// TIA Portal V17 export
// export: Created 2025-07-01T09:59:01.6776162Z, ExportSetting WithDefaults, DisplayName Totally Integrated Automation Portal, DisplayVersion V17 Update 8, DisplayName TIA Portal Openness, DisplayVersion V17 Update 8, DisplayName TIA Portal Version Control Interface, DisplayVersion V17, DisplayName SINAMICS Startdrive Advanced, DisplayVersion V17 SP2, DisplayName SINAMICS Startdrive G110M, G120, G120C, G120D, G120P, G115D, DisplayVersion V17 SP2, DisplayName SINAMICS Startdrive G130, G150, S120, S150, SINAMICS MV, S210, DisplayVersion V17 SP2, DisplayName STEP 7 Professional, DisplayVersion V17 Update 8, DisplayName SINUMERIK ONE STEP 7 Toolbox, DisplayVersion V17 Update 12, DisplayName SINUMERIK ONE PLC Basic Program Plus, DisplayVersion V17 Update 12, DisplayName SINUMERIK 840D sl STEP 7 Toolbox, DisplayVersion V17 Update 12, DisplayName STEP 7 Safety, DisplayVersion V17 Update 6, DisplayName WinCC Advanced, DisplayVersion V17 Update 8
FUNCTION "FC16015_METHOD_CALLS_U2_STA3_COAXIAL" : Void   // FC16015, LAD
{ S7_Optimized_Access := 'FALSE' }
VERSION : 0.1
// PC status values:
// 0-> Idle
// 1-> LaserCalibrating
// 2-> NozzleCalibrating
// 3-> JetCalibrating
// 4-> CladdingCalibrating
// 5-> NozzleAnalysis
// 6-> JetAnalysis
// 7-> CladdingAnalysis
// -1-> Error
// stored: AutoNumber false, IsIECCheckEnabled false, SetENOAutomatically false, UDAEnableTagReadback false
   VAR_TEMP
      AUX_WSTRING_PART_ID_STA3 : WString;
      AUX_WCHARS : Array[0..63] of WChar;
      index : Int;
      ALARM_AUX : Bool;
      TEMP_PULSE : Bool;
      STATUS_BLKMOV : Int;   // STATUS BLKMOV
      ZERO : Int;
   END_VAR
   VAR CONSTANT
      VERSIONS_MAJOR : UInt := 2;
      VERSIONS_MINOR : UInt := 0;
      FC_NUMBER : DInt := 16015;
   END_VAR
   VAR_TEMP   // added for the SCL form of the ladder/FBD networks
      _w1 : Bool;
      _w2 : Bool;
   END_VAR
BEGIN

REGION Network 1: ZERO
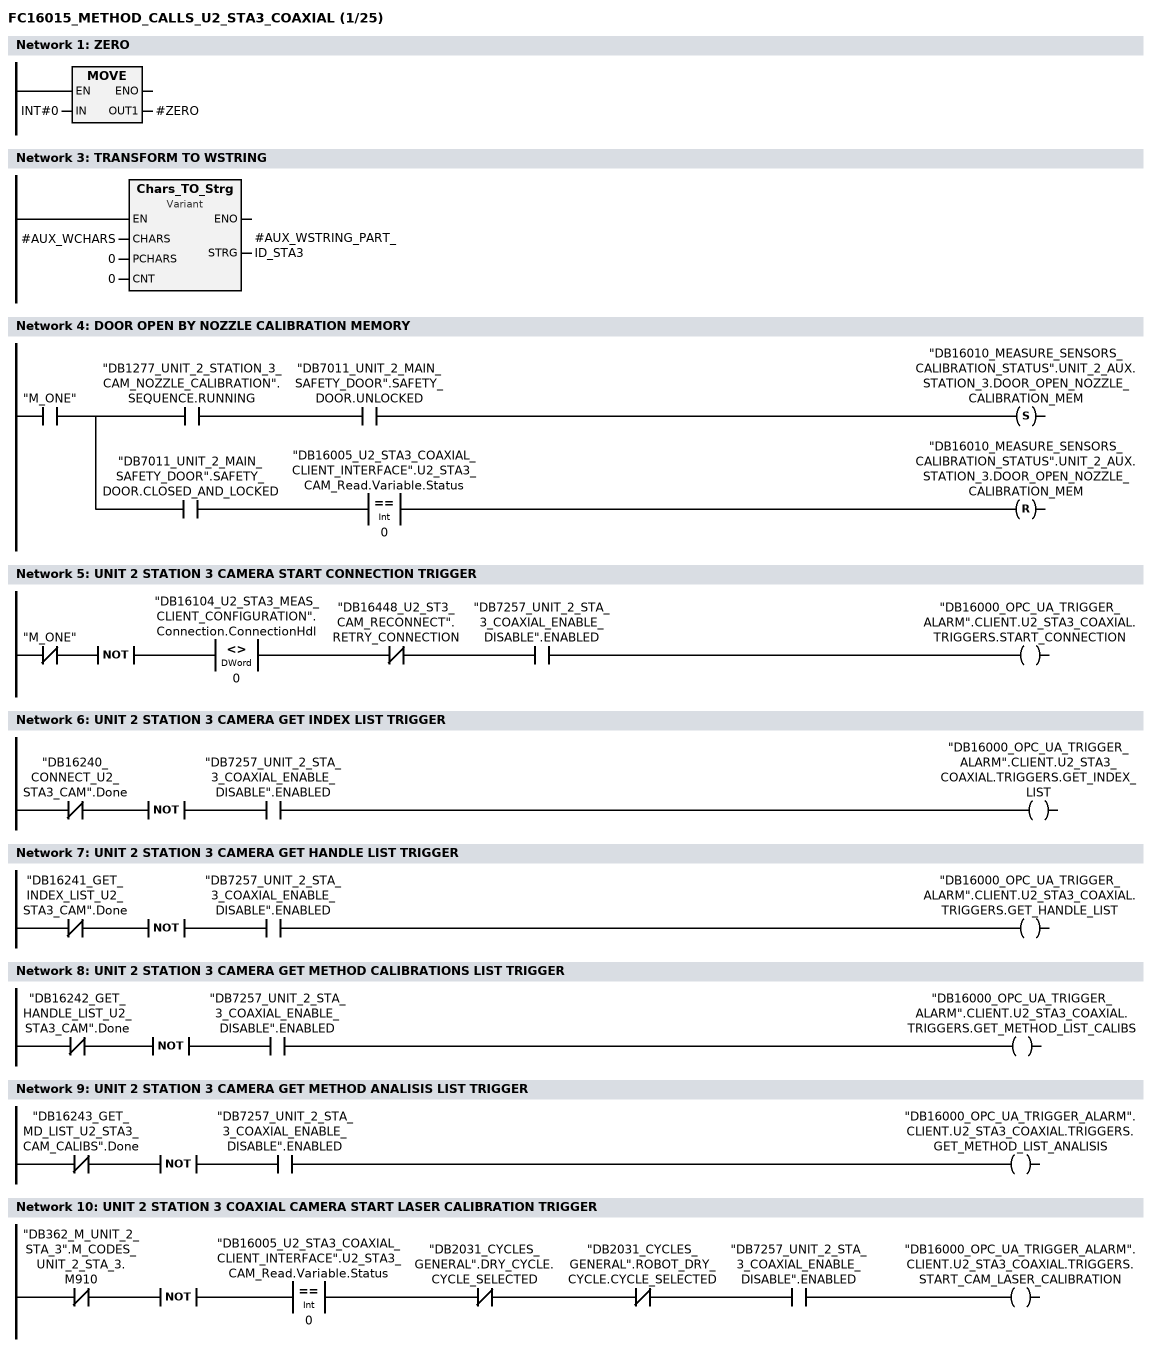
   RUNG wire#powerrail
      { S7_GenerateENO := "TRUE" } Move(in := INT#0, out1 => #ZERO)
   END_RUNG
   // the same network as SCL:
   #ZERO := INT#0;
END_REGION

REGION Network 2 (SCL): TRANSFORM TO WCHARS
   FOR #index := 0 TO 63 DO
       #AUX_WCHARS[#index] := CHAR_TO_WCHAR("DB8000_PART_STATUS".UNIT_2.STATION_3.PART_A.PART_ID[#index]);
   END_FOR;
END_REGION

REGION Network 3: TRANSFORM TO WSTRING
   RUNG wire#powerrail
      { S7_Templates := "[ptr_type := Variant, str_type := WString]" } Chars_TO_Strg(Chars := #AUX_WCHARS, pChars := 0, Cnt := 0, Strg => #AUX_WSTRING_PART_ID_STA3)
   END_RUNG
   // the same network as SCL:
   Chars_TO_Strg(Chars := #AUX_WCHARS, pChars := 0, Cnt := 0, Strg => #AUX_WSTRING_PART_ID_STA3);
END_REGION

REGION Network 4: DOOR OPEN BY NOZZLE CALIBRATION MEMORY
   RUNG wire#powerrail
      Contact( "M_ONE" )
      wire#w1
      Contact( "DB1277_UNIT_2_STATION_3_CAM_NOZZLE_CALIBRATION".SEQUENCE.RUNNING )
      Contact( "DB7011_UNIT_2_MAIN_SAFETY_DOOR".SAFETY_DOOR.UNLOCKED )
      S_Coil( "DB16010_MEASURE_SENSORS_CALIBRATION_STATUS".UNIT_2_AUX.STATION_3.DOOR_OPEN_NOZZLE_CALIBRATION_MEM )
   END_RUNG
   RUNG wire#w1
      Contact( "DB7011_UNIT_2_MAIN_SAFETY_DOOR".SAFETY_DOOR.CLOSED_AND_LOCKED )
      { S7_Templates := "SrcType := Int" } EQ_Contact(in1 := "DB16005_U2_STA3_COAXIAL_CLIENT_INTERFACE".U2_STA3_CAM_Read.Variable.Status, in2 := 0)
      R_Coil( "DB16010_MEASURE_SENSORS_CALIBRATION_STATUS".UNIT_2_AUX.STATION_3.DOOR_OPEN_NOZZLE_CALIBRATION_MEM )
   END_RUNG
   // the same network as SCL:
   IF "M_ONE" AND "DB1277_UNIT_2_STATION_3_CAM_NOZZLE_CALIBRATION".SEQUENCE.RUNNING AND "DB7011_UNIT_2_MAIN_SAFETY_DOOR".SAFETY_DOOR.UNLOCKED THEN
       "DB16010_MEASURE_SENSORS_CALIBRATION_STATUS".UNIT_2_AUX.STATION_3.DOOR_OPEN_NOZZLE_CALIBRATION_MEM := TRUE;
   END_IF;
   IF "M_ONE" AND "DB7011_UNIT_2_MAIN_SAFETY_DOOR".SAFETY_DOOR.CLOSED_AND_LOCKED AND ("DB16005_U2_STA3_COAXIAL_CLIENT_INTERFACE".U2_STA3_CAM_Read.Variable.Status = 0) THEN
       "DB16010_MEASURE_SENSORS_CALIBRATION_STATUS".UNIT_2_AUX.STATION_3.DOOR_OPEN_NOZZLE_CALIBRATION_MEM := FALSE;
   END_IF;
END_REGION

REGION Network 5: UNIT 2 STATION 3 CAMERA START CONNECTION TRIGGER
   RUNG wire#powerrail
      I_Contact( "M_ONE" )
      Not()
      { S7_Templates := "SrcType := DWord" } NE_Contact(in1 := "DB16104_U2_STA3_MEAS_CLIENT_CONFIGURATION".Connection.ConnectionHdl, in2 := 0)
      I_Contact( "DB16448_U2_ST3_CAM_RECONNECT".RETRY_CONNECTION )
      Contact( "DB7257_UNIT_2_STA_3_COAXIAL_ENABLE_DISABLE".ENABLED )
      Coil( "DB16000_OPC_UA_TRIGGER_ALARM".CLIENT.U2_STA3_COAXIAL.TRIGGERS.START_CONNECTION )
   END_RUNG
   // the same network as SCL:
   "DB16000_OPC_UA_TRIGGER_ALARM".CLIENT.U2_STA3_COAXIAL.TRIGGERS.START_CONNECTION := NOT (NOT "M_ONE") AND ("DB16104_U2_STA3_MEAS_CLIENT_CONFIGURATION".Connection.ConnectionHdl <> 0) AND NOT "DB16448_U2_ST3_CAM_RECONNECT".RETRY_CONNECTION AND "DB7257_UNIT_2_STA_3_COAXIAL_ENABLE_DISABLE".ENABLED;
END_REGION

REGION Network 6: UNIT 2 STATION 3 CAMERA GET INDEX LIST TRIGGER
   RUNG wire#powerrail
      I_Contact( "DB16240_CONNECT_U2_STA3_CAM".Done )
      Not()
      Contact( "DB7257_UNIT_2_STA_3_COAXIAL_ENABLE_DISABLE".ENABLED )
      Coil( "DB16000_OPC_UA_TRIGGER_ALARM".CLIENT.U2_STA3_COAXIAL.TRIGGERS.GET_INDEX_LIST )
   END_RUNG
   // the same network as SCL:
   "DB16000_OPC_UA_TRIGGER_ALARM".CLIENT.U2_STA3_COAXIAL.TRIGGERS.GET_INDEX_LIST := NOT (NOT "DB16240_CONNECT_U2_STA3_CAM".Done) AND "DB7257_UNIT_2_STA_3_COAXIAL_ENABLE_DISABLE".ENABLED;
END_REGION

REGION Network 7: UNIT 2 STATION 3 CAMERA GET HANDLE LIST TRIGGER
   RUNG wire#powerrail
      I_Contact( "DB16241_GET_INDEX_LIST_U2_STA3_CAM".Done )
      Not()
      Contact( "DB7257_UNIT_2_STA_3_COAXIAL_ENABLE_DISABLE".ENABLED )
      Coil( "DB16000_OPC_UA_TRIGGER_ALARM".CLIENT.U2_STA3_COAXIAL.TRIGGERS.GET_HANDLE_LIST )
   END_RUNG
   // the same network as SCL:
   "DB16000_OPC_UA_TRIGGER_ALARM".CLIENT.U2_STA3_COAXIAL.TRIGGERS.GET_HANDLE_LIST := NOT (NOT "DB16241_GET_INDEX_LIST_U2_STA3_CAM".Done) AND "DB7257_UNIT_2_STA_3_COAXIAL_ENABLE_DISABLE".ENABLED;
END_REGION

REGION Network 8: UNIT 2 STATION 3 CAMERA GET METHOD CALIBRATIONS LIST TRIGGER
   RUNG wire#powerrail
      I_Contact( "DB16242_GET_HANDLE_LIST_U2_STA3_CAM".Done )
      Not()
      Contact( "DB7257_UNIT_2_STA_3_COAXIAL_ENABLE_DISABLE".ENABLED )
      Coil( "DB16000_OPC_UA_TRIGGER_ALARM".CLIENT.U2_STA3_COAXIAL.TRIGGERS.GET_METHOD_LIST_CALIBS )
   END_RUNG
   // the same network as SCL:
   "DB16000_OPC_UA_TRIGGER_ALARM".CLIENT.U2_STA3_COAXIAL.TRIGGERS.GET_METHOD_LIST_CALIBS := NOT (NOT "DB16242_GET_HANDLE_LIST_U2_STA3_CAM".Done) AND "DB7257_UNIT_2_STA_3_COAXIAL_ENABLE_DISABLE".ENABLED;
END_REGION

REGION Network 9: UNIT 2 STATION 3 CAMERA GET METHOD ANALISIS LIST TRIGGER
   RUNG wire#powerrail
      I_Contact( "DB16243_GET_MD_LIST_U2_STA3_CAM_CALIBS".Done )
      Not()
      Contact( "DB7257_UNIT_2_STA_3_COAXIAL_ENABLE_DISABLE".ENABLED )
      Coil( "DB16000_OPC_UA_TRIGGER_ALARM".CLIENT.U2_STA3_COAXIAL.TRIGGERS.GET_METHOD_LIST_ANALISIS )
   END_RUNG
   // the same network as SCL:
   "DB16000_OPC_UA_TRIGGER_ALARM".CLIENT.U2_STA3_COAXIAL.TRIGGERS.GET_METHOD_LIST_ANALISIS := NOT (NOT "DB16243_GET_MD_LIST_U2_STA3_CAM_CALIBS".Done) AND "DB7257_UNIT_2_STA_3_COAXIAL_ENABLE_DISABLE".ENABLED;
END_REGION

REGION Network 10: UNIT 2 STATION 3 COAXIAL CAMERA START LASER CALIBRATION TRIGGER
   RUNG wire#powerrail
      I_Contact( "DB362_M_UNIT_2_STA_3".M_CODES_UNIT_2_STA_3.M910 )
      Not()
      { S7_Templates := "SrcType := Int" } EQ_Contact(in1 := "DB16005_U2_STA3_COAXIAL_CLIENT_INTERFACE".U2_STA3_CAM_Read.Variable.Status, in2 := 0)
      I_Contact( "DB2031_CYCLES_GENERAL".DRY_CYCLE.CYCLE_SELECTED )
      I_Contact( "DB2031_CYCLES_GENERAL".ROBOT_DRY_CYCLE.CYCLE_SELECTED )
      Contact( "DB7257_UNIT_2_STA_3_COAXIAL_ENABLE_DISABLE".ENABLED )
      Coil( "DB16000_OPC_UA_TRIGGER_ALARM".CLIENT.U2_STA3_COAXIAL.TRIGGERS.START_CAM_LASER_CALIBRATION )
   END_RUNG
   // the same network as SCL:
   "DB16000_OPC_UA_TRIGGER_ALARM".CLIENT.U2_STA3_COAXIAL.TRIGGERS.START_CAM_LASER_CALIBRATION := NOT (NOT "DB362_M_UNIT_2_STA_3".M_CODES_UNIT_2_STA_3.M910) AND ("DB16005_U2_STA3_COAXIAL_CLIENT_INTERFACE".U2_STA3_CAM_Read.Variable.Status = 0) AND NOT "DB2031_CYCLES_GENERAL".DRY_CYCLE.CYCLE_SELECTED AND NOT "DB2031_CYCLES_GENERAL".ROBOT_DRY_CYCLE.CYCLE_SELECTED AND "DB7257_UNIT_2_STA_3_COAXIAL_ENABLE_DISABLE".ENABLED;
END_REGION

REGION Network 11: UNIT 2 STATION 3 COAXIAL CAMERA START NOZZLE CALIBRATION TRIGGER
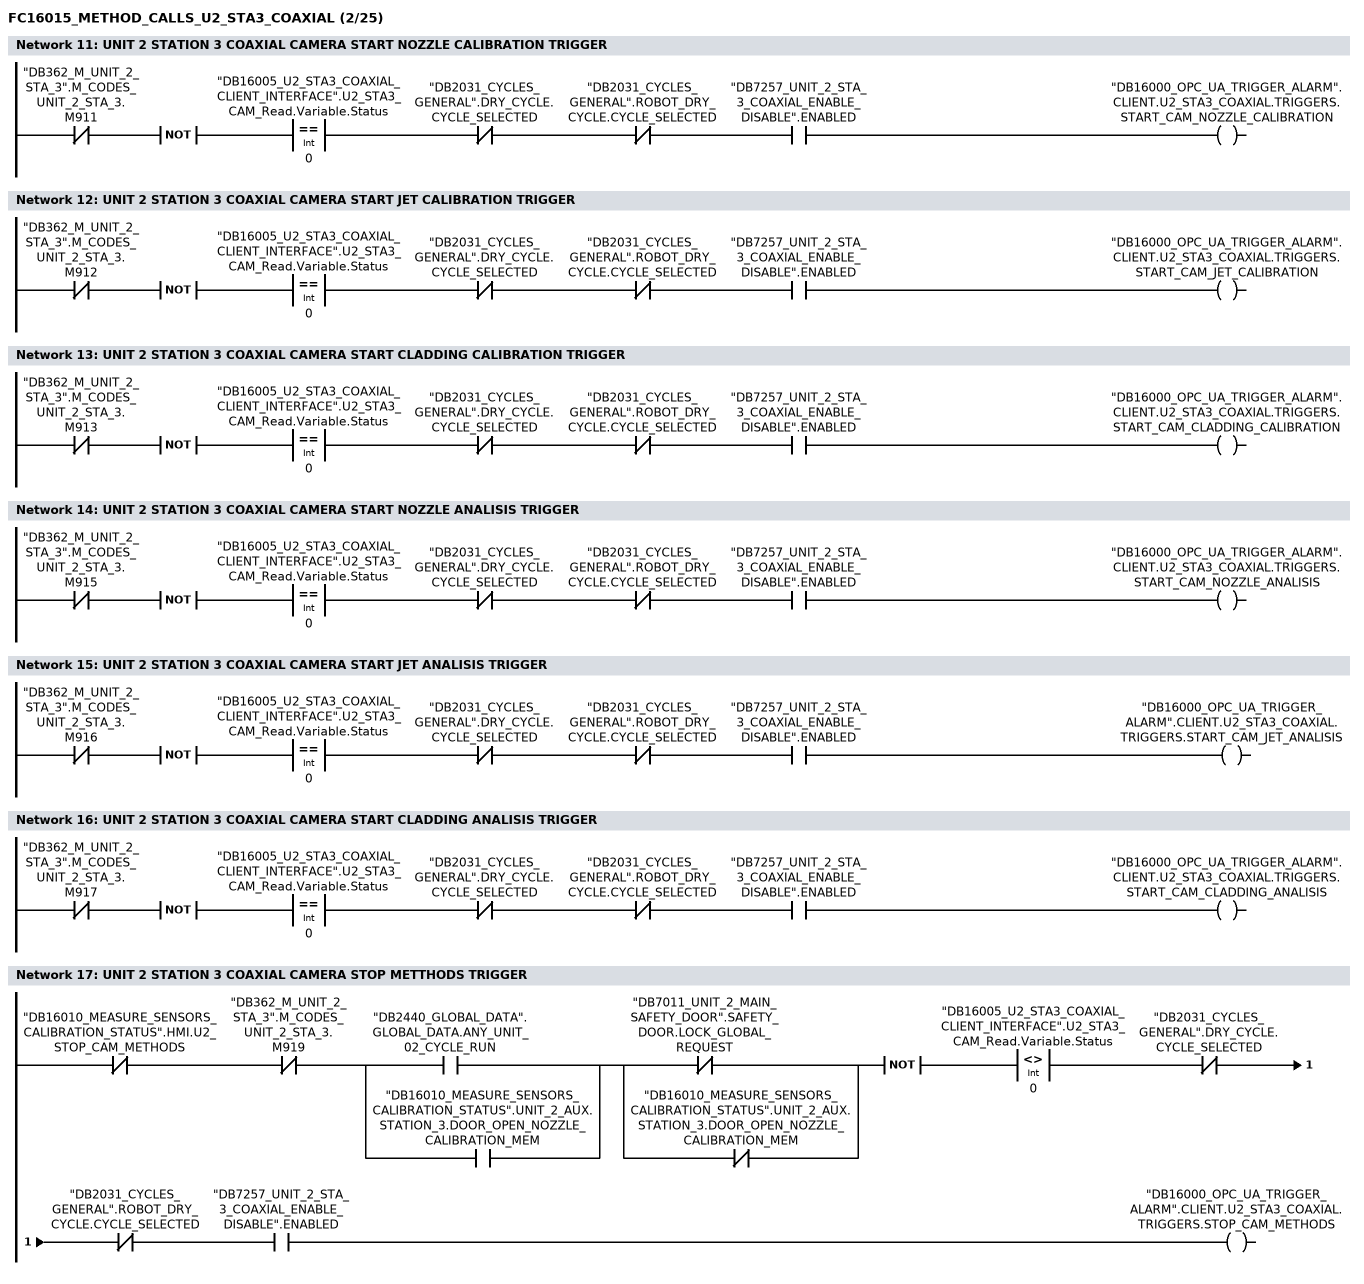
   RUNG wire#powerrail
      I_Contact( "DB362_M_UNIT_2_STA_3".M_CODES_UNIT_2_STA_3.M911 )
      Not()
      { S7_Templates := "SrcType := Int" } EQ_Contact(in1 := "DB16005_U2_STA3_COAXIAL_CLIENT_INTERFACE".U2_STA3_CAM_Read.Variable.Status, in2 := 0)
      I_Contact( "DB2031_CYCLES_GENERAL".DRY_CYCLE.CYCLE_SELECTED )
      I_Contact( "DB2031_CYCLES_GENERAL".ROBOT_DRY_CYCLE.CYCLE_SELECTED )
      Contact( "DB7257_UNIT_2_STA_3_COAXIAL_ENABLE_DISABLE".ENABLED )
      Coil( "DB16000_OPC_UA_TRIGGER_ALARM".CLIENT.U2_STA3_COAXIAL.TRIGGERS.START_CAM_NOZZLE_CALIBRATION )
   END_RUNG
   // the same network as SCL:
   "DB16000_OPC_UA_TRIGGER_ALARM".CLIENT.U2_STA3_COAXIAL.TRIGGERS.START_CAM_NOZZLE_CALIBRATION := NOT (NOT "DB362_M_UNIT_2_STA_3".M_CODES_UNIT_2_STA_3.M911) AND ("DB16005_U2_STA3_COAXIAL_CLIENT_INTERFACE".U2_STA3_CAM_Read.Variable.Status = 0) AND NOT "DB2031_CYCLES_GENERAL".DRY_CYCLE.CYCLE_SELECTED AND NOT "DB2031_CYCLES_GENERAL".ROBOT_DRY_CYCLE.CYCLE_SELECTED AND "DB7257_UNIT_2_STA_3_COAXIAL_ENABLE_DISABLE".ENABLED;
END_REGION

REGION Network 12: UNIT 2 STATION 3 COAXIAL CAMERA START JET CALIBRATION TRIGGER
   RUNG wire#powerrail
      I_Contact( "DB362_M_UNIT_2_STA_3".M_CODES_UNIT_2_STA_3.M912 )
      Not()
      { S7_Templates := "SrcType := Int" } EQ_Contact(in1 := "DB16005_U2_STA3_COAXIAL_CLIENT_INTERFACE".U2_STA3_CAM_Read.Variable.Status, in2 := 0)
      I_Contact( "DB2031_CYCLES_GENERAL".DRY_CYCLE.CYCLE_SELECTED )
      I_Contact( "DB2031_CYCLES_GENERAL".ROBOT_DRY_CYCLE.CYCLE_SELECTED )
      Contact( "DB7257_UNIT_2_STA_3_COAXIAL_ENABLE_DISABLE".ENABLED )
      Coil( "DB16000_OPC_UA_TRIGGER_ALARM".CLIENT.U2_STA3_COAXIAL.TRIGGERS.START_CAM_JET_CALIBRATION )
   END_RUNG
   // the same network as SCL:
   "DB16000_OPC_UA_TRIGGER_ALARM".CLIENT.U2_STA3_COAXIAL.TRIGGERS.START_CAM_JET_CALIBRATION := NOT (NOT "DB362_M_UNIT_2_STA_3".M_CODES_UNIT_2_STA_3.M912) AND ("DB16005_U2_STA3_COAXIAL_CLIENT_INTERFACE".U2_STA3_CAM_Read.Variable.Status = 0) AND NOT "DB2031_CYCLES_GENERAL".DRY_CYCLE.CYCLE_SELECTED AND NOT "DB2031_CYCLES_GENERAL".ROBOT_DRY_CYCLE.CYCLE_SELECTED AND "DB7257_UNIT_2_STA_3_COAXIAL_ENABLE_DISABLE".ENABLED;
END_REGION

REGION Network 13: UNIT 2 STATION 3 COAXIAL CAMERA START CLADDING CALIBRATION TRIGGER
   RUNG wire#powerrail
      I_Contact( "DB362_M_UNIT_2_STA_3".M_CODES_UNIT_2_STA_3.M913 )
      Not()
      { S7_Templates := "SrcType := Int" } EQ_Contact(in1 := "DB16005_U2_STA3_COAXIAL_CLIENT_INTERFACE".U2_STA3_CAM_Read.Variable.Status, in2 := 0)
      I_Contact( "DB2031_CYCLES_GENERAL".DRY_CYCLE.CYCLE_SELECTED )
      I_Contact( "DB2031_CYCLES_GENERAL".ROBOT_DRY_CYCLE.CYCLE_SELECTED )
      Contact( "DB7257_UNIT_2_STA_3_COAXIAL_ENABLE_DISABLE".ENABLED )
      Coil( "DB16000_OPC_UA_TRIGGER_ALARM".CLIENT.U2_STA3_COAXIAL.TRIGGERS.START_CAM_CLADDING_CALIBRATION )
   END_RUNG
   // the same network as SCL:
   "DB16000_OPC_UA_TRIGGER_ALARM".CLIENT.U2_STA3_COAXIAL.TRIGGERS.START_CAM_CLADDING_CALIBRATION := NOT (NOT "DB362_M_UNIT_2_STA_3".M_CODES_UNIT_2_STA_3.M913) AND ("DB16005_U2_STA3_COAXIAL_CLIENT_INTERFACE".U2_STA3_CAM_Read.Variable.Status = 0) AND NOT "DB2031_CYCLES_GENERAL".DRY_CYCLE.CYCLE_SELECTED AND NOT "DB2031_CYCLES_GENERAL".ROBOT_DRY_CYCLE.CYCLE_SELECTED AND "DB7257_UNIT_2_STA_3_COAXIAL_ENABLE_DISABLE".ENABLED;
END_REGION

REGION Network 14: UNIT 2 STATION 3 COAXIAL CAMERA START NOZZLE ANALISIS TRIGGER
   RUNG wire#powerrail
      I_Contact( "DB362_M_UNIT_2_STA_3".M_CODES_UNIT_2_STA_3.M915 )
      Not()
      { S7_Templates := "SrcType := Int" } EQ_Contact(in1 := "DB16005_U2_STA3_COAXIAL_CLIENT_INTERFACE".U2_STA3_CAM_Read.Variable.Status, in2 := 0)
      I_Contact( "DB2031_CYCLES_GENERAL".DRY_CYCLE.CYCLE_SELECTED )
      I_Contact( "DB2031_CYCLES_GENERAL".ROBOT_DRY_CYCLE.CYCLE_SELECTED )
      Contact( "DB7257_UNIT_2_STA_3_COAXIAL_ENABLE_DISABLE".ENABLED )
      Coil( "DB16000_OPC_UA_TRIGGER_ALARM".CLIENT.U2_STA3_COAXIAL.TRIGGERS.START_CAM_NOZZLE_ANALISIS )
   END_RUNG
   // the same network as SCL:
   "DB16000_OPC_UA_TRIGGER_ALARM".CLIENT.U2_STA3_COAXIAL.TRIGGERS.START_CAM_NOZZLE_ANALISIS := NOT (NOT "DB362_M_UNIT_2_STA_3".M_CODES_UNIT_2_STA_3.M915) AND ("DB16005_U2_STA3_COAXIAL_CLIENT_INTERFACE".U2_STA3_CAM_Read.Variable.Status = 0) AND NOT "DB2031_CYCLES_GENERAL".DRY_CYCLE.CYCLE_SELECTED AND NOT "DB2031_CYCLES_GENERAL".ROBOT_DRY_CYCLE.CYCLE_SELECTED AND "DB7257_UNIT_2_STA_3_COAXIAL_ENABLE_DISABLE".ENABLED;
END_REGION

REGION Network 15: UNIT 2 STATION 3 COAXIAL CAMERA START JET ANALISIS TRIGGER
   RUNG wire#powerrail
      I_Contact( "DB362_M_UNIT_2_STA_3".M_CODES_UNIT_2_STA_3.M916 )
      Not()
      { S7_Templates := "SrcType := Int" } EQ_Contact(in1 := "DB16005_U2_STA3_COAXIAL_CLIENT_INTERFACE".U2_STA3_CAM_Read.Variable.Status, in2 := 0)
      I_Contact( "DB2031_CYCLES_GENERAL".DRY_CYCLE.CYCLE_SELECTED )
      I_Contact( "DB2031_CYCLES_GENERAL".ROBOT_DRY_CYCLE.CYCLE_SELECTED )
      Contact( "DB7257_UNIT_2_STA_3_COAXIAL_ENABLE_DISABLE".ENABLED )
      Coil( "DB16000_OPC_UA_TRIGGER_ALARM".CLIENT.U2_STA3_COAXIAL.TRIGGERS.START_CAM_JET_ANALISIS )
   END_RUNG
   // the same network as SCL:
   "DB16000_OPC_UA_TRIGGER_ALARM".CLIENT.U2_STA3_COAXIAL.TRIGGERS.START_CAM_JET_ANALISIS := NOT (NOT "DB362_M_UNIT_2_STA_3".M_CODES_UNIT_2_STA_3.M916) AND ("DB16005_U2_STA3_COAXIAL_CLIENT_INTERFACE".U2_STA3_CAM_Read.Variable.Status = 0) AND NOT "DB2031_CYCLES_GENERAL".DRY_CYCLE.CYCLE_SELECTED AND NOT "DB2031_CYCLES_GENERAL".ROBOT_DRY_CYCLE.CYCLE_SELECTED AND "DB7257_UNIT_2_STA_3_COAXIAL_ENABLE_DISABLE".ENABLED;
END_REGION

REGION Network 16: UNIT 2 STATION 3 COAXIAL CAMERA START CLADDING ANALISIS TRIGGER
   RUNG wire#powerrail
      I_Contact( "DB362_M_UNIT_2_STA_3".M_CODES_UNIT_2_STA_3.M917 )
      Not()
      { S7_Templates := "SrcType := Int" } EQ_Contact(in1 := "DB16005_U2_STA3_COAXIAL_CLIENT_INTERFACE".U2_STA3_CAM_Read.Variable.Status, in2 := 0)
      I_Contact( "DB2031_CYCLES_GENERAL".DRY_CYCLE.CYCLE_SELECTED )
      I_Contact( "DB2031_CYCLES_GENERAL".ROBOT_DRY_CYCLE.CYCLE_SELECTED )
      Contact( "DB7257_UNIT_2_STA_3_COAXIAL_ENABLE_DISABLE".ENABLED )
      Coil( "DB16000_OPC_UA_TRIGGER_ALARM".CLIENT.U2_STA3_COAXIAL.TRIGGERS.START_CAM_CLADDING_ANALISIS )
   END_RUNG
   // the same network as SCL:
   "DB16000_OPC_UA_TRIGGER_ALARM".CLIENT.U2_STA3_COAXIAL.TRIGGERS.START_CAM_CLADDING_ANALISIS := NOT (NOT "DB362_M_UNIT_2_STA_3".M_CODES_UNIT_2_STA_3.M917) AND ("DB16005_U2_STA3_COAXIAL_CLIENT_INTERFACE".U2_STA3_CAM_Read.Variable.Status = 0) AND NOT "DB2031_CYCLES_GENERAL".DRY_CYCLE.CYCLE_SELECTED AND NOT "DB2031_CYCLES_GENERAL".ROBOT_DRY_CYCLE.CYCLE_SELECTED AND "DB7257_UNIT_2_STA_3_COAXIAL_ENABLE_DISABLE".ENABLED;
END_REGION

REGION Network 17: UNIT 2 STATION 3 COAXIAL CAMERA STOP METTHODS TRIGGER
   RUNG wire#powerrail
      I_Contact( "DB16010_MEASURE_SENSORS_CALIBRATION_STATUS".HMI.U2_STOP_CAM_METHODS )
      I_Contact( "DB362_M_UNIT_2_STA_3".M_CODES_UNIT_2_STA_3.M919 )
      wire#w1
      Contact( "DB2440_GLOBAL_DATA".GLOBAL_DATA.ANY_UNIT_02_CYCLE_RUN )
      wire#w2
      I_Contact( "DB7011_UNIT_2_MAIN_SAFETY_DOOR".SAFETY_DOOR.LOCK_GLOBAL_REQUEST )
      wire#w3
      Not()
      { S7_Templates := "SrcType := Int" } NE_Contact(in1 := "DB16005_U2_STA3_COAXIAL_CLIENT_INTERFACE".U2_STA3_CAM_Read.Variable.Status, in2 := 0)
      I_Contact( "DB2031_CYCLES_GENERAL".DRY_CYCLE.CYCLE_SELECTED )
      I_Contact( "DB2031_CYCLES_GENERAL".ROBOT_DRY_CYCLE.CYCLE_SELECTED )
      Contact( "DB7257_UNIT_2_STA_3_COAXIAL_ENABLE_DISABLE".ENABLED )
      Coil( "DB16000_OPC_UA_TRIGGER_ALARM".CLIENT.U2_STA3_COAXIAL.TRIGGERS.STOP_CAM_METHODS )
   END_RUNG
   RUNG wire#w1
      Contact( "DB16010_MEASURE_SENSORS_CALIBRATION_STATUS".UNIT_2_AUX.STATION_3.DOOR_OPEN_NOZZLE_CALIBRATION_MEM )
   END_RUNG wire#w2
   RUNG wire#w2
      I_Contact( "DB16010_MEASURE_SENSORS_CALIBRATION_STATUS".UNIT_2_AUX.STATION_3.DOOR_OPEN_NOZZLE_CALIBRATION_MEM )
   END_RUNG wire#w3
   // the same network as SCL:
   "DB16000_OPC_UA_TRIGGER_ALARM".CLIENT.U2_STA3_COAXIAL.TRIGGERS.STOP_CAM_METHODS := NOT (NOT "DB16010_MEASURE_SENSORS_CALIBRATION_STATUS".HMI.U2_STOP_CAM_METHODS AND NOT "DB362_M_UNIT_2_STA_3".M_CODES_UNIT_2_STA_3.M919 AND ("DB2440_GLOBAL_DATA".GLOBAL_DATA.ANY_UNIT_02_CYCLE_RUN OR "DB16010_MEASURE_SENSORS_CALIBRATION_STATUS".UNIT_2_AUX.STATION_3.DOOR_OPEN_NOZZLE_CALIBRATION_MEM) AND (NOT "DB7011_UNIT_2_MAIN_SAFETY_DOOR".SAFETY_DOOR.LOCK_GLOBAL_REQUEST OR NOT "DB16010_MEASURE_SENSORS_CALIBRATION_STATUS".UNIT_2_AUX.STATION_3.DOOR_OPEN_NOZZLE_CALIBRATION_MEM)) AND ("DB16005_U2_STA3_COAXIAL_CLIENT_INTERFACE".U2_STA3_CAM_Read.Variable.Status <> 0) AND NOT "DB2031_CYCLES_GENERAL".DRY_CYCLE.CYCLE_SELECTED AND NOT "DB2031_CYCLES_GENERAL".ROBOT_DRY_CYCLE.CYCLE_SELECTED AND "DB7257_UNIT_2_STA_3_COAXIAL_ENABLE_DISABLE".ENABLED;
END_REGION

REGION Network 18: UNIT 2 STATION 3 COAXIAL CAMERA RESET PC TRIGGER
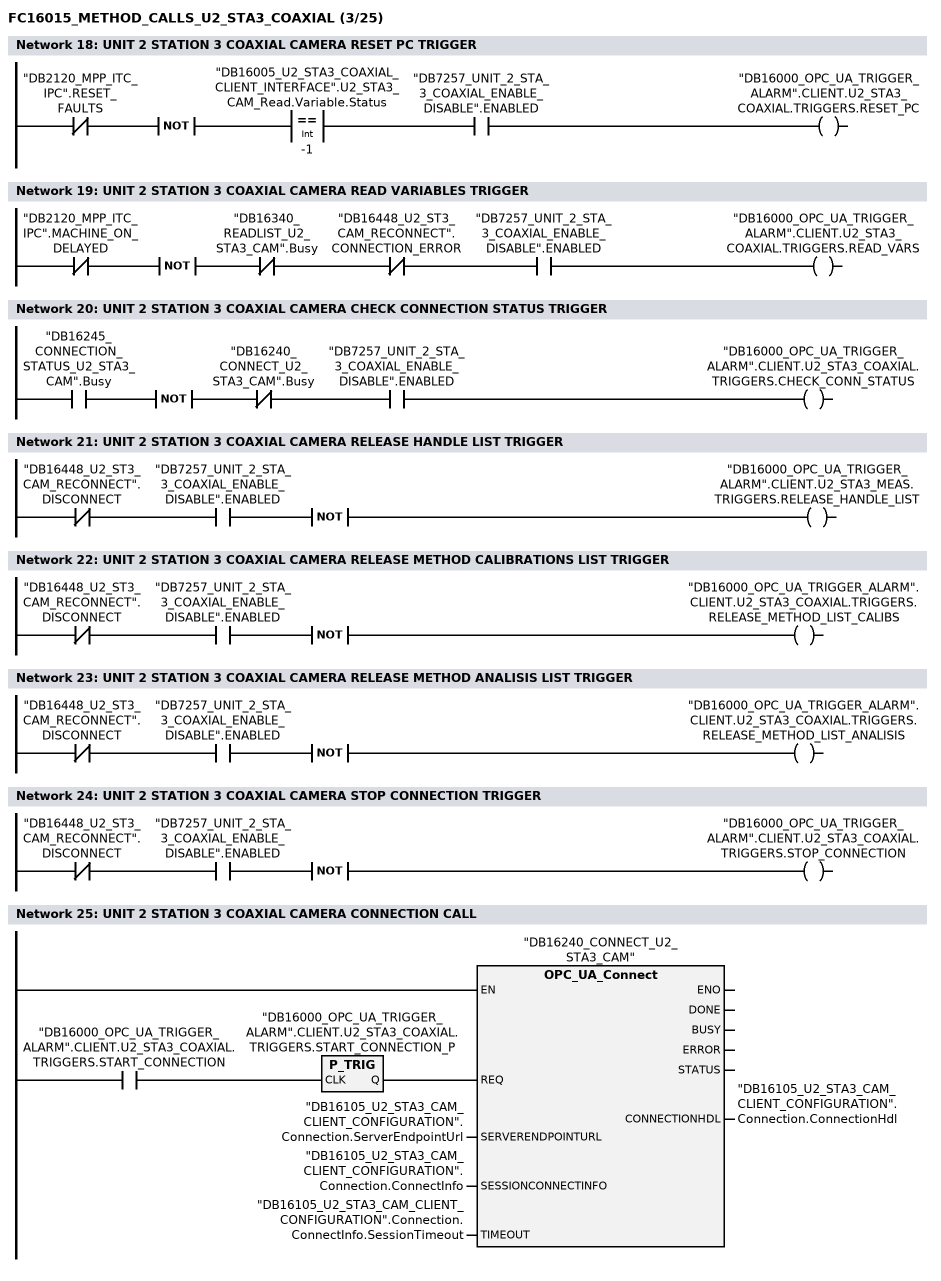
   RUNG wire#powerrail
      I_Contact( "DB2120_MPP_ITC_IPC".RESET_FAULTS )
      Not()
      { S7_Templates := "SrcType := Int" } EQ_Contact(in1 := "DB16005_U2_STA3_COAXIAL_CLIENT_INTERFACE".U2_STA3_CAM_Read.Variable.Status, in2 := -1)
      Contact( "DB7257_UNIT_2_STA_3_COAXIAL_ENABLE_DISABLE".ENABLED )
      Coil( "DB16000_OPC_UA_TRIGGER_ALARM".CLIENT.U2_STA3_COAXIAL.TRIGGERS.RESET_PC )
   END_RUNG
   // the same network as SCL:
   "DB16000_OPC_UA_TRIGGER_ALARM".CLIENT.U2_STA3_COAXIAL.TRIGGERS.RESET_PC := NOT (NOT "DB2120_MPP_ITC_IPC".RESET_FAULTS) AND ("DB16005_U2_STA3_COAXIAL_CLIENT_INTERFACE".U2_STA3_CAM_Read.Variable.Status = (-1)) AND "DB7257_UNIT_2_STA_3_COAXIAL_ENABLE_DISABLE".ENABLED;
END_REGION

REGION Network 19: UNIT 2 STATION 3 COAXIAL CAMERA READ VARIABLES TRIGGER
   RUNG wire#powerrail
      I_Contact( "DB2120_MPP_ITC_IPC".MACHINE_ON_DELAYED )
      Not()
      I_Contact( "DB16340_READLIST_U2_STA3_CAM".Busy )
      I_Contact( "DB16448_U2_ST3_CAM_RECONNECT".CONNECTION_ERROR )
      Contact( "DB7257_UNIT_2_STA_3_COAXIAL_ENABLE_DISABLE".ENABLED )
      Coil( "DB16000_OPC_UA_TRIGGER_ALARM".CLIENT.U2_STA3_COAXIAL.TRIGGERS.READ_VARS )
   END_RUNG
   // the same network as SCL:
   "DB16000_OPC_UA_TRIGGER_ALARM".CLIENT.U2_STA3_COAXIAL.TRIGGERS.READ_VARS := NOT (NOT "DB2120_MPP_ITC_IPC".MACHINE_ON_DELAYED) AND NOT "DB16340_READLIST_U2_STA3_CAM".Busy AND NOT "DB16448_U2_ST3_CAM_RECONNECT".CONNECTION_ERROR AND "DB7257_UNIT_2_STA_3_COAXIAL_ENABLE_DISABLE".ENABLED;
END_REGION

REGION Network 20: UNIT 2 STATION 3 COAXIAL CAMERA CHECK CONNECTION STATUS TRIGGER
   RUNG wire#powerrail
      Contact( "DB16245_CONNECTION_STATUS_U2_STA3_CAM".Busy )
      Not()
      I_Contact( "DB16240_CONNECT_U2_STA3_CAM".Busy )
      Contact( "DB7257_UNIT_2_STA_3_COAXIAL_ENABLE_DISABLE".ENABLED )
      Coil( "DB16000_OPC_UA_TRIGGER_ALARM".CLIENT.U2_STA3_COAXIAL.TRIGGERS.CHECK_CONN_STATUS )
   END_RUNG
   // the same network as SCL:
   "DB16000_OPC_UA_TRIGGER_ALARM".CLIENT.U2_STA3_COAXIAL.TRIGGERS.CHECK_CONN_STATUS := NOT "DB16245_CONNECTION_STATUS_U2_STA3_CAM".Busy AND NOT "DB16240_CONNECT_U2_STA3_CAM".Busy AND "DB7257_UNIT_2_STA_3_COAXIAL_ENABLE_DISABLE".ENABLED;
END_REGION

REGION Network 21: UNIT 2 STATION 3 COAXIAL CAMERA RELEASE HANDLE LIST TRIGGER
   RUNG wire#powerrail
      I_Contact( "DB16448_U2_ST3_CAM_RECONNECT".DISCONNECT )
      Contact( "DB7257_UNIT_2_STA_3_COAXIAL_ENABLE_DISABLE".ENABLED )
      Not()
      Coil( "DB16000_OPC_UA_TRIGGER_ALARM".CLIENT.U2_STA3_MEAS.TRIGGERS.RELEASE_HANDLE_LIST )
   END_RUNG
   // the same network as SCL:
   "DB16000_OPC_UA_TRIGGER_ALARM".CLIENT.U2_STA3_MEAS.TRIGGERS.RELEASE_HANDLE_LIST := NOT (NOT "DB16448_U2_ST3_CAM_RECONNECT".DISCONNECT AND "DB7257_UNIT_2_STA_3_COAXIAL_ENABLE_DISABLE".ENABLED);
END_REGION

REGION Network 22: UNIT 2 STATION 3 COAXIAL CAMERA RELEASE METHOD CALIBRATIONS LIST TRIGGER
   RUNG wire#powerrail
      I_Contact( "DB16448_U2_ST3_CAM_RECONNECT".DISCONNECT )
      Contact( "DB7257_UNIT_2_STA_3_COAXIAL_ENABLE_DISABLE".ENABLED )
      Not()
      Coil( "DB16000_OPC_UA_TRIGGER_ALARM".CLIENT.U2_STA3_COAXIAL.TRIGGERS.RELEASE_METHOD_LIST_CALIBS )
   END_RUNG
   // the same network as SCL:
   "DB16000_OPC_UA_TRIGGER_ALARM".CLIENT.U2_STA3_COAXIAL.TRIGGERS.RELEASE_METHOD_LIST_CALIBS := NOT (NOT "DB16448_U2_ST3_CAM_RECONNECT".DISCONNECT AND "DB7257_UNIT_2_STA_3_COAXIAL_ENABLE_DISABLE".ENABLED);
END_REGION

REGION Network 23: UNIT 2 STATION 3 COAXIAL CAMERA RELEASE METHOD ANALISIS LIST TRIGGER
   RUNG wire#powerrail
      I_Contact( "DB16448_U2_ST3_CAM_RECONNECT".DISCONNECT )
      Contact( "DB7257_UNIT_2_STA_3_COAXIAL_ENABLE_DISABLE".ENABLED )
      Not()
      Coil( "DB16000_OPC_UA_TRIGGER_ALARM".CLIENT.U2_STA3_COAXIAL.TRIGGERS.RELEASE_METHOD_LIST_ANALISIS )
   END_RUNG
   // the same network as SCL:
   "DB16000_OPC_UA_TRIGGER_ALARM".CLIENT.U2_STA3_COAXIAL.TRIGGERS.RELEASE_METHOD_LIST_ANALISIS := NOT (NOT "DB16448_U2_ST3_CAM_RECONNECT".DISCONNECT AND "DB7257_UNIT_2_STA_3_COAXIAL_ENABLE_DISABLE".ENABLED);
END_REGION

REGION Network 24: UNIT 2 STATION 3 COAXIAL CAMERA STOP CONNECTION TRIGGER
   RUNG wire#powerrail
      I_Contact( "DB16448_U2_ST3_CAM_RECONNECT".DISCONNECT )
      Contact( "DB7257_UNIT_2_STA_3_COAXIAL_ENABLE_DISABLE".ENABLED )
      Not()
      Coil( "DB16000_OPC_UA_TRIGGER_ALARM".CLIENT.U2_STA3_COAXIAL.TRIGGERS.STOP_CONNECTION )
   END_RUNG
   // the same network as SCL:
   "DB16000_OPC_UA_TRIGGER_ALARM".CLIENT.U2_STA3_COAXIAL.TRIGGERS.STOP_CONNECTION := NOT (NOT "DB16448_U2_ST3_CAM_RECONNECT".DISCONNECT AND "DB7257_UNIT_2_STA_3_COAXIAL_ENABLE_DISABLE".ENABLED);
END_REGION

REGION Network 25: UNIT 2 STATION 3 COAXIAL CAMERA CONNECTION CALL
   RUNG wire#powerrail
      "DB16240_CONNECT_U2_STA3_CAM".OPC_UA_Connect(REQ := wire#w1, ServerEndpointUrl := "DB16105_U2_STA3_CAM_CLIENT_CONFIGURATION".Connection.ServerEndpointUrl, SessionConnectInfo := "DB16105_U2_STA3_CAM_CLIENT_CONFIGURATION".Connection.ConnectInfo, Timeout := "DB16105_U2_STA3_CAM_CLIENT_CONFIGURATION".Connection.ConnectInfo.SessionTimeout, Done =>, Busy =>, Error =>, Status =>, ConnectionHdl => "DB16105_U2_STA3_CAM_CLIENT_CONFIGURATION".Connection.ConnectionHdl)
   END_RUNG
   RUNG wire#powerrail
      Contact( "DB16000_OPC_UA_TRIGGER_ALARM".CLIENT.U2_STA3_COAXIAL.TRIGGERS.START_CONNECTION )
      P_Trig( "DB16000_OPC_UA_TRIGGER_ALARM".CLIENT.U2_STA3_COAXIAL.TRIGGERS.START_CONNECTION_P )
   END_RUNG wire#w1
   // the same network as SCL:
   #_w1 := "DB16000_OPC_UA_TRIGGER_ALARM".CLIENT.U2_STA3_COAXIAL.TRIGGERS.START_CONNECTION AND NOT "DB16000_OPC_UA_TRIGGER_ALARM".CLIENT.U2_STA3_COAXIAL.TRIGGERS.START_CONNECTION_P;   // rising edge
   "DB16000_OPC_UA_TRIGGER_ALARM".CLIENT.U2_STA3_COAXIAL.TRIGGERS.START_CONNECTION_P := "DB16000_OPC_UA_TRIGGER_ALARM".CLIENT.U2_STA3_COAXIAL.TRIGGERS.START_CONNECTION;
   "DB16240_CONNECT_U2_STA3_CAM"(REQ := #_w1,   // OPC_UA_Connect
                           ServerEndpointUrl := "DB16105_U2_STA3_CAM_CLIENT_CONFIGURATION".Connection.ServerEndpointUrl,
                           SessionConnectInfo := "DB16105_U2_STA3_CAM_CLIENT_CONFIGURATION".Connection.ConnectInfo,
                           Timeout := "DB16105_U2_STA3_CAM_CLIENT_CONFIGURATION".Connection.ConnectInfo.SessionTimeout,
                           ConnectionHdl => "DB16105_U2_STA3_CAM_CLIENT_CONFIGURATION".Connection.ConnectionHdl);
END_REGION

REGION Network 26: UNIT 2 STATION 3 COAXIAL CAMERA GET INDEX LIST CALL
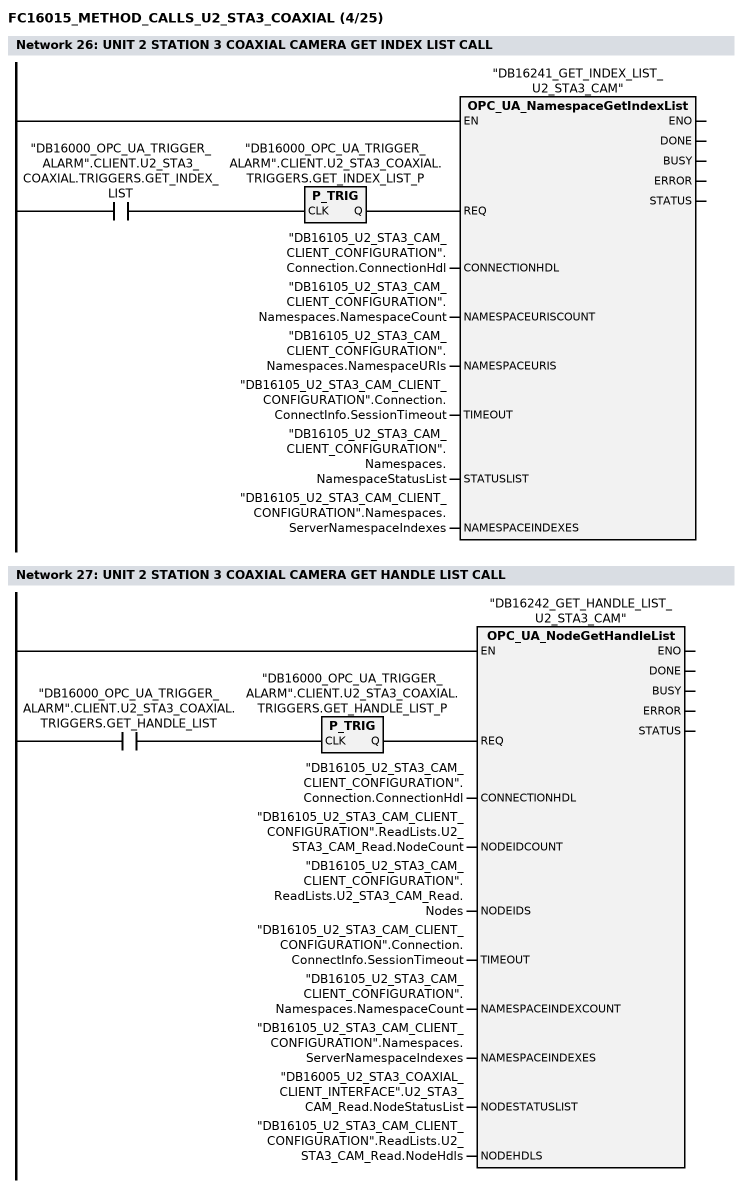
   RUNG wire#powerrail
      "DB16241_GET_INDEX_LIST_U2_STA3_CAM".OPC_UA_NamespaceGetIndexList(REQ := wire#w1, ConnectionHdl := "DB16105_U2_STA3_CAM_CLIENT_CONFIGURATION".Connection.ConnectionHdl, NamespaceUrisCount := "DB16105_U2_STA3_CAM_CLIENT_CONFIGURATION".Namespaces.NamespaceCount, NamespaceUris := "DB16105_U2_STA3_CAM_CLIENT_CONFIGURATION".Namespaces.NamespaceURIs, Timeout := "DB16105_U2_STA3_CAM_CLIENT_CONFIGURATION".Connection.ConnectInfo.SessionTimeout, StatusList := "DB16105_U2_STA3_CAM_CLIENT_CONFIGURATION".Namespaces.NamespaceStatusList, NamespaceIndexes := "DB16105_U2_STA3_CAM_CLIENT_CONFIGURATION".Namespaces.ServerNamespaceIndexes, Done =>, Busy =>, Error =>, Status =>)
   END_RUNG
   RUNG wire#powerrail
      Contact( "DB16000_OPC_UA_TRIGGER_ALARM".CLIENT.U2_STA3_COAXIAL.TRIGGERS.GET_INDEX_LIST )
      P_Trig( "DB16000_OPC_UA_TRIGGER_ALARM".CLIENT.U2_STA3_COAXIAL.TRIGGERS.GET_INDEX_LIST_P )
   END_RUNG wire#w1
   // the same network as SCL:
   #_w1 := "DB16000_OPC_UA_TRIGGER_ALARM".CLIENT.U2_STA3_COAXIAL.TRIGGERS.GET_INDEX_LIST AND NOT "DB16000_OPC_UA_TRIGGER_ALARM".CLIENT.U2_STA3_COAXIAL.TRIGGERS.GET_INDEX_LIST_P;   // rising edge
   "DB16000_OPC_UA_TRIGGER_ALARM".CLIENT.U2_STA3_COAXIAL.TRIGGERS.GET_INDEX_LIST_P := "DB16000_OPC_UA_TRIGGER_ALARM".CLIENT.U2_STA3_COAXIAL.TRIGGERS.GET_INDEX_LIST;
   "DB16241_GET_INDEX_LIST_U2_STA3_CAM"(REQ := #_w1,   // OPC_UA_NamespaceGetIndexList
                           ConnectionHdl := "DB16105_U2_STA3_CAM_CLIENT_CONFIGURATION".Connection.ConnectionHdl,
                           NamespaceUrisCount := "DB16105_U2_STA3_CAM_CLIENT_CONFIGURATION".Namespaces.NamespaceCount,
                           NamespaceUris := "DB16105_U2_STA3_CAM_CLIENT_CONFIGURATION".Namespaces.NamespaceURIs,
                           Timeout := "DB16105_U2_STA3_CAM_CLIENT_CONFIGURATION".Connection.ConnectInfo.SessionTimeout,
                           StatusList := "DB16105_U2_STA3_CAM_CLIENT_CONFIGURATION".Namespaces.NamespaceStatusList,
                           NamespaceIndexes := "DB16105_U2_STA3_CAM_CLIENT_CONFIGURATION".Namespaces.ServerNamespaceIndexes);
END_REGION

REGION Network 27: UNIT 2 STATION 3 COAXIAL CAMERA GET HANDLE LIST CALL
   RUNG wire#powerrail
      "DB16242_GET_HANDLE_LIST_U2_STA3_CAM".OPC_UA_NodeGetHandleList(REQ := wire#w1, ConnectionHdl := "DB16105_U2_STA3_CAM_CLIENT_CONFIGURATION".Connection.ConnectionHdl, NodeIDCount := "DB16105_U2_STA3_CAM_CLIENT_CONFIGURATION".ReadLists.U2_STA3_CAM_Read.NodeCount, NodeIDs := "DB16105_U2_STA3_CAM_CLIENT_CONFIGURATION".ReadLists.U2_STA3_CAM_Read.Nodes, Timeout := "DB16105_U2_STA3_CAM_CLIENT_CONFIGURATION".Connection.ConnectInfo.SessionTimeout, NamespaceIndexCount := "DB16105_U2_STA3_CAM_CLIENT_CONFIGURATION".Namespaces.NamespaceCount, NamespaceIndexes := "DB16105_U2_STA3_CAM_CLIENT_CONFIGURATION".Namespaces.ServerNamespaceIndexes, NodeStatusList := "DB16005_U2_STA3_COAXIAL_CLIENT_INTERFACE".U2_STA3_CAM_Read.NodeStatusList, NodeHdls := "DB16105_U2_STA3_CAM_CLIENT_CONFIGURATION".ReadLists.U2_STA3_CAM_Read.NodeHdls, Done =>, Busy =>, Error =>, Status =>)
   END_RUNG
   RUNG wire#powerrail
      Contact( "DB16000_OPC_UA_TRIGGER_ALARM".CLIENT.U2_STA3_COAXIAL.TRIGGERS.GET_HANDLE_LIST )
      P_Trig( "DB16000_OPC_UA_TRIGGER_ALARM".CLIENT.U2_STA3_COAXIAL.TRIGGERS.GET_HANDLE_LIST_P )
   END_RUNG wire#w1
   // the same network as SCL:
   #_w1 := "DB16000_OPC_UA_TRIGGER_ALARM".CLIENT.U2_STA3_COAXIAL.TRIGGERS.GET_HANDLE_LIST AND NOT "DB16000_OPC_UA_TRIGGER_ALARM".CLIENT.U2_STA3_COAXIAL.TRIGGERS.GET_HANDLE_LIST_P;   // rising edge
   "DB16000_OPC_UA_TRIGGER_ALARM".CLIENT.U2_STA3_COAXIAL.TRIGGERS.GET_HANDLE_LIST_P := "DB16000_OPC_UA_TRIGGER_ALARM".CLIENT.U2_STA3_COAXIAL.TRIGGERS.GET_HANDLE_LIST;
   "DB16242_GET_HANDLE_LIST_U2_STA3_CAM"(REQ := #_w1,   // OPC_UA_NodeGetHandleList
                           ConnectionHdl := "DB16105_U2_STA3_CAM_CLIENT_CONFIGURATION".Connection.ConnectionHdl,
                           NodeIDCount := "DB16105_U2_STA3_CAM_CLIENT_CONFIGURATION".ReadLists.U2_STA3_CAM_Read.NodeCount,
                           NodeIDs := "DB16105_U2_STA3_CAM_CLIENT_CONFIGURATION".ReadLists.U2_STA3_CAM_Read.Nodes,
                           Timeout := "DB16105_U2_STA3_CAM_CLIENT_CONFIGURATION".Connection.ConnectInfo.SessionTimeout,
                           NamespaceIndexCount := "DB16105_U2_STA3_CAM_CLIENT_CONFIGURATION".Namespaces.NamespaceCount,
                           NamespaceIndexes := "DB16105_U2_STA3_CAM_CLIENT_CONFIGURATION".Namespaces.ServerNamespaceIndexes,
                           NodeStatusList := "DB16005_U2_STA3_COAXIAL_CLIENT_INTERFACE".U2_STA3_CAM_Read.NodeStatusList,
                           NodeHdls := "DB16105_U2_STA3_CAM_CLIENT_CONFIGURATION".ReadLists.U2_STA3_CAM_Read.NodeHdls);
END_REGION

REGION Network 28: UNIT 2 STATION 3 COAXIAL CAMERA GET METHOD CALIBRATIONS LIST CALL
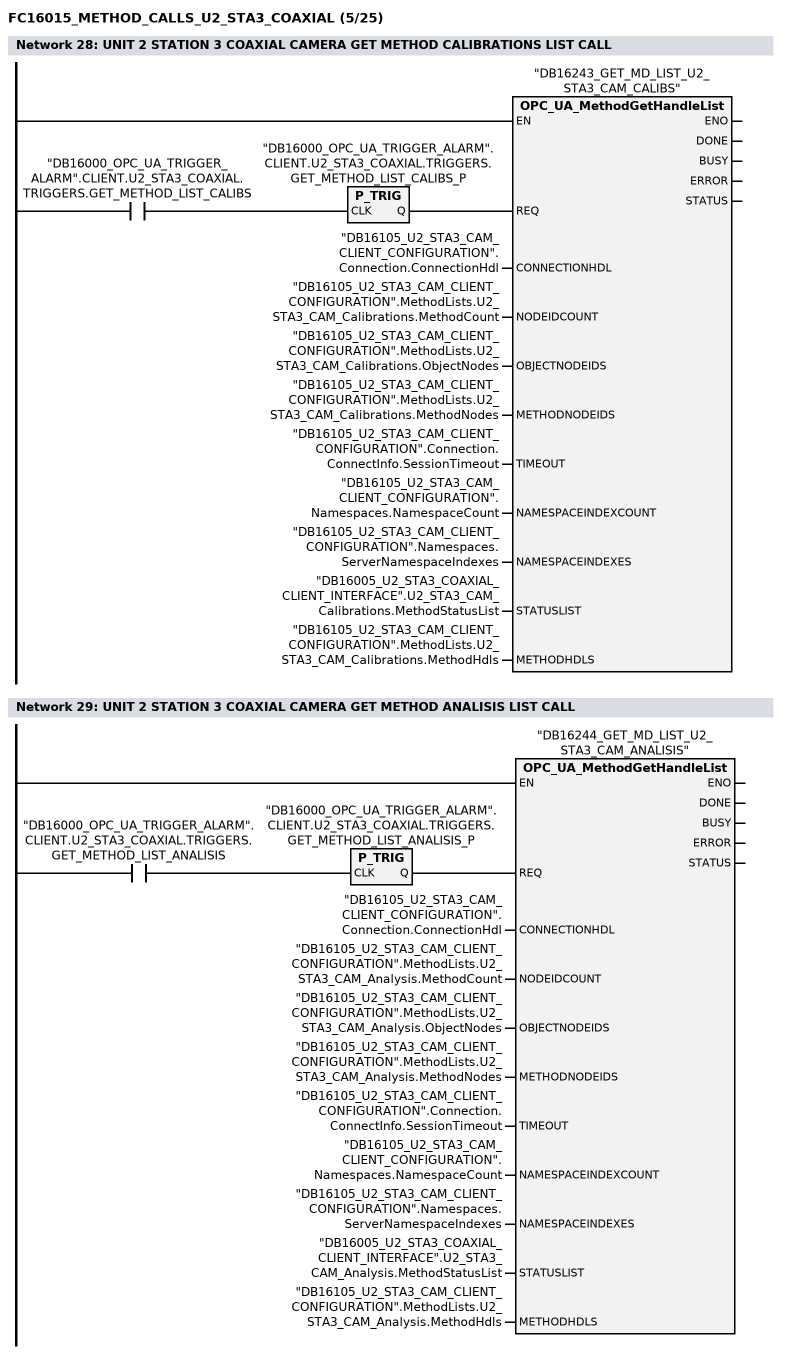
   RUNG wire#powerrail
      "DB16243_GET_MD_LIST_U2_STA3_CAM_CALIBS".OPC_UA_MethodGetHandleList(REQ := wire#w1, ConnectionHdl := "DB16105_U2_STA3_CAM_CLIENT_CONFIGURATION".Connection.ConnectionHdl, NodeIDCount := "DB16105_U2_STA3_CAM_CLIENT_CONFIGURATION".MethodLists.U2_STA3_CAM_Calibrations.MethodCount, ObjectNodeIDs := "DB16105_U2_STA3_CAM_CLIENT_CONFIGURATION".MethodLists.U2_STA3_CAM_Calibrations.ObjectNodes, MethodNodeIDs := "DB16105_U2_STA3_CAM_CLIENT_CONFIGURATION".MethodLists.U2_STA3_CAM_Calibrations.MethodNodes, Timeout := "DB16105_U2_STA3_CAM_CLIENT_CONFIGURATION".Connection.ConnectInfo.SessionTimeout, NamespaceIndexCount := "DB16105_U2_STA3_CAM_CLIENT_CONFIGURATION".Namespaces.NamespaceCount, NamespaceIndexes := "DB16105_U2_STA3_CAM_CLIENT_CONFIGURATION".Namespaces.ServerNamespaceIndexes, StatusList := "DB16005_U2_STA3_COAXIAL_CLIENT_INTERFACE".U2_STA3_CAM_Calibrations.MethodStatusList, MethodHdls := "DB16105_U2_STA3_CAM_CLIENT_CONFIGURATION".MethodLists.U2_STA3_CAM_Calibrations.MethodHdls, Done =>, Busy =>, Error =>, Status =>)
   END_RUNG
   RUNG wire#powerrail
      Contact( "DB16000_OPC_UA_TRIGGER_ALARM".CLIENT.U2_STA3_COAXIAL.TRIGGERS.GET_METHOD_LIST_CALIBS )
      P_Trig( "DB16000_OPC_UA_TRIGGER_ALARM".CLIENT.U2_STA3_COAXIAL.TRIGGERS.GET_METHOD_LIST_CALIBS_P )
   END_RUNG wire#w1
   // the same network as SCL:
   #_w1 := "DB16000_OPC_UA_TRIGGER_ALARM".CLIENT.U2_STA3_COAXIAL.TRIGGERS.GET_METHOD_LIST_CALIBS AND NOT "DB16000_OPC_UA_TRIGGER_ALARM".CLIENT.U2_STA3_COAXIAL.TRIGGERS.GET_METHOD_LIST_CALIBS_P;   // rising edge
   "DB16000_OPC_UA_TRIGGER_ALARM".CLIENT.U2_STA3_COAXIAL.TRIGGERS.GET_METHOD_LIST_CALIBS_P := "DB16000_OPC_UA_TRIGGER_ALARM".CLIENT.U2_STA3_COAXIAL.TRIGGERS.GET_METHOD_LIST_CALIBS;
   "DB16243_GET_MD_LIST_U2_STA3_CAM_CALIBS"(REQ := #_w1,   // OPC_UA_MethodGetHandleList
                           ConnectionHdl := "DB16105_U2_STA3_CAM_CLIENT_CONFIGURATION".Connection.ConnectionHdl,
                           NodeIDCount := "DB16105_U2_STA3_CAM_CLIENT_CONFIGURATION".MethodLists.U2_STA3_CAM_Calibrations.MethodCount,
                           ObjectNodeIDs := "DB16105_U2_STA3_CAM_CLIENT_CONFIGURATION".MethodLists.U2_STA3_CAM_Calibrations.ObjectNodes,
                           MethodNodeIDs := "DB16105_U2_STA3_CAM_CLIENT_CONFIGURATION".MethodLists.U2_STA3_CAM_Calibrations.MethodNodes,
                           Timeout := "DB16105_U2_STA3_CAM_CLIENT_CONFIGURATION".Connection.ConnectInfo.SessionTimeout,
                           NamespaceIndexCount := "DB16105_U2_STA3_CAM_CLIENT_CONFIGURATION".Namespaces.NamespaceCount,
                           NamespaceIndexes := "DB16105_U2_STA3_CAM_CLIENT_CONFIGURATION".Namespaces.ServerNamespaceIndexes,
                           StatusList := "DB16005_U2_STA3_COAXIAL_CLIENT_INTERFACE".U2_STA3_CAM_Calibrations.MethodStatusList,
                           MethodHdls := "DB16105_U2_STA3_CAM_CLIENT_CONFIGURATION".MethodLists.U2_STA3_CAM_Calibrations.MethodHdls);
END_REGION

REGION Network 29: UNIT 2 STATION 3 COAXIAL CAMERA GET METHOD ANALISIS LIST CALL
   RUNG wire#powerrail
      "DB16244_GET_MD_LIST_U2_STA3_CAM_ANALISIS".OPC_UA_MethodGetHandleList(REQ := wire#w1, ConnectionHdl := "DB16105_U2_STA3_CAM_CLIENT_CONFIGURATION".Connection.ConnectionHdl, NodeIDCount := "DB16105_U2_STA3_CAM_CLIENT_CONFIGURATION".MethodLists.U2_STA3_CAM_Analysis.MethodCount, ObjectNodeIDs := "DB16105_U2_STA3_CAM_CLIENT_CONFIGURATION".MethodLists.U2_STA3_CAM_Analysis.ObjectNodes, MethodNodeIDs := "DB16105_U2_STA3_CAM_CLIENT_CONFIGURATION".MethodLists.U2_STA3_CAM_Analysis.MethodNodes, Timeout := "DB16105_U2_STA3_CAM_CLIENT_CONFIGURATION".Connection.ConnectInfo.SessionTimeout, NamespaceIndexCount := "DB16105_U2_STA3_CAM_CLIENT_CONFIGURATION".Namespaces.NamespaceCount, NamespaceIndexes := "DB16105_U2_STA3_CAM_CLIENT_CONFIGURATION".Namespaces.ServerNamespaceIndexes, StatusList := "DB16005_U2_STA3_COAXIAL_CLIENT_INTERFACE".U2_STA3_CAM_Analysis.MethodStatusList, MethodHdls := "DB16105_U2_STA3_CAM_CLIENT_CONFIGURATION".MethodLists.U2_STA3_CAM_Analysis.MethodHdls, Done =>, Busy =>, Error =>, Status =>)
   END_RUNG
   RUNG wire#powerrail
      Contact( "DB16000_OPC_UA_TRIGGER_ALARM".CLIENT.U2_STA3_COAXIAL.TRIGGERS.GET_METHOD_LIST_ANALISIS )
      P_Trig( "DB16000_OPC_UA_TRIGGER_ALARM".CLIENT.U2_STA3_COAXIAL.TRIGGERS.GET_METHOD_LIST_ANALISIS_P )
   END_RUNG wire#w1
   // the same network as SCL:
   #_w1 := "DB16000_OPC_UA_TRIGGER_ALARM".CLIENT.U2_STA3_COAXIAL.TRIGGERS.GET_METHOD_LIST_ANALISIS AND NOT "DB16000_OPC_UA_TRIGGER_ALARM".CLIENT.U2_STA3_COAXIAL.TRIGGERS.GET_METHOD_LIST_ANALISIS_P;   // rising edge
   "DB16000_OPC_UA_TRIGGER_ALARM".CLIENT.U2_STA3_COAXIAL.TRIGGERS.GET_METHOD_LIST_ANALISIS_P := "DB16000_OPC_UA_TRIGGER_ALARM".CLIENT.U2_STA3_COAXIAL.TRIGGERS.GET_METHOD_LIST_ANALISIS;
   "DB16244_GET_MD_LIST_U2_STA3_CAM_ANALISIS"(REQ := #_w1,   // OPC_UA_MethodGetHandleList
                           ConnectionHdl := "DB16105_U2_STA3_CAM_CLIENT_CONFIGURATION".Connection.ConnectionHdl,
                           NodeIDCount := "DB16105_U2_STA3_CAM_CLIENT_CONFIGURATION".MethodLists.U2_STA3_CAM_Analysis.MethodCount,
                           ObjectNodeIDs := "DB16105_U2_STA3_CAM_CLIENT_CONFIGURATION".MethodLists.U2_STA3_CAM_Analysis.ObjectNodes,
                           MethodNodeIDs := "DB16105_U2_STA3_CAM_CLIENT_CONFIGURATION".MethodLists.U2_STA3_CAM_Analysis.MethodNodes,
                           Timeout := "DB16105_U2_STA3_CAM_CLIENT_CONFIGURATION".Connection.ConnectInfo.SessionTimeout,
                           NamespaceIndexCount := "DB16105_U2_STA3_CAM_CLIENT_CONFIGURATION".Namespaces.NamespaceCount,
                           NamespaceIndexes := "DB16105_U2_STA3_CAM_CLIENT_CONFIGURATION".Namespaces.ServerNamespaceIndexes,
                           StatusList := "DB16005_U2_STA3_COAXIAL_CLIENT_INTERFACE".U2_STA3_CAM_Analysis.MethodStatusList,
                           MethodHdls := "DB16105_U2_STA3_CAM_CLIENT_CONFIGURATION".MethodLists.U2_STA3_CAM_Analysis.MethodHdls);
END_REGION

REGION Network 30: UNIT 2 STATION 3 COAXIAL CAMERA START LASER CALIBRATION TRIGGER CALL
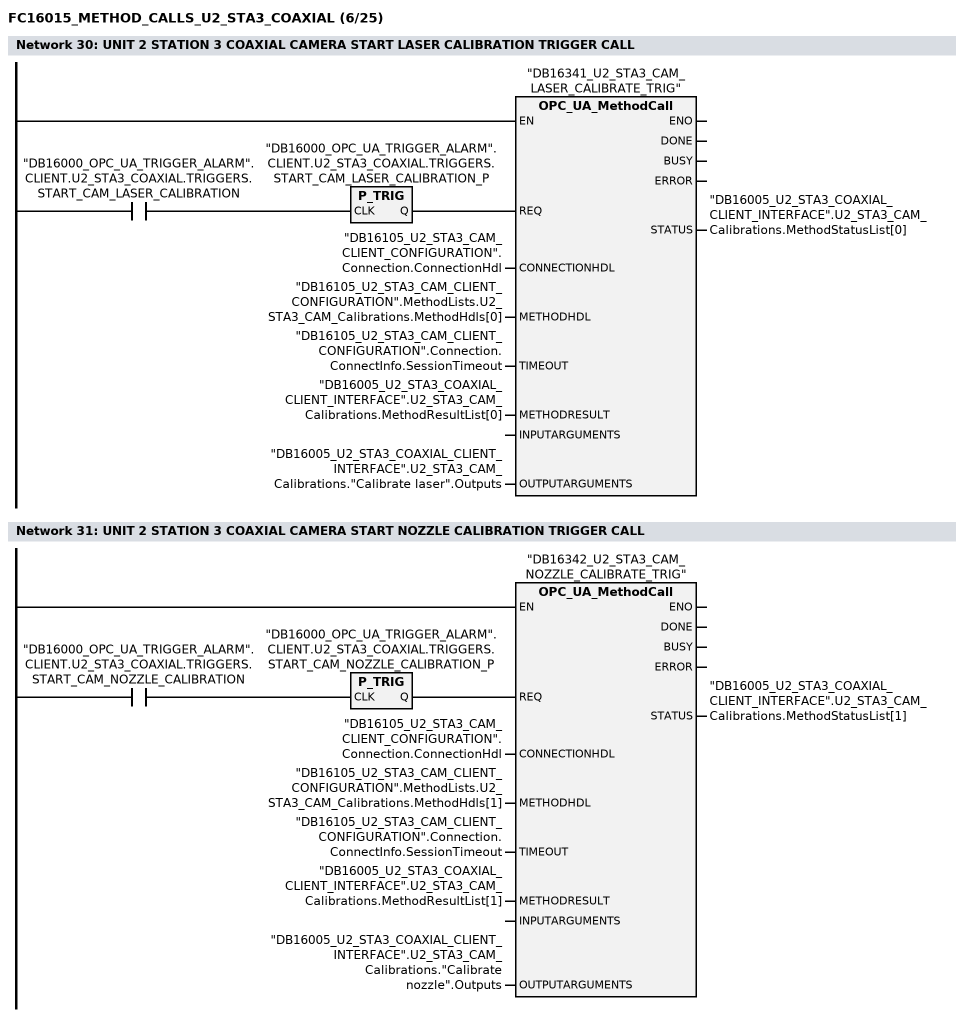
   RUNG wire#powerrail
      "DB16341_U2_STA3_CAM_LASER_CALIBRATE_TRIG".OPC_UA_MethodCall(REQ := wire#w1, ConnectionHdl := "DB16105_U2_STA3_CAM_CLIENT_CONFIGURATION".Connection.ConnectionHdl, MethodHdl := "DB16105_U2_STA3_CAM_CLIENT_CONFIGURATION".MethodLists.U2_STA3_CAM_Calibrations.MethodHdls[0], Timeout := "DB16105_U2_STA3_CAM_CLIENT_CONFIGURATION".Connection.ConnectInfo.SessionTimeout, MethodResult := "DB16005_U2_STA3_COAXIAL_CLIENT_INTERFACE".U2_STA3_CAM_Calibrations.MethodResultList[0], InputArguments :=, OutputArguments := "DB16005_U2_STA3_COAXIAL_CLIENT_INTERFACE".U2_STA3_CAM_Calibrations."Calibrate laser".Outputs, Done =>, Busy =>, Error =>, Status => "DB16005_U2_STA3_COAXIAL_CLIENT_INTERFACE".U2_STA3_CAM_Calibrations.MethodStatusList[0])
   END_RUNG
   RUNG wire#powerrail
      Contact( "DB16000_OPC_UA_TRIGGER_ALARM".CLIENT.U2_STA3_COAXIAL.TRIGGERS.START_CAM_LASER_CALIBRATION )
      P_Trig( "DB16000_OPC_UA_TRIGGER_ALARM".CLIENT.U2_STA3_COAXIAL.TRIGGERS.START_CAM_LASER_CALIBRATION_P )
   END_RUNG wire#w1
   // the same network as SCL:
   #_w1 := "DB16000_OPC_UA_TRIGGER_ALARM".CLIENT.U2_STA3_COAXIAL.TRIGGERS.START_CAM_LASER_CALIBRATION AND NOT "DB16000_OPC_UA_TRIGGER_ALARM".CLIENT.U2_STA3_COAXIAL.TRIGGERS.START_CAM_LASER_CALIBRATION_P;   // rising edge
   "DB16000_OPC_UA_TRIGGER_ALARM".CLIENT.U2_STA3_COAXIAL.TRIGGERS.START_CAM_LASER_CALIBRATION_P := "DB16000_OPC_UA_TRIGGER_ALARM".CLIENT.U2_STA3_COAXIAL.TRIGGERS.START_CAM_LASER_CALIBRATION;
   "DB16341_U2_STA3_CAM_LASER_CALIBRATE_TRIG"(REQ := #_w1,   // OPC_UA_MethodCall
                           ConnectionHdl := "DB16105_U2_STA3_CAM_CLIENT_CONFIGURATION".Connection.ConnectionHdl,
                           MethodHdl := "DB16105_U2_STA3_CAM_CLIENT_CONFIGURATION".MethodLists.U2_STA3_CAM_Calibrations.MethodHdls[0],
                           Timeout := "DB16105_U2_STA3_CAM_CLIENT_CONFIGURATION".Connection.ConnectInfo.SessionTimeout,
                           MethodResult := "DB16005_U2_STA3_COAXIAL_CLIENT_INTERFACE".U2_STA3_CAM_Calibrations.MethodResultList[0],
                           OutputArguments := "DB16005_U2_STA3_COAXIAL_CLIENT_INTERFACE".U2_STA3_CAM_Calibrations."Calibrate laser".Outputs,
                           Status => "DB16005_U2_STA3_COAXIAL_CLIENT_INTERFACE".U2_STA3_CAM_Calibrations.MethodStatusList[0]);
END_REGION

REGION Network 31: UNIT 2 STATION 3 COAXIAL CAMERA START NOZZLE CALIBRATION TRIGGER CALL
   RUNG wire#powerrail
      "DB16342_U2_STA3_CAM_NOZZLE_CALIBRATE_TRIG".OPC_UA_MethodCall(REQ := wire#w1, ConnectionHdl := "DB16105_U2_STA3_CAM_CLIENT_CONFIGURATION".Connection.ConnectionHdl, MethodHdl := "DB16105_U2_STA3_CAM_CLIENT_CONFIGURATION".MethodLists.U2_STA3_CAM_Calibrations.MethodHdls[1], Timeout := "DB16105_U2_STA3_CAM_CLIENT_CONFIGURATION".Connection.ConnectInfo.SessionTimeout, MethodResult := "DB16005_U2_STA3_COAXIAL_CLIENT_INTERFACE".U2_STA3_CAM_Calibrations.MethodResultList[1], InputArguments :=, OutputArguments := "DB16005_U2_STA3_COAXIAL_CLIENT_INTERFACE".U2_STA3_CAM_Calibrations."Calibrate nozzle".Outputs, Done =>, Busy =>, Error =>, Status => "DB16005_U2_STA3_COAXIAL_CLIENT_INTERFACE".U2_STA3_CAM_Calibrations.MethodStatusList[1])
   END_RUNG
   RUNG wire#powerrail
      Contact( "DB16000_OPC_UA_TRIGGER_ALARM".CLIENT.U2_STA3_COAXIAL.TRIGGERS.START_CAM_NOZZLE_CALIBRATION )
      P_Trig( "DB16000_OPC_UA_TRIGGER_ALARM".CLIENT.U2_STA3_COAXIAL.TRIGGERS.START_CAM_NOZZLE_CALIBRATION_P )
   END_RUNG wire#w1
   // the same network as SCL:
   #_w1 := "DB16000_OPC_UA_TRIGGER_ALARM".CLIENT.U2_STA3_COAXIAL.TRIGGERS.START_CAM_NOZZLE_CALIBRATION AND NOT "DB16000_OPC_UA_TRIGGER_ALARM".CLIENT.U2_STA3_COAXIAL.TRIGGERS.START_CAM_NOZZLE_CALIBRATION_P;   // rising edge
   "DB16000_OPC_UA_TRIGGER_ALARM".CLIENT.U2_STA3_COAXIAL.TRIGGERS.START_CAM_NOZZLE_CALIBRATION_P := "DB16000_OPC_UA_TRIGGER_ALARM".CLIENT.U2_STA3_COAXIAL.TRIGGERS.START_CAM_NOZZLE_CALIBRATION;
   "DB16342_U2_STA3_CAM_NOZZLE_CALIBRATE_TRIG"(REQ := #_w1,   // OPC_UA_MethodCall
                           ConnectionHdl := "DB16105_U2_STA3_CAM_CLIENT_CONFIGURATION".Connection.ConnectionHdl,
                           MethodHdl := "DB16105_U2_STA3_CAM_CLIENT_CONFIGURATION".MethodLists.U2_STA3_CAM_Calibrations.MethodHdls[1],
                           Timeout := "DB16105_U2_STA3_CAM_CLIENT_CONFIGURATION".Connection.ConnectInfo.SessionTimeout,
                           MethodResult := "DB16005_U2_STA3_COAXIAL_CLIENT_INTERFACE".U2_STA3_CAM_Calibrations.MethodResultList[1],
                           OutputArguments := "DB16005_U2_STA3_COAXIAL_CLIENT_INTERFACE".U2_STA3_CAM_Calibrations."Calibrate nozzle".Outputs,
                           Status => "DB16005_U2_STA3_COAXIAL_CLIENT_INTERFACE".U2_STA3_CAM_Calibrations.MethodStatusList[1]);
END_REGION

REGION Network 32: UNIT 2 STATION 3 COAXIAL CAMERA START JET CALIBRATION TRIGGER CALL
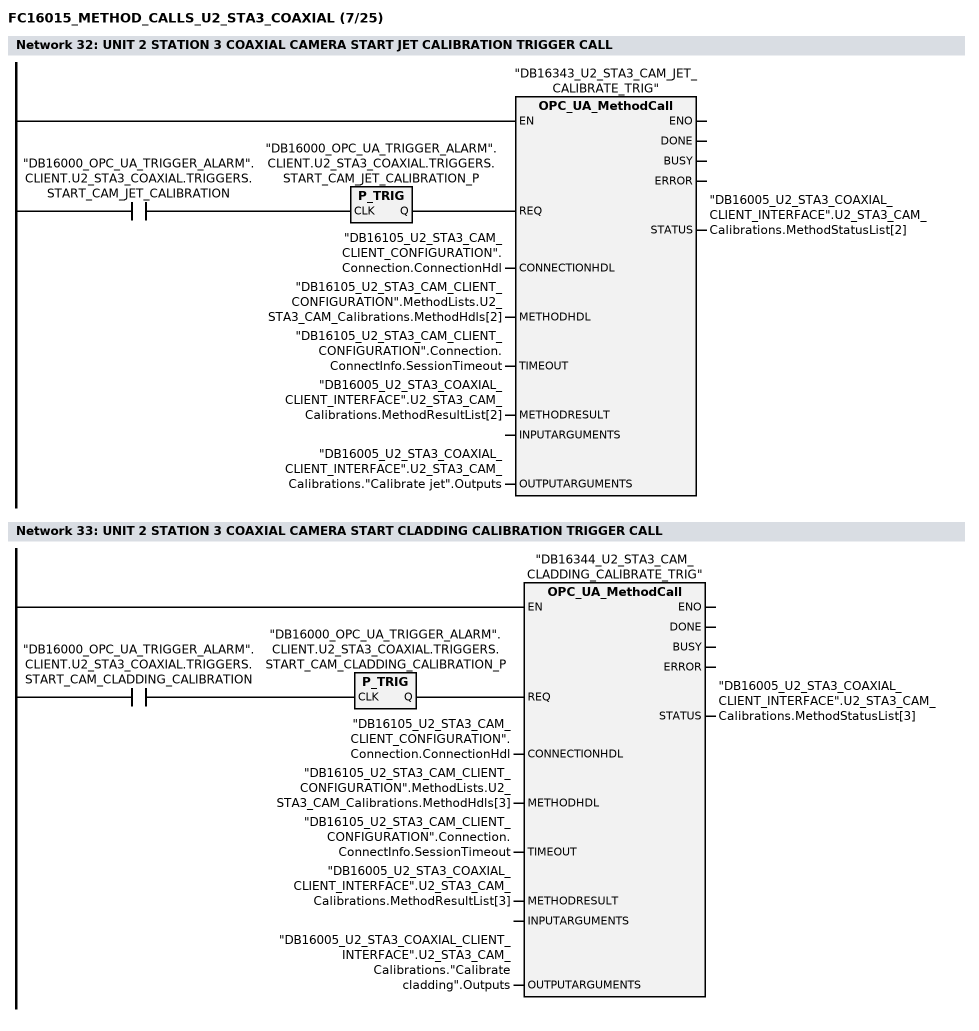
   RUNG wire#powerrail
      "DB16343_U2_STA3_CAM_JET_CALIBRATE_TRIG".OPC_UA_MethodCall(REQ := wire#w1, ConnectionHdl := "DB16105_U2_STA3_CAM_CLIENT_CONFIGURATION".Connection.ConnectionHdl, MethodHdl := "DB16105_U2_STA3_CAM_CLIENT_CONFIGURATION".MethodLists.U2_STA3_CAM_Calibrations.MethodHdls[2], Timeout := "DB16105_U2_STA3_CAM_CLIENT_CONFIGURATION".Connection.ConnectInfo.SessionTimeout, MethodResult := "DB16005_U2_STA3_COAXIAL_CLIENT_INTERFACE".U2_STA3_CAM_Calibrations.MethodResultList[2], InputArguments :=, OutputArguments := "DB16005_U2_STA3_COAXIAL_CLIENT_INTERFACE".U2_STA3_CAM_Calibrations."Calibrate jet".Outputs, Done =>, Busy =>, Error =>, Status => "DB16005_U2_STA3_COAXIAL_CLIENT_INTERFACE".U2_STA3_CAM_Calibrations.MethodStatusList[2])
   END_RUNG
   RUNG wire#powerrail
      Contact( "DB16000_OPC_UA_TRIGGER_ALARM".CLIENT.U2_STA3_COAXIAL.TRIGGERS.START_CAM_JET_CALIBRATION )
      P_Trig( "DB16000_OPC_UA_TRIGGER_ALARM".CLIENT.U2_STA3_COAXIAL.TRIGGERS.START_CAM_JET_CALIBRATION_P )
   END_RUNG wire#w1
   // the same network as SCL:
   #_w1 := "DB16000_OPC_UA_TRIGGER_ALARM".CLIENT.U2_STA3_COAXIAL.TRIGGERS.START_CAM_JET_CALIBRATION AND NOT "DB16000_OPC_UA_TRIGGER_ALARM".CLIENT.U2_STA3_COAXIAL.TRIGGERS.START_CAM_JET_CALIBRATION_P;   // rising edge
   "DB16000_OPC_UA_TRIGGER_ALARM".CLIENT.U2_STA3_COAXIAL.TRIGGERS.START_CAM_JET_CALIBRATION_P := "DB16000_OPC_UA_TRIGGER_ALARM".CLIENT.U2_STA3_COAXIAL.TRIGGERS.START_CAM_JET_CALIBRATION;
   "DB16343_U2_STA3_CAM_JET_CALIBRATE_TRIG"(REQ := #_w1,   // OPC_UA_MethodCall
                           ConnectionHdl := "DB16105_U2_STA3_CAM_CLIENT_CONFIGURATION".Connection.ConnectionHdl,
                           MethodHdl := "DB16105_U2_STA3_CAM_CLIENT_CONFIGURATION".MethodLists.U2_STA3_CAM_Calibrations.MethodHdls[2],
                           Timeout := "DB16105_U2_STA3_CAM_CLIENT_CONFIGURATION".Connection.ConnectInfo.SessionTimeout,
                           MethodResult := "DB16005_U2_STA3_COAXIAL_CLIENT_INTERFACE".U2_STA3_CAM_Calibrations.MethodResultList[2],
                           OutputArguments := "DB16005_U2_STA3_COAXIAL_CLIENT_INTERFACE".U2_STA3_CAM_Calibrations."Calibrate jet".Outputs,
                           Status => "DB16005_U2_STA3_COAXIAL_CLIENT_INTERFACE".U2_STA3_CAM_Calibrations.MethodStatusList[2]);
END_REGION

REGION Network 33: UNIT 2 STATION 3 COAXIAL CAMERA START CLADDING CALIBRATION TRIGGER CALL
   RUNG wire#powerrail
      "DB16344_U2_STA3_CAM_CLADDING_CALIBRATE_TRIG".OPC_UA_MethodCall(REQ := wire#w1, ConnectionHdl := "DB16105_U2_STA3_CAM_CLIENT_CONFIGURATION".Connection.ConnectionHdl, MethodHdl := "DB16105_U2_STA3_CAM_CLIENT_CONFIGURATION".MethodLists.U2_STA3_CAM_Calibrations.MethodHdls[3], Timeout := "DB16105_U2_STA3_CAM_CLIENT_CONFIGURATION".Connection.ConnectInfo.SessionTimeout, MethodResult := "DB16005_U2_STA3_COAXIAL_CLIENT_INTERFACE".U2_STA3_CAM_Calibrations.MethodResultList[3], InputArguments :=, OutputArguments := "DB16005_U2_STA3_COAXIAL_CLIENT_INTERFACE".U2_STA3_CAM_Calibrations."Calibrate cladding".Outputs, Done =>, Busy =>, Error =>, Status => "DB16005_U2_STA3_COAXIAL_CLIENT_INTERFACE".U2_STA3_CAM_Calibrations.MethodStatusList[3])
   END_RUNG
   RUNG wire#powerrail
      Contact( "DB16000_OPC_UA_TRIGGER_ALARM".CLIENT.U2_STA3_COAXIAL.TRIGGERS.START_CAM_CLADDING_CALIBRATION )
      P_Trig( "DB16000_OPC_UA_TRIGGER_ALARM".CLIENT.U2_STA3_COAXIAL.TRIGGERS.START_CAM_CLADDING_CALIBRATION_P )
   END_RUNG wire#w1
   // the same network as SCL:
   #_w1 := "DB16000_OPC_UA_TRIGGER_ALARM".CLIENT.U2_STA3_COAXIAL.TRIGGERS.START_CAM_CLADDING_CALIBRATION AND NOT "DB16000_OPC_UA_TRIGGER_ALARM".CLIENT.U2_STA3_COAXIAL.TRIGGERS.START_CAM_CLADDING_CALIBRATION_P;   // rising edge
   "DB16000_OPC_UA_TRIGGER_ALARM".CLIENT.U2_STA3_COAXIAL.TRIGGERS.START_CAM_CLADDING_CALIBRATION_P := "DB16000_OPC_UA_TRIGGER_ALARM".CLIENT.U2_STA3_COAXIAL.TRIGGERS.START_CAM_CLADDING_CALIBRATION;
   "DB16344_U2_STA3_CAM_CLADDING_CALIBRATE_TRIG"(REQ := #_w1,   // OPC_UA_MethodCall
                           ConnectionHdl := "DB16105_U2_STA3_CAM_CLIENT_CONFIGURATION".Connection.ConnectionHdl,
                           MethodHdl := "DB16105_U2_STA3_CAM_CLIENT_CONFIGURATION".MethodLists.U2_STA3_CAM_Calibrations.MethodHdls[3],
                           Timeout := "DB16105_U2_STA3_CAM_CLIENT_CONFIGURATION".Connection.ConnectInfo.SessionTimeout,
                           MethodResult := "DB16005_U2_STA3_COAXIAL_CLIENT_INTERFACE".U2_STA3_CAM_Calibrations.MethodResultList[3],
                           OutputArguments := "DB16005_U2_STA3_COAXIAL_CLIENT_INTERFACE".U2_STA3_CAM_Calibrations."Calibrate cladding".Outputs,
                           Status => "DB16005_U2_STA3_COAXIAL_CLIENT_INTERFACE".U2_STA3_CAM_Calibrations.MethodStatusList[3]);
END_REGION

REGION Network 34: UNIT 2 STATION 3 COAXIAL CAMERA START NOZZLE ANALISIS TRIGGER CALL
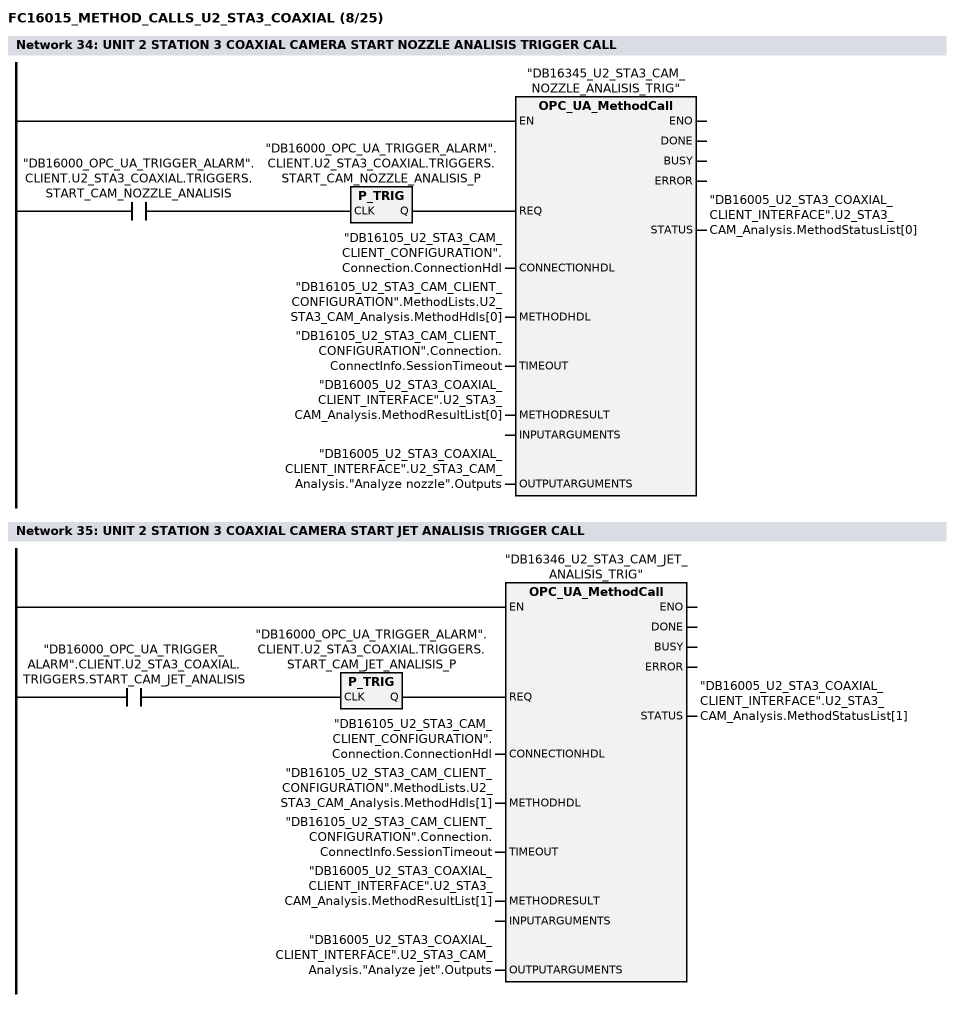
   RUNG wire#powerrail
      "DB16345_U2_STA3_CAM_NOZZLE_ANALISIS_TRIG".OPC_UA_MethodCall(REQ := wire#w1, ConnectionHdl := "DB16105_U2_STA3_CAM_CLIENT_CONFIGURATION".Connection.ConnectionHdl, MethodHdl := "DB16105_U2_STA3_CAM_CLIENT_CONFIGURATION".MethodLists.U2_STA3_CAM_Analysis.MethodHdls[0], Timeout := "DB16105_U2_STA3_CAM_CLIENT_CONFIGURATION".Connection.ConnectInfo.SessionTimeout, MethodResult := "DB16005_U2_STA3_COAXIAL_CLIENT_INTERFACE".U2_STA3_CAM_Analysis.MethodResultList[0], InputArguments :=, OutputArguments := "DB16005_U2_STA3_COAXIAL_CLIENT_INTERFACE".U2_STA3_CAM_Analysis."Analyze nozzle".Outputs, Done =>, Busy =>, Error =>, Status => "DB16005_U2_STA3_COAXIAL_CLIENT_INTERFACE".U2_STA3_CAM_Analysis.MethodStatusList[0])
   END_RUNG
   RUNG wire#powerrail
      Contact( "DB16000_OPC_UA_TRIGGER_ALARM".CLIENT.U2_STA3_COAXIAL.TRIGGERS.START_CAM_NOZZLE_ANALISIS )
      P_Trig( "DB16000_OPC_UA_TRIGGER_ALARM".CLIENT.U2_STA3_COAXIAL.TRIGGERS.START_CAM_NOZZLE_ANALISIS_P )
   END_RUNG wire#w1
   // the same network as SCL:
   #_w1 := "DB16000_OPC_UA_TRIGGER_ALARM".CLIENT.U2_STA3_COAXIAL.TRIGGERS.START_CAM_NOZZLE_ANALISIS AND NOT "DB16000_OPC_UA_TRIGGER_ALARM".CLIENT.U2_STA3_COAXIAL.TRIGGERS.START_CAM_NOZZLE_ANALISIS_P;   // rising edge
   "DB16000_OPC_UA_TRIGGER_ALARM".CLIENT.U2_STA3_COAXIAL.TRIGGERS.START_CAM_NOZZLE_ANALISIS_P := "DB16000_OPC_UA_TRIGGER_ALARM".CLIENT.U2_STA3_COAXIAL.TRIGGERS.START_CAM_NOZZLE_ANALISIS;
   "DB16345_U2_STA3_CAM_NOZZLE_ANALISIS_TRIG"(REQ := #_w1,   // OPC_UA_MethodCall
                           ConnectionHdl := "DB16105_U2_STA3_CAM_CLIENT_CONFIGURATION".Connection.ConnectionHdl,
                           MethodHdl := "DB16105_U2_STA3_CAM_CLIENT_CONFIGURATION".MethodLists.U2_STA3_CAM_Analysis.MethodHdls[0],
                           Timeout := "DB16105_U2_STA3_CAM_CLIENT_CONFIGURATION".Connection.ConnectInfo.SessionTimeout,
                           MethodResult := "DB16005_U2_STA3_COAXIAL_CLIENT_INTERFACE".U2_STA3_CAM_Analysis.MethodResultList[0],
                           OutputArguments := "DB16005_U2_STA3_COAXIAL_CLIENT_INTERFACE".U2_STA3_CAM_Analysis."Analyze nozzle".Outputs,
                           Status => "DB16005_U2_STA3_COAXIAL_CLIENT_INTERFACE".U2_STA3_CAM_Analysis.MethodStatusList[0]);
END_REGION

REGION Network 35: UNIT 2 STATION 3 COAXIAL CAMERA START JET ANALISIS TRIGGER CALL
   RUNG wire#powerrail
      "DB16346_U2_STA3_CAM_JET_ANALISIS_TRIG".OPC_UA_MethodCall(REQ := wire#w1, ConnectionHdl := "DB16105_U2_STA3_CAM_CLIENT_CONFIGURATION".Connection.ConnectionHdl, MethodHdl := "DB16105_U2_STA3_CAM_CLIENT_CONFIGURATION".MethodLists.U2_STA3_CAM_Analysis.MethodHdls[1], Timeout := "DB16105_U2_STA3_CAM_CLIENT_CONFIGURATION".Connection.ConnectInfo.SessionTimeout, MethodResult := "DB16005_U2_STA3_COAXIAL_CLIENT_INTERFACE".U2_STA3_CAM_Analysis.MethodResultList[1], InputArguments :=, OutputArguments := "DB16005_U2_STA3_COAXIAL_CLIENT_INTERFACE".U2_STA3_CAM_Analysis."Analyze jet".Outputs, Done =>, Busy =>, Error =>, Status => "DB16005_U2_STA3_COAXIAL_CLIENT_INTERFACE".U2_STA3_CAM_Analysis.MethodStatusList[1])
   END_RUNG
   RUNG wire#powerrail
      Contact( "DB16000_OPC_UA_TRIGGER_ALARM".CLIENT.U2_STA3_COAXIAL.TRIGGERS.START_CAM_JET_ANALISIS )
      P_Trig( "DB16000_OPC_UA_TRIGGER_ALARM".CLIENT.U2_STA3_COAXIAL.TRIGGERS.START_CAM_JET_ANALISIS_P )
   END_RUNG wire#w1
   // the same network as SCL:
   #_w1 := "DB16000_OPC_UA_TRIGGER_ALARM".CLIENT.U2_STA3_COAXIAL.TRIGGERS.START_CAM_JET_ANALISIS AND NOT "DB16000_OPC_UA_TRIGGER_ALARM".CLIENT.U2_STA3_COAXIAL.TRIGGERS.START_CAM_JET_ANALISIS_P;   // rising edge
   "DB16000_OPC_UA_TRIGGER_ALARM".CLIENT.U2_STA3_COAXIAL.TRIGGERS.START_CAM_JET_ANALISIS_P := "DB16000_OPC_UA_TRIGGER_ALARM".CLIENT.U2_STA3_COAXIAL.TRIGGERS.START_CAM_JET_ANALISIS;
   "DB16346_U2_STA3_CAM_JET_ANALISIS_TRIG"(REQ := #_w1,   // OPC_UA_MethodCall
                           ConnectionHdl := "DB16105_U2_STA3_CAM_CLIENT_CONFIGURATION".Connection.ConnectionHdl,
                           MethodHdl := "DB16105_U2_STA3_CAM_CLIENT_CONFIGURATION".MethodLists.U2_STA3_CAM_Analysis.MethodHdls[1],
                           Timeout := "DB16105_U2_STA3_CAM_CLIENT_CONFIGURATION".Connection.ConnectInfo.SessionTimeout,
                           MethodResult := "DB16005_U2_STA3_COAXIAL_CLIENT_INTERFACE".U2_STA3_CAM_Analysis.MethodResultList[1],
                           OutputArguments := "DB16005_U2_STA3_COAXIAL_CLIENT_INTERFACE".U2_STA3_CAM_Analysis."Analyze jet".Outputs,
                           Status => "DB16005_U2_STA3_COAXIAL_CLIENT_INTERFACE".U2_STA3_CAM_Analysis.MethodStatusList[1]);
END_REGION

REGION Network 36: UNIT 2 STATION 3 COAXIAL CAMERA START CLADDING ANALISIS TRIGGER CALL
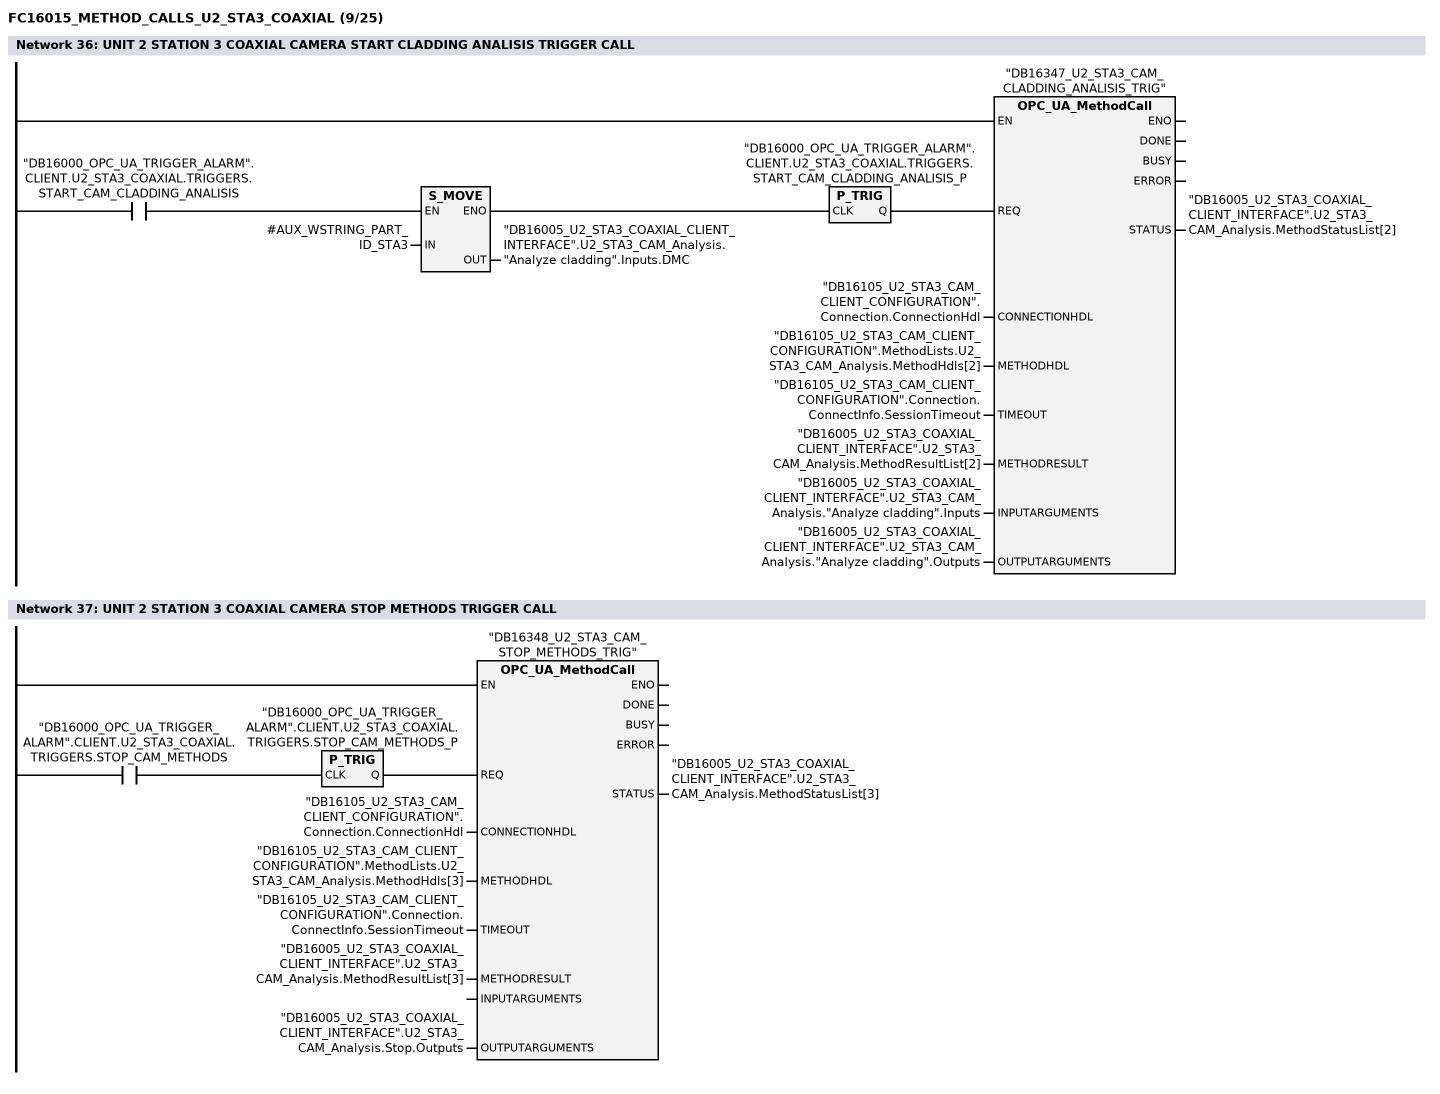
   RUNG wire#powerrail
      "DB16347_U2_STA3_CAM_CLADDING_ANALISIS_TRIG".OPC_UA_MethodCall(REQ := wire#w1, ConnectionHdl := "DB16105_U2_STA3_CAM_CLIENT_CONFIGURATION".Connection.ConnectionHdl, MethodHdl := "DB16105_U2_STA3_CAM_CLIENT_CONFIGURATION".MethodLists.U2_STA3_CAM_Analysis.MethodHdls[2], Timeout := "DB16105_U2_STA3_CAM_CLIENT_CONFIGURATION".Connection.ConnectInfo.SessionTimeout, MethodResult := "DB16005_U2_STA3_COAXIAL_CLIENT_INTERFACE".U2_STA3_CAM_Analysis.MethodResultList[2], InputArguments := "DB16005_U2_STA3_COAXIAL_CLIENT_INTERFACE".U2_STA3_CAM_Analysis."Analyze cladding".Inputs, OutputArguments := "DB16005_U2_STA3_COAXIAL_CLIENT_INTERFACE".U2_STA3_CAM_Analysis."Analyze cladding".Outputs, Done =>, Busy =>, Error =>, Status => "DB16005_U2_STA3_COAXIAL_CLIENT_INTERFACE".U2_STA3_CAM_Analysis.MethodStatusList[2])
   END_RUNG
   RUNG wire#powerrail
      Contact( "DB16000_OPC_UA_TRIGGER_ALARM".CLIENT.U2_STA3_COAXIAL.TRIGGERS.START_CAM_CLADDING_ANALISIS )
      S_Move(in := #AUX_WSTRING_PART_ID_STA3, out => "DB16005_U2_STA3_COAXIAL_CLIENT_INTERFACE".U2_STA3_CAM_Analysis."Analyze cladding".Inputs.DMC)
      P_Trig( "DB16000_OPC_UA_TRIGGER_ALARM".CLIENT.U2_STA3_COAXIAL.TRIGGERS.START_CAM_CLADDING_ANALISIS_P )
   END_RUNG wire#w1
   // the same network as SCL:
   IF "DB16000_OPC_UA_TRIGGER_ALARM".CLIENT.U2_STA3_COAXIAL.TRIGGERS.START_CAM_CLADDING_ANALISIS THEN
       "DB16005_U2_STA3_COAXIAL_CLIENT_INTERFACE".U2_STA3_CAM_Analysis."Analyze cladding".Inputs.DMC := #AUX_WSTRING_PART_ID_STA3;
   END_IF;
   #_w1 := "DB16000_OPC_UA_TRIGGER_ALARM".CLIENT.U2_STA3_COAXIAL.TRIGGERS.START_CAM_CLADDING_ANALISIS AND NOT "DB16000_OPC_UA_TRIGGER_ALARM".CLIENT.U2_STA3_COAXIAL.TRIGGERS.START_CAM_CLADDING_ANALISIS_P;   // rising edge
   "DB16000_OPC_UA_TRIGGER_ALARM".CLIENT.U2_STA3_COAXIAL.TRIGGERS.START_CAM_CLADDING_ANALISIS_P := "DB16000_OPC_UA_TRIGGER_ALARM".CLIENT.U2_STA3_COAXIAL.TRIGGERS.START_CAM_CLADDING_ANALISIS;
   "DB16347_U2_STA3_CAM_CLADDING_ANALISIS_TRIG"(REQ := #_w1,   // OPC_UA_MethodCall
                           ConnectionHdl := "DB16105_U2_STA3_CAM_CLIENT_CONFIGURATION".Connection.ConnectionHdl,
                           MethodHdl := "DB16105_U2_STA3_CAM_CLIENT_CONFIGURATION".MethodLists.U2_STA3_CAM_Analysis.MethodHdls[2],
                           Timeout := "DB16105_U2_STA3_CAM_CLIENT_CONFIGURATION".Connection.ConnectInfo.SessionTimeout,
                           MethodResult := "DB16005_U2_STA3_COAXIAL_CLIENT_INTERFACE".U2_STA3_CAM_Analysis.MethodResultList[2],
                           InputArguments := "DB16005_U2_STA3_COAXIAL_CLIENT_INTERFACE".U2_STA3_CAM_Analysis."Analyze cladding".Inputs,
                           OutputArguments := "DB16005_U2_STA3_COAXIAL_CLIENT_INTERFACE".U2_STA3_CAM_Analysis."Analyze cladding".Outputs,
                           Status => "DB16005_U2_STA3_COAXIAL_CLIENT_INTERFACE".U2_STA3_CAM_Analysis.MethodStatusList[2]);
END_REGION

REGION Network 37: UNIT 2 STATION 3 COAXIAL CAMERA STOP METHODS TRIGGER CALL
   RUNG wire#powerrail
      "DB16348_U2_STA3_CAM_STOP_METHODS_TRIG".OPC_UA_MethodCall(REQ := wire#w1, ConnectionHdl := "DB16105_U2_STA3_CAM_CLIENT_CONFIGURATION".Connection.ConnectionHdl, MethodHdl := "DB16105_U2_STA3_CAM_CLIENT_CONFIGURATION".MethodLists.U2_STA3_CAM_Analysis.MethodHdls[3], Timeout := "DB16105_U2_STA3_CAM_CLIENT_CONFIGURATION".Connection.ConnectInfo.SessionTimeout, MethodResult := "DB16005_U2_STA3_COAXIAL_CLIENT_INTERFACE".U2_STA3_CAM_Analysis.MethodResultList[3], InputArguments :=, OutputArguments := "DB16005_U2_STA3_COAXIAL_CLIENT_INTERFACE".U2_STA3_CAM_Analysis.Stop.Outputs, Done =>, Busy =>, Error =>, Status => "DB16005_U2_STA3_COAXIAL_CLIENT_INTERFACE".U2_STA3_CAM_Analysis.MethodStatusList[3])
   END_RUNG
   RUNG wire#powerrail
      Contact( "DB16000_OPC_UA_TRIGGER_ALARM".CLIENT.U2_STA3_COAXIAL.TRIGGERS.STOP_CAM_METHODS )
      P_Trig( "DB16000_OPC_UA_TRIGGER_ALARM".CLIENT.U2_STA3_COAXIAL.TRIGGERS.STOP_CAM_METHODS_P )
   END_RUNG wire#w1
   // the same network as SCL:
   #_w1 := "DB16000_OPC_UA_TRIGGER_ALARM".CLIENT.U2_STA3_COAXIAL.TRIGGERS.STOP_CAM_METHODS AND NOT "DB16000_OPC_UA_TRIGGER_ALARM".CLIENT.U2_STA3_COAXIAL.TRIGGERS.STOP_CAM_METHODS_P;   // rising edge
   "DB16000_OPC_UA_TRIGGER_ALARM".CLIENT.U2_STA3_COAXIAL.TRIGGERS.STOP_CAM_METHODS_P := "DB16000_OPC_UA_TRIGGER_ALARM".CLIENT.U2_STA3_COAXIAL.TRIGGERS.STOP_CAM_METHODS;
   "DB16348_U2_STA3_CAM_STOP_METHODS_TRIG"(REQ := #_w1,   // OPC_UA_MethodCall
                           ConnectionHdl := "DB16105_U2_STA3_CAM_CLIENT_CONFIGURATION".Connection.ConnectionHdl,
                           MethodHdl := "DB16105_U2_STA3_CAM_CLIENT_CONFIGURATION".MethodLists.U2_STA3_CAM_Analysis.MethodHdls[3],
                           Timeout := "DB16105_U2_STA3_CAM_CLIENT_CONFIGURATION".Connection.ConnectInfo.SessionTimeout,
                           MethodResult := "DB16005_U2_STA3_COAXIAL_CLIENT_INTERFACE".U2_STA3_CAM_Analysis.MethodResultList[3],
                           OutputArguments := "DB16005_U2_STA3_COAXIAL_CLIENT_INTERFACE".U2_STA3_CAM_Analysis.Stop.Outputs,
                           Status => "DB16005_U2_STA3_COAXIAL_CLIENT_INTERFACE".U2_STA3_CAM_Analysis.MethodStatusList[3]);
END_REGION

REGION Network 38: UNIT 2 STATION 3 COAXIAL CAMERA RESET PC TRIGGER CALL
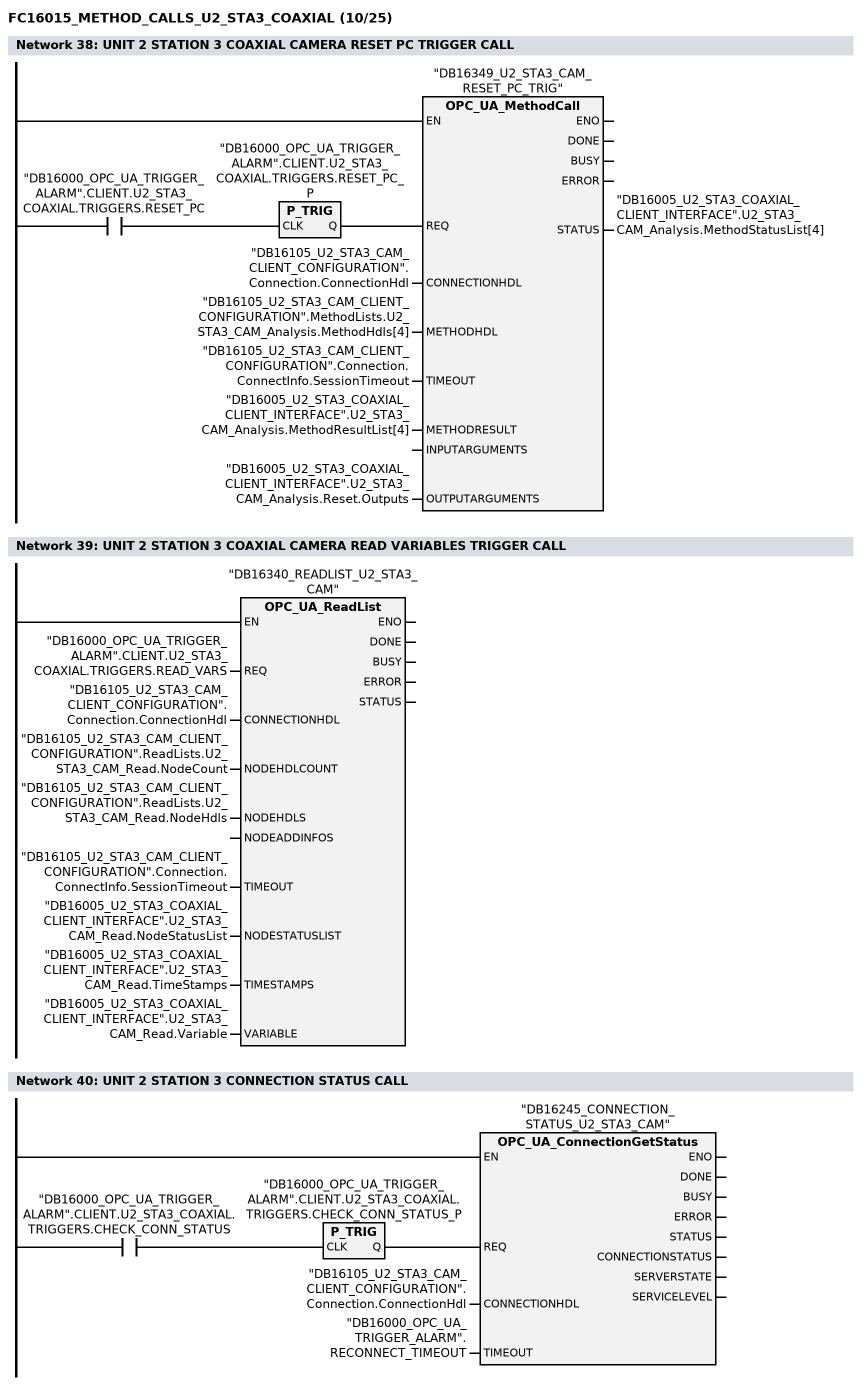
   RUNG wire#powerrail
      "DB16349_U2_STA3_CAM_RESET_PC_TRIG".OPC_UA_MethodCall(REQ := wire#w1, ConnectionHdl := "DB16105_U2_STA3_CAM_CLIENT_CONFIGURATION".Connection.ConnectionHdl, MethodHdl := "DB16105_U2_STA3_CAM_CLIENT_CONFIGURATION".MethodLists.U2_STA3_CAM_Analysis.MethodHdls[4], Timeout := "DB16105_U2_STA3_CAM_CLIENT_CONFIGURATION".Connection.ConnectInfo.SessionTimeout, MethodResult := "DB16005_U2_STA3_COAXIAL_CLIENT_INTERFACE".U2_STA3_CAM_Analysis.MethodResultList[4], InputArguments :=, OutputArguments := "DB16005_U2_STA3_COAXIAL_CLIENT_INTERFACE".U2_STA3_CAM_Analysis.Reset.Outputs, Done =>, Busy =>, Error =>, Status => "DB16005_U2_STA3_COAXIAL_CLIENT_INTERFACE".U2_STA3_CAM_Analysis.MethodStatusList[4])
   END_RUNG
   RUNG wire#powerrail
      Contact( "DB16000_OPC_UA_TRIGGER_ALARM".CLIENT.U2_STA3_COAXIAL.TRIGGERS.RESET_PC )
      P_Trig( "DB16000_OPC_UA_TRIGGER_ALARM".CLIENT.U2_STA3_COAXIAL.TRIGGERS.RESET_PC_P )
   END_RUNG wire#w1
   // the same network as SCL:
   #_w1 := "DB16000_OPC_UA_TRIGGER_ALARM".CLIENT.U2_STA3_COAXIAL.TRIGGERS.RESET_PC AND NOT "DB16000_OPC_UA_TRIGGER_ALARM".CLIENT.U2_STA3_COAXIAL.TRIGGERS.RESET_PC_P;   // rising edge
   "DB16000_OPC_UA_TRIGGER_ALARM".CLIENT.U2_STA3_COAXIAL.TRIGGERS.RESET_PC_P := "DB16000_OPC_UA_TRIGGER_ALARM".CLIENT.U2_STA3_COAXIAL.TRIGGERS.RESET_PC;
   "DB16349_U2_STA3_CAM_RESET_PC_TRIG"(REQ := #_w1,   // OPC_UA_MethodCall
                           ConnectionHdl := "DB16105_U2_STA3_CAM_CLIENT_CONFIGURATION".Connection.ConnectionHdl,
                           MethodHdl := "DB16105_U2_STA3_CAM_CLIENT_CONFIGURATION".MethodLists.U2_STA3_CAM_Analysis.MethodHdls[4],
                           Timeout := "DB16105_U2_STA3_CAM_CLIENT_CONFIGURATION".Connection.ConnectInfo.SessionTimeout,
                           MethodResult := "DB16005_U2_STA3_COAXIAL_CLIENT_INTERFACE".U2_STA3_CAM_Analysis.MethodResultList[4],
                           OutputArguments := "DB16005_U2_STA3_COAXIAL_CLIENT_INTERFACE".U2_STA3_CAM_Analysis.Reset.Outputs,
                           Status => "DB16005_U2_STA3_COAXIAL_CLIENT_INTERFACE".U2_STA3_CAM_Analysis.MethodStatusList[4]);
END_REGION

REGION Network 39: UNIT 2 STATION 3 COAXIAL CAMERA READ VARIABLES TRIGGER CALL
   RUNG wire#powerrail
      "DB16340_READLIST_U2_STA3_CAM".OPC_UA_ReadList(REQ := "DB16000_OPC_UA_TRIGGER_ALARM".CLIENT.U2_STA3_COAXIAL.TRIGGERS.READ_VARS, ConnectionHdl := "DB16105_U2_STA3_CAM_CLIENT_CONFIGURATION".Connection.ConnectionHdl, NodeHdlCount := "DB16105_U2_STA3_CAM_CLIENT_CONFIGURATION".ReadLists.U2_STA3_CAM_Read.NodeCount, NodeHdls := "DB16105_U2_STA3_CAM_CLIENT_CONFIGURATION".ReadLists.U2_STA3_CAM_Read.NodeHdls, NodeAddInfos :=, Timeout := "DB16105_U2_STA3_CAM_CLIENT_CONFIGURATION".Connection.ConnectInfo.SessionTimeout, NodeStatusList := "DB16005_U2_STA3_COAXIAL_CLIENT_INTERFACE".U2_STA3_CAM_Read.NodeStatusList, TimeStamps := "DB16005_U2_STA3_COAXIAL_CLIENT_INTERFACE".U2_STA3_CAM_Read.TimeStamps, Variable := "DB16005_U2_STA3_COAXIAL_CLIENT_INTERFACE".U2_STA3_CAM_Read.Variable, Done =>, Busy =>, Error =>, Status =>)
   END_RUNG
   // the same network as SCL:
   "DB16340_READLIST_U2_STA3_CAM"(REQ := "DB16000_OPC_UA_TRIGGER_ALARM".CLIENT.U2_STA3_COAXIAL.TRIGGERS.READ_VARS,   // OPC_UA_ReadList
                           ConnectionHdl := "DB16105_U2_STA3_CAM_CLIENT_CONFIGURATION".Connection.ConnectionHdl,
                           NodeHdlCount := "DB16105_U2_STA3_CAM_CLIENT_CONFIGURATION".ReadLists.U2_STA3_CAM_Read.NodeCount,
                           NodeHdls := "DB16105_U2_STA3_CAM_CLIENT_CONFIGURATION".ReadLists.U2_STA3_CAM_Read.NodeHdls,
                           Timeout := "DB16105_U2_STA3_CAM_CLIENT_CONFIGURATION".Connection.ConnectInfo.SessionTimeout,
                           NodeStatusList := "DB16005_U2_STA3_COAXIAL_CLIENT_INTERFACE".U2_STA3_CAM_Read.NodeStatusList,
                           TimeStamps := "DB16005_U2_STA3_COAXIAL_CLIENT_INTERFACE".U2_STA3_CAM_Read.TimeStamps,
                           Variable := "DB16005_U2_STA3_COAXIAL_CLIENT_INTERFACE".U2_STA3_CAM_Read.Variable);
END_REGION

REGION Network 40: UNIT 2 STATION 3 CONNECTION STATUS CALL
   RUNG wire#powerrail
      "DB16245_CONNECTION_STATUS_U2_STA3_CAM".OPC_UA_ConnectionGetStatus(REQ := wire#w1, ConnectionHdl := "DB16105_U2_STA3_CAM_CLIENT_CONFIGURATION".Connection.ConnectionHdl, Timeout := "DB16000_OPC_UA_TRIGGER_ALARM".RECONNECT_TIMEOUT, Done =>, Busy =>, Error =>, Status =>, ConnectionStatus =>, ServerState =>, ServiceLevel =>)
   END_RUNG
   RUNG wire#powerrail
      Contact( "DB16000_OPC_UA_TRIGGER_ALARM".CLIENT.U2_STA3_COAXIAL.TRIGGERS.CHECK_CONN_STATUS )
      P_Trig( "DB16000_OPC_UA_TRIGGER_ALARM".CLIENT.U2_STA3_COAXIAL.TRIGGERS.CHECK_CONN_STATUS_P )
   END_RUNG wire#w1
   // the same network as SCL:
   #_w1 := "DB16000_OPC_UA_TRIGGER_ALARM".CLIENT.U2_STA3_COAXIAL.TRIGGERS.CHECK_CONN_STATUS AND NOT "DB16000_OPC_UA_TRIGGER_ALARM".CLIENT.U2_STA3_COAXIAL.TRIGGERS.CHECK_CONN_STATUS_P;   // rising edge
   "DB16000_OPC_UA_TRIGGER_ALARM".CLIENT.U2_STA3_COAXIAL.TRIGGERS.CHECK_CONN_STATUS_P := "DB16000_OPC_UA_TRIGGER_ALARM".CLIENT.U2_STA3_COAXIAL.TRIGGERS.CHECK_CONN_STATUS;
   "DB16245_CONNECTION_STATUS_U2_STA3_CAM"(REQ := #_w1,   // OPC_UA_ConnectionGetStatus
                           ConnectionHdl := "DB16105_U2_STA3_CAM_CLIENT_CONFIGURATION".Connection.ConnectionHdl,
                           Timeout := "DB16000_OPC_UA_TRIGGER_ALARM".RECONNECT_TIMEOUT);
END_REGION

REGION Network 41: UNIT 2 STATION 3 RELEASE HANDLE LIST CALL
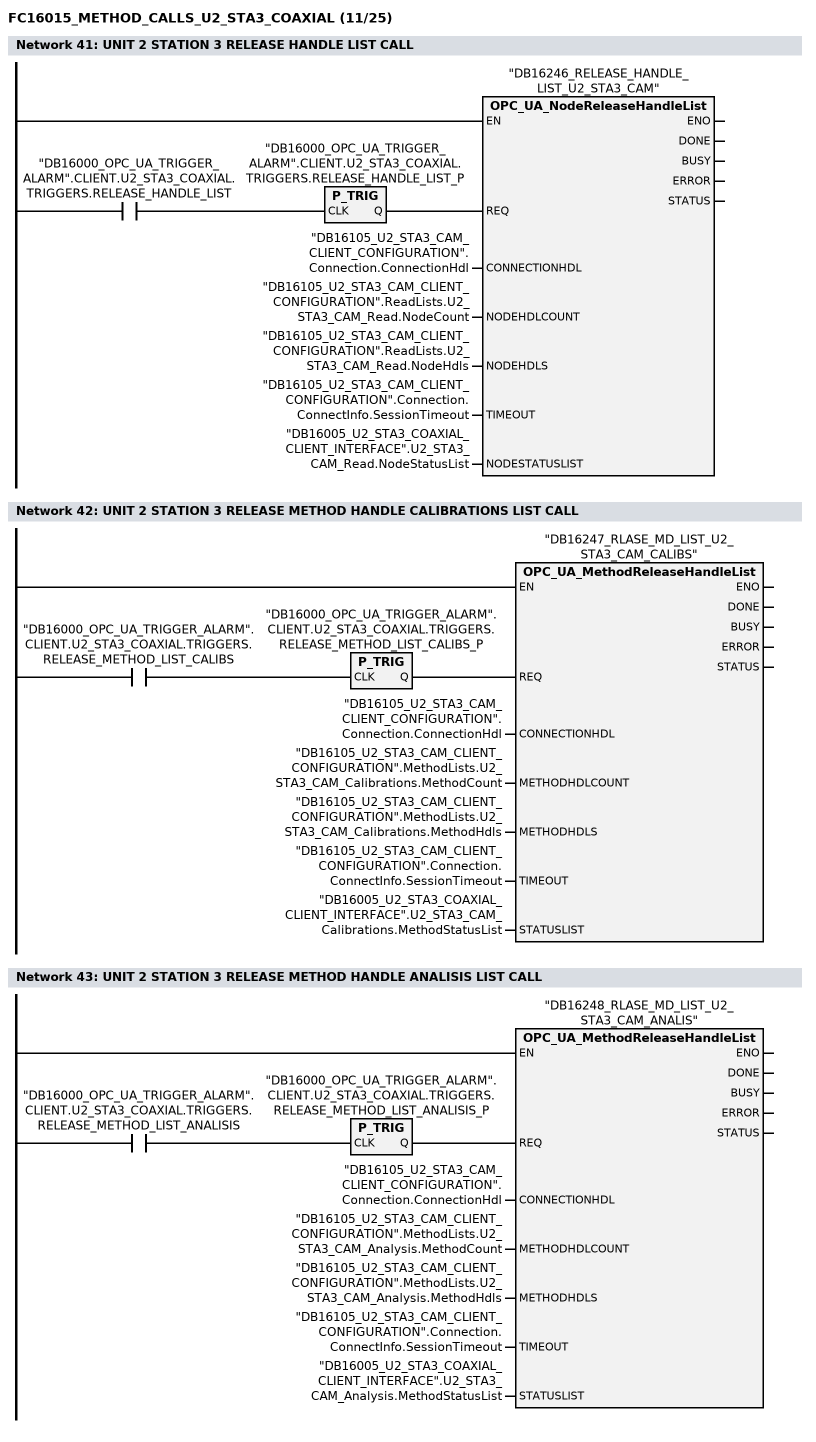
   RUNG wire#powerrail
      "DB16246_RELEASE_HANDLE_LIST_U2_STA3_CAM".OPC_UA_NodeReleaseHandleList(REQ := wire#w1, ConnectionHdl := "DB16105_U2_STA3_CAM_CLIENT_CONFIGURATION".Connection.ConnectionHdl, NodeHdlCount := "DB16105_U2_STA3_CAM_CLIENT_CONFIGURATION".ReadLists.U2_STA3_CAM_Read.NodeCount, NodeHdls := "DB16105_U2_STA3_CAM_CLIENT_CONFIGURATION".ReadLists.U2_STA3_CAM_Read.NodeHdls, Timeout := "DB16105_U2_STA3_CAM_CLIENT_CONFIGURATION".Connection.ConnectInfo.SessionTimeout, NodeStatusList := "DB16005_U2_STA3_COAXIAL_CLIENT_INTERFACE".U2_STA3_CAM_Read.NodeStatusList, Done =>, Busy =>, Error =>, Status =>)
   END_RUNG
   RUNG wire#powerrail
      Contact( "DB16000_OPC_UA_TRIGGER_ALARM".CLIENT.U2_STA3_COAXIAL.TRIGGERS.RELEASE_HANDLE_LIST )
      P_Trig( "DB16000_OPC_UA_TRIGGER_ALARM".CLIENT.U2_STA3_COAXIAL.TRIGGERS.RELEASE_HANDLE_LIST_P )
   END_RUNG wire#w1
   // the same network as SCL:
   #_w1 := "DB16000_OPC_UA_TRIGGER_ALARM".CLIENT.U2_STA3_COAXIAL.TRIGGERS.RELEASE_HANDLE_LIST AND NOT "DB16000_OPC_UA_TRIGGER_ALARM".CLIENT.U2_STA3_COAXIAL.TRIGGERS.RELEASE_HANDLE_LIST_P;   // rising edge
   "DB16000_OPC_UA_TRIGGER_ALARM".CLIENT.U2_STA3_COAXIAL.TRIGGERS.RELEASE_HANDLE_LIST_P := "DB16000_OPC_UA_TRIGGER_ALARM".CLIENT.U2_STA3_COAXIAL.TRIGGERS.RELEASE_HANDLE_LIST;
   "DB16246_RELEASE_HANDLE_LIST_U2_STA3_CAM"(REQ := #_w1,   // OPC_UA_NodeReleaseHandleList
                           ConnectionHdl := "DB16105_U2_STA3_CAM_CLIENT_CONFIGURATION".Connection.ConnectionHdl,
                           NodeHdlCount := "DB16105_U2_STA3_CAM_CLIENT_CONFIGURATION".ReadLists.U2_STA3_CAM_Read.NodeCount,
                           NodeHdls := "DB16105_U2_STA3_CAM_CLIENT_CONFIGURATION".ReadLists.U2_STA3_CAM_Read.NodeHdls,
                           Timeout := "DB16105_U2_STA3_CAM_CLIENT_CONFIGURATION".Connection.ConnectInfo.SessionTimeout,
                           NodeStatusList := "DB16005_U2_STA3_COAXIAL_CLIENT_INTERFACE".U2_STA3_CAM_Read.NodeStatusList);
END_REGION

REGION Network 42: UNIT 2 STATION 3 RELEASE METHOD HANDLE CALIBRATIONS LIST CALL
   RUNG wire#powerrail
      "DB16247_RLASE_MD_LIST_U2_STA3_CAM_CALIBS".OPC_UA_MethodReleaseHandleList(REQ := wire#w1, ConnectionHdl := "DB16105_U2_STA3_CAM_CLIENT_CONFIGURATION".Connection.ConnectionHdl, MethodHdlCount := "DB16105_U2_STA3_CAM_CLIENT_CONFIGURATION".MethodLists.U2_STA3_CAM_Calibrations.MethodCount, MethodHdls := "DB16105_U2_STA3_CAM_CLIENT_CONFIGURATION".MethodLists.U2_STA3_CAM_Calibrations.MethodHdls, Timeout := "DB16105_U2_STA3_CAM_CLIENT_CONFIGURATION".Connection.ConnectInfo.SessionTimeout, StatusList := "DB16005_U2_STA3_COAXIAL_CLIENT_INTERFACE".U2_STA3_CAM_Calibrations.MethodStatusList, Done =>, Busy =>, Error =>, Status =>)
   END_RUNG
   RUNG wire#powerrail
      Contact( "DB16000_OPC_UA_TRIGGER_ALARM".CLIENT.U2_STA3_COAXIAL.TRIGGERS.RELEASE_METHOD_LIST_CALIBS )
      P_Trig( "DB16000_OPC_UA_TRIGGER_ALARM".CLIENT.U2_STA3_COAXIAL.TRIGGERS.RELEASE_METHOD_LIST_CALIBS_P )
   END_RUNG wire#w1
   // the same network as SCL:
   #_w1 := "DB16000_OPC_UA_TRIGGER_ALARM".CLIENT.U2_STA3_COAXIAL.TRIGGERS.RELEASE_METHOD_LIST_CALIBS AND NOT "DB16000_OPC_UA_TRIGGER_ALARM".CLIENT.U2_STA3_COAXIAL.TRIGGERS.RELEASE_METHOD_LIST_CALIBS_P;   // rising edge
   "DB16000_OPC_UA_TRIGGER_ALARM".CLIENT.U2_STA3_COAXIAL.TRIGGERS.RELEASE_METHOD_LIST_CALIBS_P := "DB16000_OPC_UA_TRIGGER_ALARM".CLIENT.U2_STA3_COAXIAL.TRIGGERS.RELEASE_METHOD_LIST_CALIBS;
   "DB16247_RLASE_MD_LIST_U2_STA3_CAM_CALIBS"(REQ := #_w1,   // OPC_UA_MethodReleaseHandleList
                           ConnectionHdl := "DB16105_U2_STA3_CAM_CLIENT_CONFIGURATION".Connection.ConnectionHdl,
                           MethodHdlCount := "DB16105_U2_STA3_CAM_CLIENT_CONFIGURATION".MethodLists.U2_STA3_CAM_Calibrations.MethodCount,
                           MethodHdls := "DB16105_U2_STA3_CAM_CLIENT_CONFIGURATION".MethodLists.U2_STA3_CAM_Calibrations.MethodHdls,
                           Timeout := "DB16105_U2_STA3_CAM_CLIENT_CONFIGURATION".Connection.ConnectInfo.SessionTimeout,
                           StatusList := "DB16005_U2_STA3_COAXIAL_CLIENT_INTERFACE".U2_STA3_CAM_Calibrations.MethodStatusList);
END_REGION

REGION Network 43: UNIT 2 STATION 3 RELEASE METHOD HANDLE ANALISIS LIST CALL
   RUNG wire#powerrail
      "DB16248_RLASE_MD_LIST_U2_STA3_CAM_ANALIS".OPC_UA_MethodReleaseHandleList(REQ := wire#w1, ConnectionHdl := "DB16105_U2_STA3_CAM_CLIENT_CONFIGURATION".Connection.ConnectionHdl, MethodHdlCount := "DB16105_U2_STA3_CAM_CLIENT_CONFIGURATION".MethodLists.U2_STA3_CAM_Analysis.MethodCount, MethodHdls := "DB16105_U2_STA3_CAM_CLIENT_CONFIGURATION".MethodLists.U2_STA3_CAM_Analysis.MethodHdls, Timeout := "DB16105_U2_STA3_CAM_CLIENT_CONFIGURATION".Connection.ConnectInfo.SessionTimeout, StatusList := "DB16005_U2_STA3_COAXIAL_CLIENT_INTERFACE".U2_STA3_CAM_Analysis.MethodStatusList, Done =>, Busy =>, Error =>, Status =>)
   END_RUNG
   RUNG wire#powerrail
      Contact( "DB16000_OPC_UA_TRIGGER_ALARM".CLIENT.U2_STA3_COAXIAL.TRIGGERS.RELEASE_METHOD_LIST_ANALISIS )
      P_Trig( "DB16000_OPC_UA_TRIGGER_ALARM".CLIENT.U2_STA3_COAXIAL.TRIGGERS.RELEASE_METHOD_LIST_ANALISIS_P )
   END_RUNG wire#w1
   // the same network as SCL:
   #_w1 := "DB16000_OPC_UA_TRIGGER_ALARM".CLIENT.U2_STA3_COAXIAL.TRIGGERS.RELEASE_METHOD_LIST_ANALISIS AND NOT "DB16000_OPC_UA_TRIGGER_ALARM".CLIENT.U2_STA3_COAXIAL.TRIGGERS.RELEASE_METHOD_LIST_ANALISIS_P;   // rising edge
   "DB16000_OPC_UA_TRIGGER_ALARM".CLIENT.U2_STA3_COAXIAL.TRIGGERS.RELEASE_METHOD_LIST_ANALISIS_P := "DB16000_OPC_UA_TRIGGER_ALARM".CLIENT.U2_STA3_COAXIAL.TRIGGERS.RELEASE_METHOD_LIST_ANALISIS;
   "DB16248_RLASE_MD_LIST_U2_STA3_CAM_ANALIS"(REQ := #_w1,   // OPC_UA_MethodReleaseHandleList
                           ConnectionHdl := "DB16105_U2_STA3_CAM_CLIENT_CONFIGURATION".Connection.ConnectionHdl,
                           MethodHdlCount := "DB16105_U2_STA3_CAM_CLIENT_CONFIGURATION".MethodLists.U2_STA3_CAM_Analysis.MethodCount,
                           MethodHdls := "DB16105_U2_STA3_CAM_CLIENT_CONFIGURATION".MethodLists.U2_STA3_CAM_Analysis.MethodHdls,
                           Timeout := "DB16105_U2_STA3_CAM_CLIENT_CONFIGURATION".Connection.ConnectInfo.SessionTimeout,
                           StatusList := "DB16005_U2_STA3_COAXIAL_CLIENT_INTERFACE".U2_STA3_CAM_Analysis.MethodStatusList);
END_REGION

REGION Network 44: UNIT 2 STATION 3 DISCONNECT CALL
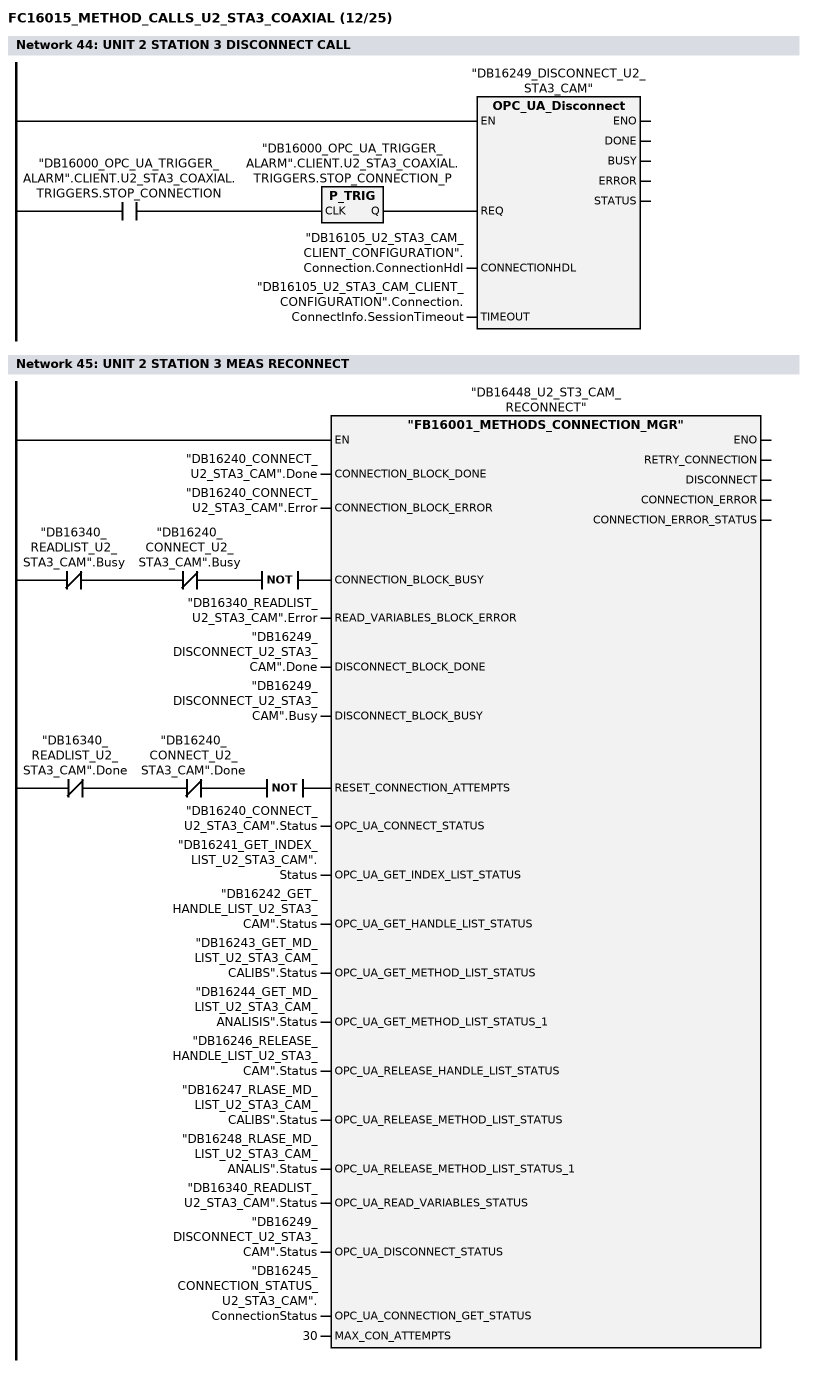
   RUNG wire#powerrail
      "DB16249_DISCONNECT_U2_STA3_CAM".OPC_UA_Disconnect(REQ := wire#w1, ConnectionHdl := "DB16105_U2_STA3_CAM_CLIENT_CONFIGURATION".Connection.ConnectionHdl, Timeout := "DB16105_U2_STA3_CAM_CLIENT_CONFIGURATION".Connection.ConnectInfo.SessionTimeout, Done =>, Busy =>, Error =>, Status =>)
   END_RUNG
   RUNG wire#powerrail
      Contact( "DB16000_OPC_UA_TRIGGER_ALARM".CLIENT.U2_STA3_COAXIAL.TRIGGERS.STOP_CONNECTION )
      P_Trig( "DB16000_OPC_UA_TRIGGER_ALARM".CLIENT.U2_STA3_COAXIAL.TRIGGERS.STOP_CONNECTION_P )
   END_RUNG wire#w1
   // the same network as SCL:
   #_w1 := "DB16000_OPC_UA_TRIGGER_ALARM".CLIENT.U2_STA3_COAXIAL.TRIGGERS.STOP_CONNECTION AND NOT "DB16000_OPC_UA_TRIGGER_ALARM".CLIENT.U2_STA3_COAXIAL.TRIGGERS.STOP_CONNECTION_P;   // rising edge
   "DB16000_OPC_UA_TRIGGER_ALARM".CLIENT.U2_STA3_COAXIAL.TRIGGERS.STOP_CONNECTION_P := "DB16000_OPC_UA_TRIGGER_ALARM".CLIENT.U2_STA3_COAXIAL.TRIGGERS.STOP_CONNECTION;
   "DB16249_DISCONNECT_U2_STA3_CAM"(REQ := #_w1,   // OPC_UA_Disconnect
                           ConnectionHdl := "DB16105_U2_STA3_CAM_CLIENT_CONFIGURATION".Connection.ConnectionHdl,
                           Timeout := "DB16105_U2_STA3_CAM_CLIENT_CONFIGURATION".Connection.ConnectInfo.SessionTimeout);
END_REGION

REGION Network 45: UNIT 2 STATION 3 MEAS RECONNECT
   RUNG wire#powerrail
      "DB16448_U2_ST3_CAM_RECONNECT"(CONNECTION_BLOCK_BUSY := wire#w1, RESET_CONNECTION_ATTEMPTS := wire#w2, CONNECTION_BLOCK_DONE := "DB16240_CONNECT_U2_STA3_CAM".Done, CONNECTION_BLOCK_ERROR := "DB16240_CONNECT_U2_STA3_CAM".Error, READ_VARIABLES_BLOCK_ERROR := "DB16340_READLIST_U2_STA3_CAM".Error, DISCONNECT_BLOCK_DONE := "DB16249_DISCONNECT_U2_STA3_CAM".Done, DISCONNECT_BLOCK_BUSY := "DB16249_DISCONNECT_U2_STA3_CAM".Busy, OPC_UA_CONNECT_STATUS := "DB16240_CONNECT_U2_STA3_CAM".Status, OPC_UA_GET_INDEX_LIST_STATUS := "DB16241_GET_INDEX_LIST_U2_STA3_CAM".Status, OPC_UA_GET_HANDLE_LIST_STATUS := "DB16242_GET_HANDLE_LIST_U2_STA3_CAM".Status, OPC_UA_GET_METHOD_LIST_STATUS := "DB16243_GET_MD_LIST_U2_STA3_CAM_CALIBS".Status, OPC_UA_GET_METHOD_LIST_STATUS_1 := "DB16244_GET_MD_LIST_U2_STA3_CAM_ANALISIS".Status, OPC_UA_RELEASE_HANDLE_LIST_STATUS := "DB16246_RELEASE_HANDLE_LIST_U2_STA3_CAM".Status, OPC_UA_RELEASE_METHOD_LIST_STATUS := "DB16247_RLASE_MD_LIST_U2_STA3_CAM_CALIBS".Status, OPC_UA_RELEASE_METHOD_LIST_STATUS_1 := "DB16248_RLASE_MD_LIST_U2_STA3_CAM_ANALIS".Status, OPC_UA_READ_VARIABLES_STATUS := "DB16340_READLIST_U2_STA3_CAM".Status, OPC_UA_DISCONNECT_STATUS := "DB16249_DISCONNECT_U2_STA3_CAM".Status, OPC_UA_CONNECTION_GET_STATUS := "DB16245_CONNECTION_STATUS_U2_STA3_CAM".ConnectionStatus, MAX_CON_ATTEMPTS := 30, RETRY_CONNECTION =>, DISCONNECT =>, CONNECTION_ERROR =>, CONNECTION_ERROR_STATUS =>)
   END_RUNG
   RUNG wire#powerrail
      I_Contact( "DB16340_READLIST_U2_STA3_CAM".Busy )
      I_Contact( "DB16240_CONNECT_U2_STA3_CAM".Busy )
      Not()
   END_RUNG wire#w1
   RUNG wire#powerrail
      I_Contact( "DB16340_READLIST_U2_STA3_CAM".Done )
      I_Contact( "DB16240_CONNECT_U2_STA3_CAM".Done )
      Not()
   END_RUNG wire#w2
   // the same network as SCL:
   "DB16448_U2_ST3_CAM_RECONNECT"(CONNECTION_BLOCK_DONE := "DB16240_CONNECT_U2_STA3_CAM".Done,   // "FB16001_METHODS_CONNECTION_MGR"
                           CONNECTION_BLOCK_ERROR := "DB16240_CONNECT_U2_STA3_CAM".Error,
                           CONNECTION_BLOCK_BUSY := NOT (NOT "DB16340_READLIST_U2_STA3_CAM".Busy AND NOT "DB16240_CONNECT_U2_STA3_CAM".Busy),
                           READ_VARIABLES_BLOCK_ERROR := "DB16340_READLIST_U2_STA3_CAM".Error,
                           DISCONNECT_BLOCK_DONE := "DB16249_DISCONNECT_U2_STA3_CAM".Done,
                           DISCONNECT_BLOCK_BUSY := "DB16249_DISCONNECT_U2_STA3_CAM".Busy,
                           RESET_CONNECTION_ATTEMPTS := NOT (NOT "DB16340_READLIST_U2_STA3_CAM".Done AND NOT "DB16240_CONNECT_U2_STA3_CAM".Done),
                           OPC_UA_CONNECT_STATUS := "DB16240_CONNECT_U2_STA3_CAM".Status,
                           OPC_UA_GET_INDEX_LIST_STATUS := "DB16241_GET_INDEX_LIST_U2_STA3_CAM".Status,
                           OPC_UA_GET_HANDLE_LIST_STATUS := "DB16242_GET_HANDLE_LIST_U2_STA3_CAM".Status,
                           OPC_UA_GET_METHOD_LIST_STATUS := "DB16243_GET_MD_LIST_U2_STA3_CAM_CALIBS".Status,
                           OPC_UA_GET_METHOD_LIST_STATUS_1 := "DB16244_GET_MD_LIST_U2_STA3_CAM_ANALISIS".Status,
                           OPC_UA_RELEASE_HANDLE_LIST_STATUS := "DB16246_RELEASE_HANDLE_LIST_U2_STA3_CAM".Status,
                           OPC_UA_RELEASE_METHOD_LIST_STATUS := "DB16247_RLASE_MD_LIST_U2_STA3_CAM_CALIBS".Status,
                           OPC_UA_RELEASE_METHOD_LIST_STATUS_1 := "DB16248_RLASE_MD_LIST_U2_STA3_CAM_ANALIS".Status,
                           OPC_UA_READ_VARIABLES_STATUS := "DB16340_READLIST_U2_STA3_CAM".Status,
                           OPC_UA_DISCONNECT_STATUS := "DB16249_DISCONNECT_U2_STA3_CAM".Status,
                           OPC_UA_CONNECTION_GET_STATUS := "DB16245_CONNECTION_STATUS_U2_STA3_CAM".ConnectionStatus,
                           MAX_CON_ATTEMPTS := 30);
END_REGION

REGION Network 46: UNIT 2 PC STATUS UPDATE
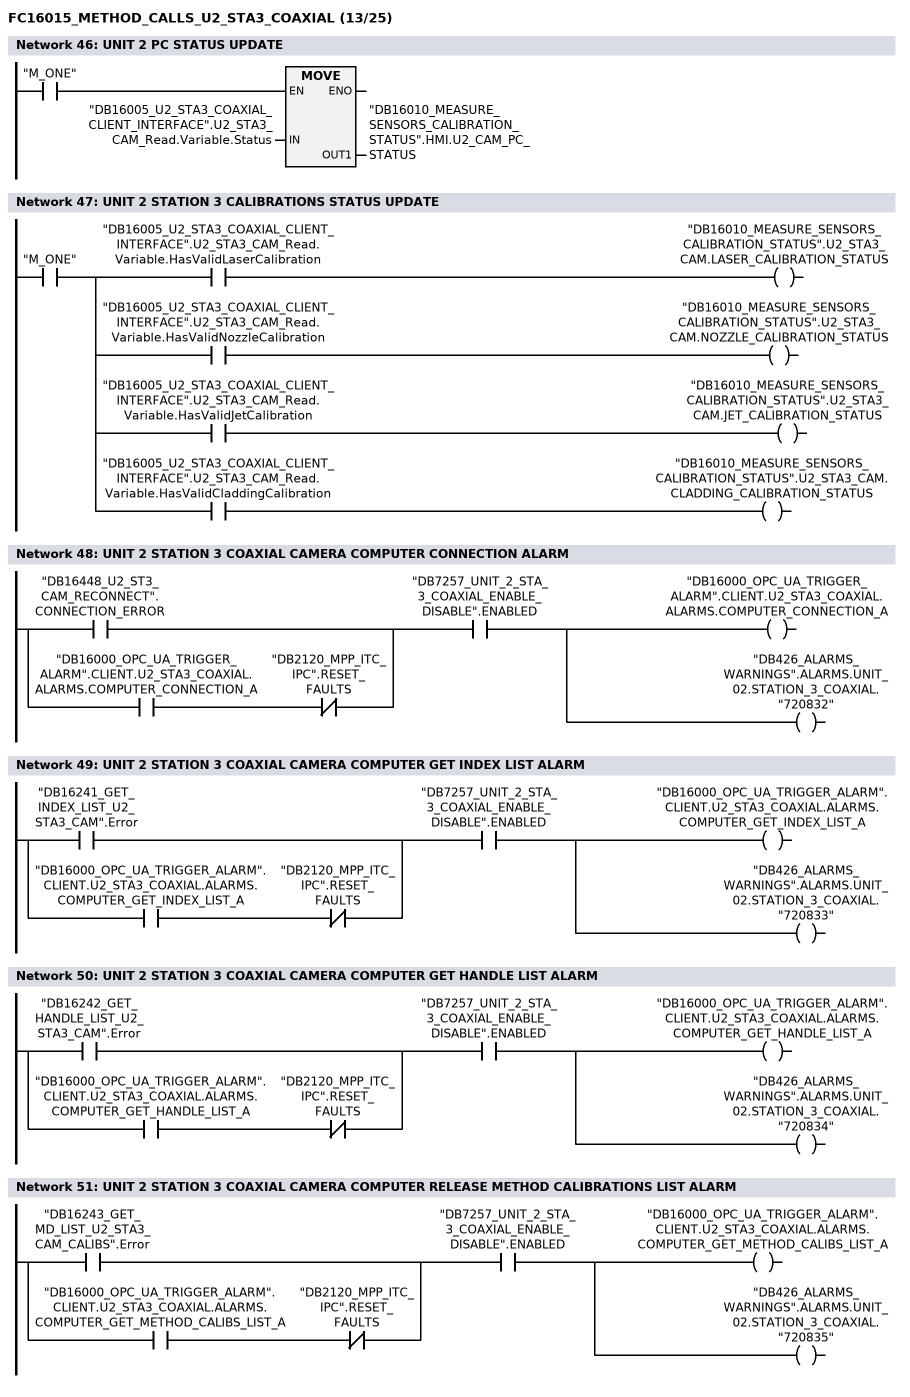
   RUNG wire#powerrail
      Contact( "M_ONE" )
      Move(in := "DB16005_U2_STA3_COAXIAL_CLIENT_INTERFACE".U2_STA3_CAM_Read.Variable.Status, out1 => "DB16010_MEASURE_SENSORS_CALIBRATION_STATUS".HMI.U2_CAM_PC_STATUS)
   END_RUNG
   // the same network as SCL:
   IF "M_ONE" THEN
       "DB16010_MEASURE_SENSORS_CALIBRATION_STATUS".HMI.U2_CAM_PC_STATUS := "DB16005_U2_STA3_COAXIAL_CLIENT_INTERFACE".U2_STA3_CAM_Read.Variable.Status;
   END_IF;
END_REGION

REGION Network 47: UNIT 2 STATION 3 CALIBRATIONS STATUS UPDATE
   RUNG wire#powerrail
      Contact( "M_ONE" )
      wire#w1
      Contact( "DB16005_U2_STA3_COAXIAL_CLIENT_INTERFACE".U2_STA3_CAM_Read.Variable.HasValidLaserCalibration )
      Coil( "DB16010_MEASURE_SENSORS_CALIBRATION_STATUS".U2_STA3_CAM.LASER_CALIBRATION_STATUS )
   END_RUNG
   RUNG wire#w1
      Contact( "DB16005_U2_STA3_COAXIAL_CLIENT_INTERFACE".U2_STA3_CAM_Read.Variable.HasValidNozzleCalibration )
      Coil( "DB16010_MEASURE_SENSORS_CALIBRATION_STATUS".U2_STA3_CAM.NOZZLE_CALIBRATION_STATUS )
   END_RUNG
   RUNG wire#w1
      Contact( "DB16005_U2_STA3_COAXIAL_CLIENT_INTERFACE".U2_STA3_CAM_Read.Variable.HasValidJetCalibration )
      Coil( "DB16010_MEASURE_SENSORS_CALIBRATION_STATUS".U2_STA3_CAM.JET_CALIBRATION_STATUS )
   END_RUNG
   RUNG wire#w1
      Contact( "DB16005_U2_STA3_COAXIAL_CLIENT_INTERFACE".U2_STA3_CAM_Read.Variable.HasValidCladdingCalibration )
      Coil( "DB16010_MEASURE_SENSORS_CALIBRATION_STATUS".U2_STA3_CAM.CLADDING_CALIBRATION_STATUS )
   END_RUNG
   // the same network as SCL:
   "DB16010_MEASURE_SENSORS_CALIBRATION_STATUS".U2_STA3_CAM.LASER_CALIBRATION_STATUS := "M_ONE" AND "DB16005_U2_STA3_COAXIAL_CLIENT_INTERFACE".U2_STA3_CAM_Read.Variable.HasValidLaserCalibration;
   "DB16010_MEASURE_SENSORS_CALIBRATION_STATUS".U2_STA3_CAM.NOZZLE_CALIBRATION_STATUS := "M_ONE" AND "DB16005_U2_STA3_COAXIAL_CLIENT_INTERFACE".U2_STA3_CAM_Read.Variable.HasValidNozzleCalibration;
   "DB16010_MEASURE_SENSORS_CALIBRATION_STATUS".U2_STA3_CAM.JET_CALIBRATION_STATUS := "M_ONE" AND "DB16005_U2_STA3_COAXIAL_CLIENT_INTERFACE".U2_STA3_CAM_Read.Variable.HasValidJetCalibration;
   "DB16010_MEASURE_SENSORS_CALIBRATION_STATUS".U2_STA3_CAM.CLADDING_CALIBRATION_STATUS := "M_ONE" AND "DB16005_U2_STA3_COAXIAL_CLIENT_INTERFACE".U2_STA3_CAM_Read.Variable.HasValidCladdingCalibration;
END_REGION

REGION Network 48: UNIT 2 STATION 3 COAXIAL CAMERA COMPUTER CONNECTION ALARM
   RUNG wire#powerrail
      Contact( "DB16448_U2_ST3_CAM_RECONNECT".CONNECTION_ERROR )
      wire#w1
      Contact( "DB7257_UNIT_2_STA_3_COAXIAL_ENABLE_DISABLE".ENABLED )
      wire#w2
      Coil( "DB16000_OPC_UA_TRIGGER_ALARM".CLIENT.U2_STA3_COAXIAL.ALARMS.COMPUTER_CONNECTION_A )
   END_RUNG
   RUNG wire#powerrail
      Contact( "DB16000_OPC_UA_TRIGGER_ALARM".CLIENT.U2_STA3_COAXIAL.ALARMS.COMPUTER_CONNECTION_A )
      I_Contact( "DB2120_MPP_ITC_IPC".RESET_FAULTS )
   END_RUNG wire#w1
   RUNG wire#w2
      Coil( "DB426_ALARMS_WARNINGS".ALARMS.UNIT_02.STATION_3_COAXIAL."720832" )
   END_RUNG
   // the same network as SCL:
   "DB16000_OPC_UA_TRIGGER_ALARM".CLIENT.U2_STA3_COAXIAL.ALARMS.COMPUTER_CONNECTION_A := ("DB16448_U2_ST3_CAM_RECONNECT".CONNECTION_ERROR OR ("DB16000_OPC_UA_TRIGGER_ALARM".CLIENT.U2_STA3_COAXIAL.ALARMS.COMPUTER_CONNECTION_A AND NOT "DB2120_MPP_ITC_IPC".RESET_FAULTS)) AND "DB7257_UNIT_2_STA_3_COAXIAL_ENABLE_DISABLE".ENABLED;
   "DB426_ALARMS_WARNINGS".ALARMS.UNIT_02.STATION_3_COAXIAL."720832" := "DB16000_OPC_UA_TRIGGER_ALARM".CLIENT.U2_STA3_COAXIAL.ALARMS.COMPUTER_CONNECTION_A;
END_REGION

REGION Network 49: UNIT 2 STATION 3 COAXIAL CAMERA COMPUTER GET INDEX LIST ALARM
   RUNG wire#powerrail
      Contact( "DB16241_GET_INDEX_LIST_U2_STA3_CAM".Error )
      wire#w1
      Contact( "DB7257_UNIT_2_STA_3_COAXIAL_ENABLE_DISABLE".ENABLED )
      wire#w2
      Coil( "DB16000_OPC_UA_TRIGGER_ALARM".CLIENT.U2_STA3_COAXIAL.ALARMS.COMPUTER_GET_INDEX_LIST_A )
   END_RUNG
   RUNG wire#powerrail
      Contact( "DB16000_OPC_UA_TRIGGER_ALARM".CLIENT.U2_STA3_COAXIAL.ALARMS.COMPUTER_GET_INDEX_LIST_A )
      I_Contact( "DB2120_MPP_ITC_IPC".RESET_FAULTS )
   END_RUNG wire#w1
   RUNG wire#w2
      Coil( "DB426_ALARMS_WARNINGS".ALARMS.UNIT_02.STATION_3_COAXIAL."720833" )
   END_RUNG
   // the same network as SCL:
   "DB16000_OPC_UA_TRIGGER_ALARM".CLIENT.U2_STA3_COAXIAL.ALARMS.COMPUTER_GET_INDEX_LIST_A := ("DB16241_GET_INDEX_LIST_U2_STA3_CAM".Error OR ("DB16000_OPC_UA_TRIGGER_ALARM".CLIENT.U2_STA3_COAXIAL.ALARMS.COMPUTER_GET_INDEX_LIST_A AND NOT "DB2120_MPP_ITC_IPC".RESET_FAULTS)) AND "DB7257_UNIT_2_STA_3_COAXIAL_ENABLE_DISABLE".ENABLED;
   "DB426_ALARMS_WARNINGS".ALARMS.UNIT_02.STATION_3_COAXIAL."720833" := "DB16000_OPC_UA_TRIGGER_ALARM".CLIENT.U2_STA3_COAXIAL.ALARMS.COMPUTER_GET_INDEX_LIST_A;
END_REGION

REGION Network 50: UNIT 2 STATION 3 COAXIAL CAMERA COMPUTER GET HANDLE LIST ALARM
   RUNG wire#powerrail
      Contact( "DB16242_GET_HANDLE_LIST_U2_STA3_CAM".Error )
      wire#w1
      Contact( "DB7257_UNIT_2_STA_3_COAXIAL_ENABLE_DISABLE".ENABLED )
      wire#w2
      Coil( "DB16000_OPC_UA_TRIGGER_ALARM".CLIENT.U2_STA3_COAXIAL.ALARMS.COMPUTER_GET_HANDLE_LIST_A )
   END_RUNG
   RUNG wire#powerrail
      Contact( "DB16000_OPC_UA_TRIGGER_ALARM".CLIENT.U2_STA3_COAXIAL.ALARMS.COMPUTER_GET_HANDLE_LIST_A )
      I_Contact( "DB2120_MPP_ITC_IPC".RESET_FAULTS )
   END_RUNG wire#w1
   RUNG wire#w2
      Coil( "DB426_ALARMS_WARNINGS".ALARMS.UNIT_02.STATION_3_COAXIAL."720834" )
   END_RUNG
   // the same network as SCL:
   "DB16000_OPC_UA_TRIGGER_ALARM".CLIENT.U2_STA3_COAXIAL.ALARMS.COMPUTER_GET_HANDLE_LIST_A := ("DB16242_GET_HANDLE_LIST_U2_STA3_CAM".Error OR ("DB16000_OPC_UA_TRIGGER_ALARM".CLIENT.U2_STA3_COAXIAL.ALARMS.COMPUTER_GET_HANDLE_LIST_A AND NOT "DB2120_MPP_ITC_IPC".RESET_FAULTS)) AND "DB7257_UNIT_2_STA_3_COAXIAL_ENABLE_DISABLE".ENABLED;
   "DB426_ALARMS_WARNINGS".ALARMS.UNIT_02.STATION_3_COAXIAL."720834" := "DB16000_OPC_UA_TRIGGER_ALARM".CLIENT.U2_STA3_COAXIAL.ALARMS.COMPUTER_GET_HANDLE_LIST_A;
END_REGION

REGION Network 51: UNIT 2 STATION 3 COAXIAL CAMERA COMPUTER RELEASE METHOD CALIBRATIONS LIST ALARM
   RUNG wire#powerrail
      Contact( "DB16243_GET_MD_LIST_U2_STA3_CAM_CALIBS".Error )
      wire#w1
      Contact( "DB7257_UNIT_2_STA_3_COAXIAL_ENABLE_DISABLE".ENABLED )
      wire#w2
      Coil( "DB16000_OPC_UA_TRIGGER_ALARM".CLIENT.U2_STA3_COAXIAL.ALARMS.COMPUTER_GET_METHOD_CALIBS_LIST_A )
   END_RUNG
   RUNG wire#powerrail
      Contact( "DB16000_OPC_UA_TRIGGER_ALARM".CLIENT.U2_STA3_COAXIAL.ALARMS.COMPUTER_GET_METHOD_CALIBS_LIST_A )
      I_Contact( "DB2120_MPP_ITC_IPC".RESET_FAULTS )
   END_RUNG wire#w1
   RUNG wire#w2
      Coil( "DB426_ALARMS_WARNINGS".ALARMS.UNIT_02.STATION_3_COAXIAL."720835" )
   END_RUNG
   // the same network as SCL:
   "DB16000_OPC_UA_TRIGGER_ALARM".CLIENT.U2_STA3_COAXIAL.ALARMS.COMPUTER_GET_METHOD_CALIBS_LIST_A := ("DB16243_GET_MD_LIST_U2_STA3_CAM_CALIBS".Error OR ("DB16000_OPC_UA_TRIGGER_ALARM".CLIENT.U2_STA3_COAXIAL.ALARMS.COMPUTER_GET_METHOD_CALIBS_LIST_A AND NOT "DB2120_MPP_ITC_IPC".RESET_FAULTS)) AND "DB7257_UNIT_2_STA_3_COAXIAL_ENABLE_DISABLE".ENABLED;
   "DB426_ALARMS_WARNINGS".ALARMS.UNIT_02.STATION_3_COAXIAL."720835" := "DB16000_OPC_UA_TRIGGER_ALARM".CLIENT.U2_STA3_COAXIAL.ALARMS.COMPUTER_GET_METHOD_CALIBS_LIST_A;
END_REGION

REGION Network 52: UNIT 2 STATION 3 COAXIAL CAMERA COMPUTER RELEASE METHOD ANALISIS LIST ALARM
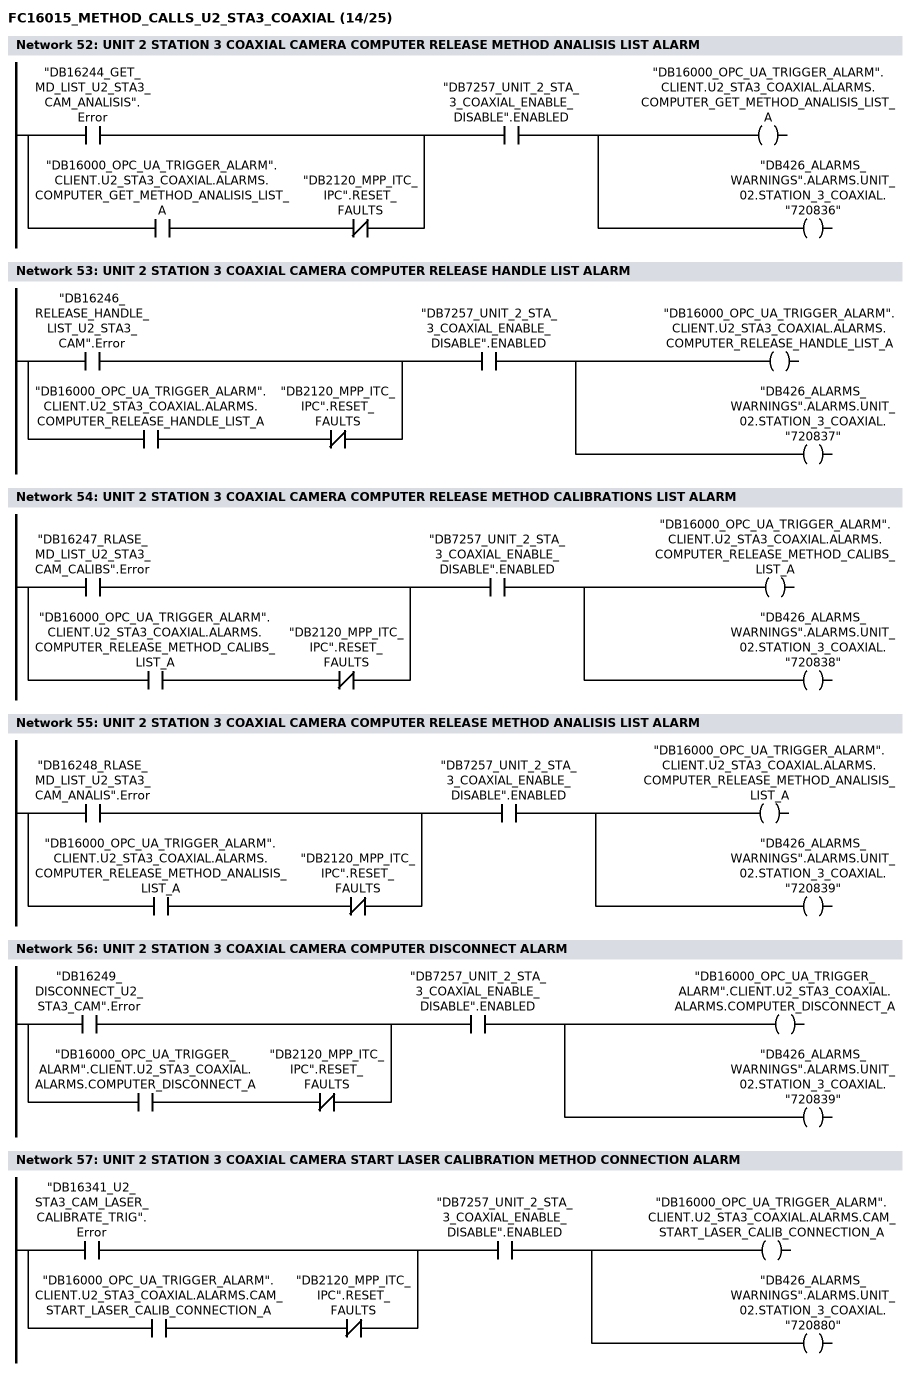
   RUNG wire#powerrail
      Contact( "DB16244_GET_MD_LIST_U2_STA3_CAM_ANALISIS".Error )
      wire#w1
      Contact( "DB7257_UNIT_2_STA_3_COAXIAL_ENABLE_DISABLE".ENABLED )
      wire#w2
      Coil( "DB16000_OPC_UA_TRIGGER_ALARM".CLIENT.U2_STA3_COAXIAL.ALARMS.COMPUTER_GET_METHOD_ANALISIS_LIST_A )
   END_RUNG
   RUNG wire#powerrail
      Contact( "DB16000_OPC_UA_TRIGGER_ALARM".CLIENT.U2_STA3_COAXIAL.ALARMS.COMPUTER_GET_METHOD_ANALISIS_LIST_A )
      I_Contact( "DB2120_MPP_ITC_IPC".RESET_FAULTS )
   END_RUNG wire#w1
   RUNG wire#w2
      Coil( "DB426_ALARMS_WARNINGS".ALARMS.UNIT_02.STATION_3_COAXIAL."720836" )
   END_RUNG
   // the same network as SCL:
   "DB16000_OPC_UA_TRIGGER_ALARM".CLIENT.U2_STA3_COAXIAL.ALARMS.COMPUTER_GET_METHOD_ANALISIS_LIST_A := ("DB16244_GET_MD_LIST_U2_STA3_CAM_ANALISIS".Error OR ("DB16000_OPC_UA_TRIGGER_ALARM".CLIENT.U2_STA3_COAXIAL.ALARMS.COMPUTER_GET_METHOD_ANALISIS_LIST_A AND NOT "DB2120_MPP_ITC_IPC".RESET_FAULTS)) AND "DB7257_UNIT_2_STA_3_COAXIAL_ENABLE_DISABLE".ENABLED;
   "DB426_ALARMS_WARNINGS".ALARMS.UNIT_02.STATION_3_COAXIAL."720836" := "DB16000_OPC_UA_TRIGGER_ALARM".CLIENT.U2_STA3_COAXIAL.ALARMS.COMPUTER_GET_METHOD_ANALISIS_LIST_A;
END_REGION

REGION Network 53: UNIT 2 STATION 3 COAXIAL CAMERA COMPUTER RELEASE HANDLE LIST ALARM
   RUNG wire#powerrail
      Contact( "DB16246_RELEASE_HANDLE_LIST_U2_STA3_CAM".Error )
      wire#w1
      Contact( "DB7257_UNIT_2_STA_3_COAXIAL_ENABLE_DISABLE".ENABLED )
      wire#w2
      Coil( "DB16000_OPC_UA_TRIGGER_ALARM".CLIENT.U2_STA3_COAXIAL.ALARMS.COMPUTER_RELEASE_HANDLE_LIST_A )
   END_RUNG
   RUNG wire#powerrail
      Contact( "DB16000_OPC_UA_TRIGGER_ALARM".CLIENT.U2_STA3_COAXIAL.ALARMS.COMPUTER_RELEASE_HANDLE_LIST_A )
      I_Contact( "DB2120_MPP_ITC_IPC".RESET_FAULTS )
   END_RUNG wire#w1
   RUNG wire#w2
      Coil( "DB426_ALARMS_WARNINGS".ALARMS.UNIT_02.STATION_3_COAXIAL."720837" )
   END_RUNG
   // the same network as SCL:
   "DB16000_OPC_UA_TRIGGER_ALARM".CLIENT.U2_STA3_COAXIAL.ALARMS.COMPUTER_RELEASE_HANDLE_LIST_A := ("DB16246_RELEASE_HANDLE_LIST_U2_STA3_CAM".Error OR ("DB16000_OPC_UA_TRIGGER_ALARM".CLIENT.U2_STA3_COAXIAL.ALARMS.COMPUTER_RELEASE_HANDLE_LIST_A AND NOT "DB2120_MPP_ITC_IPC".RESET_FAULTS)) AND "DB7257_UNIT_2_STA_3_COAXIAL_ENABLE_DISABLE".ENABLED;
   "DB426_ALARMS_WARNINGS".ALARMS.UNIT_02.STATION_3_COAXIAL."720837" := "DB16000_OPC_UA_TRIGGER_ALARM".CLIENT.U2_STA3_COAXIAL.ALARMS.COMPUTER_RELEASE_HANDLE_LIST_A;
END_REGION

REGION Network 54: UNIT 2 STATION 3 COAXIAL CAMERA COMPUTER RELEASE METHOD CALIBRATIONS LIST ALARM
   RUNG wire#powerrail
      Contact( "DB16247_RLASE_MD_LIST_U2_STA3_CAM_CALIBS".Error )
      wire#w1
      Contact( "DB7257_UNIT_2_STA_3_COAXIAL_ENABLE_DISABLE".ENABLED )
      wire#w2
      Coil( "DB16000_OPC_UA_TRIGGER_ALARM".CLIENT.U2_STA3_COAXIAL.ALARMS.COMPUTER_RELEASE_METHOD_CALIBS_LIST_A )
   END_RUNG
   RUNG wire#powerrail
      Contact( "DB16000_OPC_UA_TRIGGER_ALARM".CLIENT.U2_STA3_COAXIAL.ALARMS.COMPUTER_RELEASE_METHOD_CALIBS_LIST_A )
      I_Contact( "DB2120_MPP_ITC_IPC".RESET_FAULTS )
   END_RUNG wire#w1
   RUNG wire#w2
      Coil( "DB426_ALARMS_WARNINGS".ALARMS.UNIT_02.STATION_3_COAXIAL."720838" )
   END_RUNG
   // the same network as SCL:
   "DB16000_OPC_UA_TRIGGER_ALARM".CLIENT.U2_STA3_COAXIAL.ALARMS.COMPUTER_RELEASE_METHOD_CALIBS_LIST_A := ("DB16247_RLASE_MD_LIST_U2_STA3_CAM_CALIBS".Error OR ("DB16000_OPC_UA_TRIGGER_ALARM".CLIENT.U2_STA3_COAXIAL.ALARMS.COMPUTER_RELEASE_METHOD_CALIBS_LIST_A AND NOT "DB2120_MPP_ITC_IPC".RESET_FAULTS)) AND "DB7257_UNIT_2_STA_3_COAXIAL_ENABLE_DISABLE".ENABLED;
   "DB426_ALARMS_WARNINGS".ALARMS.UNIT_02.STATION_3_COAXIAL."720838" := "DB16000_OPC_UA_TRIGGER_ALARM".CLIENT.U2_STA3_COAXIAL.ALARMS.COMPUTER_RELEASE_METHOD_CALIBS_LIST_A;
END_REGION

REGION Network 55: UNIT 2 STATION 3 COAXIAL CAMERA COMPUTER RELEASE METHOD ANALISIS LIST ALARM
   RUNG wire#powerrail
      Contact( "DB16248_RLASE_MD_LIST_U2_STA3_CAM_ANALIS".Error )
      wire#w1
      Contact( "DB7257_UNIT_2_STA_3_COAXIAL_ENABLE_DISABLE".ENABLED )
      wire#w2
      Coil( "DB16000_OPC_UA_TRIGGER_ALARM".CLIENT.U2_STA3_COAXIAL.ALARMS.COMPUTER_RELEASE_METHOD_ANALISIS_LIST_A )
   END_RUNG
   RUNG wire#powerrail
      Contact( "DB16000_OPC_UA_TRIGGER_ALARM".CLIENT.U2_STA3_COAXIAL.ALARMS.COMPUTER_RELEASE_METHOD_ANALISIS_LIST_A )
      I_Contact( "DB2120_MPP_ITC_IPC".RESET_FAULTS )
   END_RUNG wire#w1
   RUNG wire#w2
      Coil( "DB426_ALARMS_WARNINGS".ALARMS.UNIT_02.STATION_3_COAXIAL."720839" )
   END_RUNG
   // the same network as SCL:
   "DB16000_OPC_UA_TRIGGER_ALARM".CLIENT.U2_STA3_COAXIAL.ALARMS.COMPUTER_RELEASE_METHOD_ANALISIS_LIST_A := ("DB16248_RLASE_MD_LIST_U2_STA3_CAM_ANALIS".Error OR ("DB16000_OPC_UA_TRIGGER_ALARM".CLIENT.U2_STA3_COAXIAL.ALARMS.COMPUTER_RELEASE_METHOD_ANALISIS_LIST_A AND NOT "DB2120_MPP_ITC_IPC".RESET_FAULTS)) AND "DB7257_UNIT_2_STA_3_COAXIAL_ENABLE_DISABLE".ENABLED;
   "DB426_ALARMS_WARNINGS".ALARMS.UNIT_02.STATION_3_COAXIAL."720839" := "DB16000_OPC_UA_TRIGGER_ALARM".CLIENT.U2_STA3_COAXIAL.ALARMS.COMPUTER_RELEASE_METHOD_ANALISIS_LIST_A;
END_REGION

REGION Network 56: UNIT 2 STATION 3 COAXIAL CAMERA COMPUTER DISCONNECT ALARM
   RUNG wire#powerrail
      Contact( "DB16249_DISCONNECT_U2_STA3_CAM".Error )
      wire#w1
      Contact( "DB7257_UNIT_2_STA_3_COAXIAL_ENABLE_DISABLE".ENABLED )
      wire#w2
      Coil( "DB16000_OPC_UA_TRIGGER_ALARM".CLIENT.U2_STA3_COAXIAL.ALARMS.COMPUTER_DISCONNECT_A )
   END_RUNG
   RUNG wire#powerrail
      Contact( "DB16000_OPC_UA_TRIGGER_ALARM".CLIENT.U2_STA3_COAXIAL.ALARMS.COMPUTER_DISCONNECT_A )
      I_Contact( "DB2120_MPP_ITC_IPC".RESET_FAULTS )
   END_RUNG wire#w1
   RUNG wire#w2
      Coil( "DB426_ALARMS_WARNINGS".ALARMS.UNIT_02.STATION_3_COAXIAL."720839" )
   END_RUNG
   // the same network as SCL:
   "DB16000_OPC_UA_TRIGGER_ALARM".CLIENT.U2_STA3_COAXIAL.ALARMS.COMPUTER_DISCONNECT_A := ("DB16249_DISCONNECT_U2_STA3_CAM".Error OR ("DB16000_OPC_UA_TRIGGER_ALARM".CLIENT.U2_STA3_COAXIAL.ALARMS.COMPUTER_DISCONNECT_A AND NOT "DB2120_MPP_ITC_IPC".RESET_FAULTS)) AND "DB7257_UNIT_2_STA_3_COAXIAL_ENABLE_DISABLE".ENABLED;
   "DB426_ALARMS_WARNINGS".ALARMS.UNIT_02.STATION_3_COAXIAL."720839" := "DB16000_OPC_UA_TRIGGER_ALARM".CLIENT.U2_STA3_COAXIAL.ALARMS.COMPUTER_DISCONNECT_A;
END_REGION

REGION Network 57: UNIT 2 STATION 3 COAXIAL CAMERA START LASER CALIBRATION METHOD CONNECTION ALARM
   RUNG wire#powerrail
      Contact( "DB16341_U2_STA3_CAM_LASER_CALIBRATE_TRIG".Error )
      wire#w1
      Contact( "DB7257_UNIT_2_STA_3_COAXIAL_ENABLE_DISABLE".ENABLED )
      wire#w2
      Coil( "DB16000_OPC_UA_TRIGGER_ALARM".CLIENT.U2_STA3_COAXIAL.ALARMS.CAM_START_LASER_CALIB_CONNECTION_A )
   END_RUNG
   RUNG wire#powerrail
      Contact( "DB16000_OPC_UA_TRIGGER_ALARM".CLIENT.U2_STA3_COAXIAL.ALARMS.CAM_START_LASER_CALIB_CONNECTION_A )
      I_Contact( "DB2120_MPP_ITC_IPC".RESET_FAULTS )
   END_RUNG wire#w1
   RUNG wire#w2
      Coil( "DB426_ALARMS_WARNINGS".ALARMS.UNIT_02.STATION_3_COAXIAL."720880" )
   END_RUNG
   // the same network as SCL:
   "DB16000_OPC_UA_TRIGGER_ALARM".CLIENT.U2_STA3_COAXIAL.ALARMS.CAM_START_LASER_CALIB_CONNECTION_A := ("DB16341_U2_STA3_CAM_LASER_CALIBRATE_TRIG".Error OR ("DB16000_OPC_UA_TRIGGER_ALARM".CLIENT.U2_STA3_COAXIAL.ALARMS.CAM_START_LASER_CALIB_CONNECTION_A AND NOT "DB2120_MPP_ITC_IPC".RESET_FAULTS)) AND "DB7257_UNIT_2_STA_3_COAXIAL_ENABLE_DISABLE".ENABLED;
   "DB426_ALARMS_WARNINGS".ALARMS.UNIT_02.STATION_3_COAXIAL."720880" := "DB16000_OPC_UA_TRIGGER_ALARM".CLIENT.U2_STA3_COAXIAL.ALARMS.CAM_START_LASER_CALIB_CONNECTION_A;
END_REGION

REGION Network 58: UNIT 2 STATION 3 COAXIAL CAMERA START LASER CALIBRATION METHOD WORKING OR BLOCKED ALARM
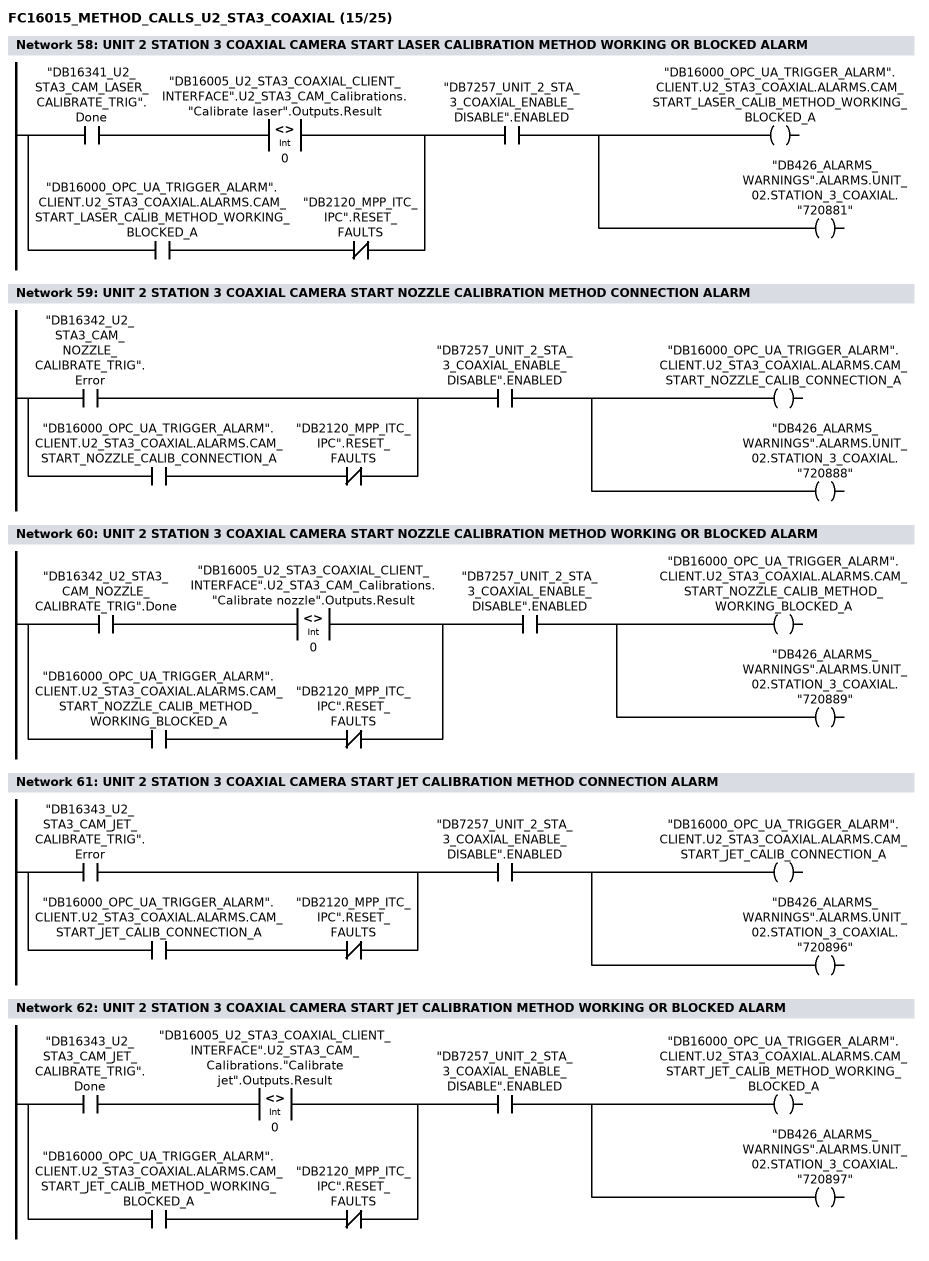
   RUNG wire#powerrail
      Contact( "DB16341_U2_STA3_CAM_LASER_CALIBRATE_TRIG".Done )
      { S7_Templates := "SrcType := Int" } NE_Contact(in1 := "DB16005_U2_STA3_COAXIAL_CLIENT_INTERFACE".U2_STA3_CAM_Calibrations."Calibrate laser".Outputs.Result, in2 := 0)
      wire#w1
      Contact( "DB7257_UNIT_2_STA_3_COAXIAL_ENABLE_DISABLE".ENABLED )
      wire#w2
      Coil( "DB16000_OPC_UA_TRIGGER_ALARM".CLIENT.U2_STA3_COAXIAL.ALARMS.CAM_START_LASER_CALIB_METHOD_WORKING_BLOCKED_A )
   END_RUNG
   RUNG wire#powerrail
      Contact( "DB16000_OPC_UA_TRIGGER_ALARM".CLIENT.U2_STA3_COAXIAL.ALARMS.CAM_START_LASER_CALIB_METHOD_WORKING_BLOCKED_A )
      I_Contact( "DB2120_MPP_ITC_IPC".RESET_FAULTS )
   END_RUNG wire#w1
   RUNG wire#w2
      Coil( "DB426_ALARMS_WARNINGS".ALARMS.UNIT_02.STATION_3_COAXIAL."720881" )
   END_RUNG
   // the same network as SCL:
   "DB16000_OPC_UA_TRIGGER_ALARM".CLIENT.U2_STA3_COAXIAL.ALARMS.CAM_START_LASER_CALIB_METHOD_WORKING_BLOCKED_A := (("DB16341_U2_STA3_CAM_LASER_CALIBRATE_TRIG".Done AND ("DB16005_U2_STA3_COAXIAL_CLIENT_INTERFACE".U2_STA3_CAM_Calibrations."Calibrate laser".Outputs.Result <> 0)) OR ("DB16000_OPC_UA_TRIGGER_ALARM".CLIENT.U2_STA3_COAXIAL.ALARMS.CAM_START_LASER_CALIB_METHOD_WORKING_BLOCKED_A AND NOT "DB2120_MPP_ITC_IPC".RESET_FAULTS)) AND "DB7257_UNIT_2_STA_3_COAXIAL_ENABLE_DISABLE".ENABLED;
   "DB426_ALARMS_WARNINGS".ALARMS.UNIT_02.STATION_3_COAXIAL."720881" := "DB16000_OPC_UA_TRIGGER_ALARM".CLIENT.U2_STA3_COAXIAL.ALARMS.CAM_START_LASER_CALIB_METHOD_WORKING_BLOCKED_A;
END_REGION

REGION Network 59: UNIT 2 STATION 3 COAXIAL CAMERA START NOZZLE CALIBRATION METHOD CONNECTION ALARM
   RUNG wire#powerrail
      Contact( "DB16342_U2_STA3_CAM_NOZZLE_CALIBRATE_TRIG".Error )
      wire#w1
      Contact( "DB7257_UNIT_2_STA_3_COAXIAL_ENABLE_DISABLE".ENABLED )
      wire#w2
      Coil( "DB16000_OPC_UA_TRIGGER_ALARM".CLIENT.U2_STA3_COAXIAL.ALARMS.CAM_START_NOZZLE_CALIB_CONNECTION_A )
   END_RUNG
   RUNG wire#powerrail
      Contact( "DB16000_OPC_UA_TRIGGER_ALARM".CLIENT.U2_STA3_COAXIAL.ALARMS.CAM_START_NOZZLE_CALIB_CONNECTION_A )
      I_Contact( "DB2120_MPP_ITC_IPC".RESET_FAULTS )
   END_RUNG wire#w1
   RUNG wire#w2
      Coil( "DB426_ALARMS_WARNINGS".ALARMS.UNIT_02.STATION_3_COAXIAL."720888" )
   END_RUNG
   // the same network as SCL:
   "DB16000_OPC_UA_TRIGGER_ALARM".CLIENT.U2_STA3_COAXIAL.ALARMS.CAM_START_NOZZLE_CALIB_CONNECTION_A := ("DB16342_U2_STA3_CAM_NOZZLE_CALIBRATE_TRIG".Error OR ("DB16000_OPC_UA_TRIGGER_ALARM".CLIENT.U2_STA3_COAXIAL.ALARMS.CAM_START_NOZZLE_CALIB_CONNECTION_A AND NOT "DB2120_MPP_ITC_IPC".RESET_FAULTS)) AND "DB7257_UNIT_2_STA_3_COAXIAL_ENABLE_DISABLE".ENABLED;
   "DB426_ALARMS_WARNINGS".ALARMS.UNIT_02.STATION_3_COAXIAL."720888" := "DB16000_OPC_UA_TRIGGER_ALARM".CLIENT.U2_STA3_COAXIAL.ALARMS.CAM_START_NOZZLE_CALIB_CONNECTION_A;
END_REGION

REGION Network 60: UNIT 2 STATION 3 COAXIAL CAMERA START NOZZLE CALIBRATION METHOD WORKING OR BLOCKED ALARM
   RUNG wire#powerrail
      Contact( "DB16342_U2_STA3_CAM_NOZZLE_CALIBRATE_TRIG".Done )
      { S7_Templates := "SrcType := Int" } NE_Contact(in1 := "DB16005_U2_STA3_COAXIAL_CLIENT_INTERFACE".U2_STA3_CAM_Calibrations."Calibrate nozzle".Outputs.Result, in2 := 0)
      wire#w1
      Contact( "DB7257_UNIT_2_STA_3_COAXIAL_ENABLE_DISABLE".ENABLED )
      wire#w2
      Coil( "DB16000_OPC_UA_TRIGGER_ALARM".CLIENT.U2_STA3_COAXIAL.ALARMS.CAM_START_NOZZLE_CALIB_METHOD_WORKING_BLOCKED_A )
   END_RUNG
   RUNG wire#powerrail
      Contact( "DB16000_OPC_UA_TRIGGER_ALARM".CLIENT.U2_STA3_COAXIAL.ALARMS.CAM_START_NOZZLE_CALIB_METHOD_WORKING_BLOCKED_A )
      I_Contact( "DB2120_MPP_ITC_IPC".RESET_FAULTS )
   END_RUNG wire#w1
   RUNG wire#w2
      Coil( "DB426_ALARMS_WARNINGS".ALARMS.UNIT_02.STATION_3_COAXIAL."720889" )
   END_RUNG
   // the same network as SCL:
   "DB16000_OPC_UA_TRIGGER_ALARM".CLIENT.U2_STA3_COAXIAL.ALARMS.CAM_START_NOZZLE_CALIB_METHOD_WORKING_BLOCKED_A := (("DB16342_U2_STA3_CAM_NOZZLE_CALIBRATE_TRIG".Done AND ("DB16005_U2_STA3_COAXIAL_CLIENT_INTERFACE".U2_STA3_CAM_Calibrations."Calibrate nozzle".Outputs.Result <> 0)) OR ("DB16000_OPC_UA_TRIGGER_ALARM".CLIENT.U2_STA3_COAXIAL.ALARMS.CAM_START_NOZZLE_CALIB_METHOD_WORKING_BLOCKED_A AND NOT "DB2120_MPP_ITC_IPC".RESET_FAULTS)) AND "DB7257_UNIT_2_STA_3_COAXIAL_ENABLE_DISABLE".ENABLED;
   "DB426_ALARMS_WARNINGS".ALARMS.UNIT_02.STATION_3_COAXIAL."720889" := "DB16000_OPC_UA_TRIGGER_ALARM".CLIENT.U2_STA3_COAXIAL.ALARMS.CAM_START_NOZZLE_CALIB_METHOD_WORKING_BLOCKED_A;
END_REGION

REGION Network 61: UNIT 2 STATION 3 COAXIAL CAMERA START JET CALIBRATION METHOD CONNECTION ALARM
   RUNG wire#powerrail
      Contact( "DB16343_U2_STA3_CAM_JET_CALIBRATE_TRIG".Error )
      wire#w1
      Contact( "DB7257_UNIT_2_STA_3_COAXIAL_ENABLE_DISABLE".ENABLED )
      wire#w2
      Coil( "DB16000_OPC_UA_TRIGGER_ALARM".CLIENT.U2_STA3_COAXIAL.ALARMS.CAM_START_JET_CALIB_CONNECTION_A )
   END_RUNG
   RUNG wire#powerrail
      Contact( "DB16000_OPC_UA_TRIGGER_ALARM".CLIENT.U2_STA3_COAXIAL.ALARMS.CAM_START_JET_CALIB_CONNECTION_A )
      I_Contact( "DB2120_MPP_ITC_IPC".RESET_FAULTS )
   END_RUNG wire#w1
   RUNG wire#w2
      Coil( "DB426_ALARMS_WARNINGS".ALARMS.UNIT_02.STATION_3_COAXIAL."720896" )
   END_RUNG
   // the same network as SCL:
   "DB16000_OPC_UA_TRIGGER_ALARM".CLIENT.U2_STA3_COAXIAL.ALARMS.CAM_START_JET_CALIB_CONNECTION_A := ("DB16343_U2_STA3_CAM_JET_CALIBRATE_TRIG".Error OR ("DB16000_OPC_UA_TRIGGER_ALARM".CLIENT.U2_STA3_COAXIAL.ALARMS.CAM_START_JET_CALIB_CONNECTION_A AND NOT "DB2120_MPP_ITC_IPC".RESET_FAULTS)) AND "DB7257_UNIT_2_STA_3_COAXIAL_ENABLE_DISABLE".ENABLED;
   "DB426_ALARMS_WARNINGS".ALARMS.UNIT_02.STATION_3_COAXIAL."720896" := "DB16000_OPC_UA_TRIGGER_ALARM".CLIENT.U2_STA3_COAXIAL.ALARMS.CAM_START_JET_CALIB_CONNECTION_A;
END_REGION

REGION Network 62: UNIT 2 STATION 3 COAXIAL CAMERA START JET CALIBRATION METHOD WORKING OR BLOCKED ALARM
   RUNG wire#powerrail
      Contact( "DB16343_U2_STA3_CAM_JET_CALIBRATE_TRIG".Done )
      { S7_Templates := "SrcType := Int" } NE_Contact(in1 := "DB16005_U2_STA3_COAXIAL_CLIENT_INTERFACE".U2_STA3_CAM_Calibrations."Calibrate jet".Outputs.Result, in2 := 0)
      wire#w1
      Contact( "DB7257_UNIT_2_STA_3_COAXIAL_ENABLE_DISABLE".ENABLED )
      wire#w2
      Coil( "DB16000_OPC_UA_TRIGGER_ALARM".CLIENT.U2_STA3_COAXIAL.ALARMS.CAM_START_JET_CALIB_METHOD_WORKING_BLOCKED_A )
   END_RUNG
   RUNG wire#powerrail
      Contact( "DB16000_OPC_UA_TRIGGER_ALARM".CLIENT.U2_STA3_COAXIAL.ALARMS.CAM_START_JET_CALIB_METHOD_WORKING_BLOCKED_A )
      I_Contact( "DB2120_MPP_ITC_IPC".RESET_FAULTS )
   END_RUNG wire#w1
   RUNG wire#w2
      Coil( "DB426_ALARMS_WARNINGS".ALARMS.UNIT_02.STATION_3_COAXIAL."720897" )
   END_RUNG
   // the same network as SCL:
   "DB16000_OPC_UA_TRIGGER_ALARM".CLIENT.U2_STA3_COAXIAL.ALARMS.CAM_START_JET_CALIB_METHOD_WORKING_BLOCKED_A := (("DB16343_U2_STA3_CAM_JET_CALIBRATE_TRIG".Done AND ("DB16005_U2_STA3_COAXIAL_CLIENT_INTERFACE".U2_STA3_CAM_Calibrations."Calibrate jet".Outputs.Result <> 0)) OR ("DB16000_OPC_UA_TRIGGER_ALARM".CLIENT.U2_STA3_COAXIAL.ALARMS.CAM_START_JET_CALIB_METHOD_WORKING_BLOCKED_A AND NOT "DB2120_MPP_ITC_IPC".RESET_FAULTS)) AND "DB7257_UNIT_2_STA_3_COAXIAL_ENABLE_DISABLE".ENABLED;
   "DB426_ALARMS_WARNINGS".ALARMS.UNIT_02.STATION_3_COAXIAL."720897" := "DB16000_OPC_UA_TRIGGER_ALARM".CLIENT.U2_STA3_COAXIAL.ALARMS.CAM_START_JET_CALIB_METHOD_WORKING_BLOCKED_A;
END_REGION

REGION Network 63: UNIT 2 STATION 3 COAXIAL CAMERA START CLADDING CALIBRATION METHOD CONNECTION ALARM
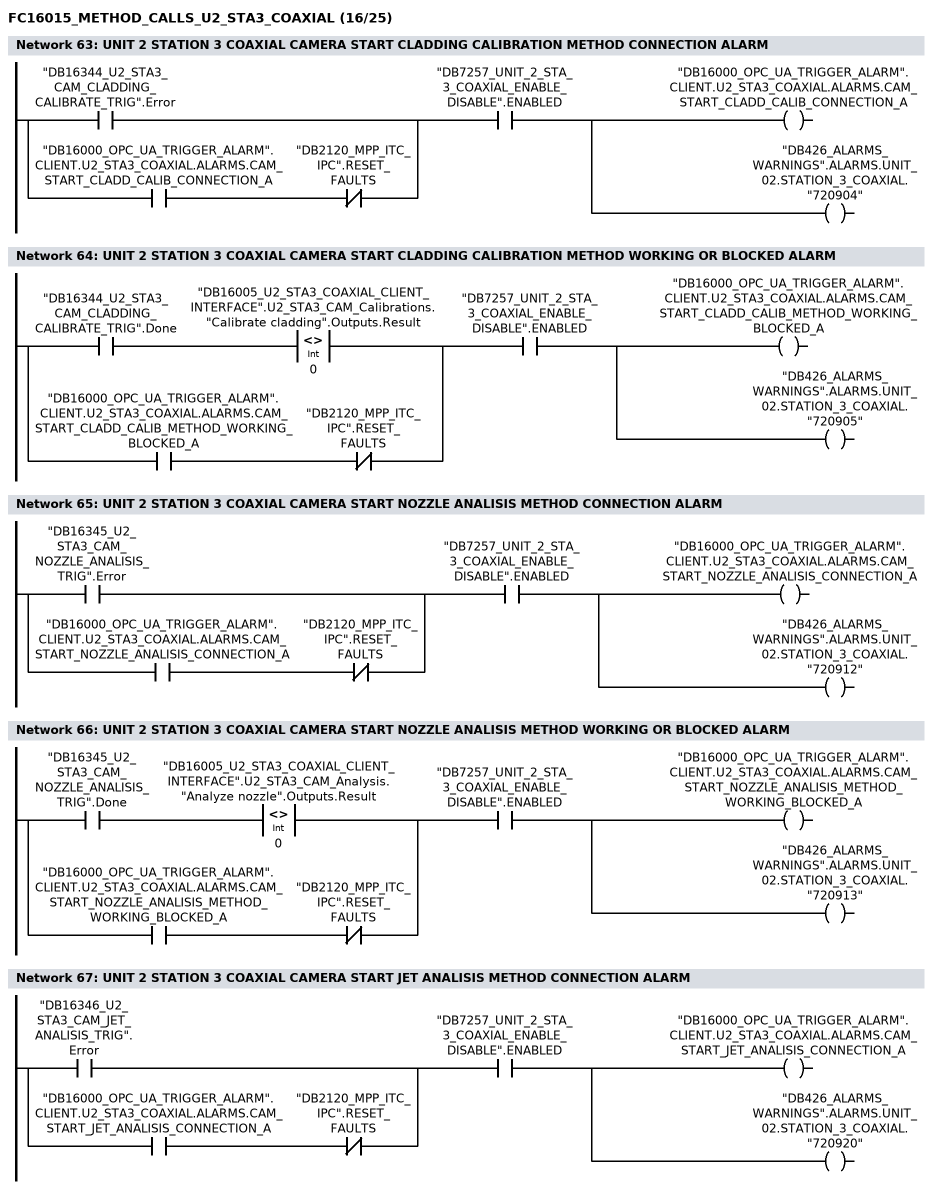
   RUNG wire#powerrail
      Contact( "DB16344_U2_STA3_CAM_CLADDING_CALIBRATE_TRIG".Error )
      wire#w1
      Contact( "DB7257_UNIT_2_STA_3_COAXIAL_ENABLE_DISABLE".ENABLED )
      wire#w2
      Coil( "DB16000_OPC_UA_TRIGGER_ALARM".CLIENT.U2_STA3_COAXIAL.ALARMS.CAM_START_CLADD_CALIB_CONNECTION_A )
   END_RUNG
   RUNG wire#powerrail
      Contact( "DB16000_OPC_UA_TRIGGER_ALARM".CLIENT.U2_STA3_COAXIAL.ALARMS.CAM_START_CLADD_CALIB_CONNECTION_A )
      I_Contact( "DB2120_MPP_ITC_IPC".RESET_FAULTS )
   END_RUNG wire#w1
   RUNG wire#w2
      Coil( "DB426_ALARMS_WARNINGS".ALARMS.UNIT_02.STATION_3_COAXIAL."720904" )
   END_RUNG
   // the same network as SCL:
   "DB16000_OPC_UA_TRIGGER_ALARM".CLIENT.U2_STA3_COAXIAL.ALARMS.CAM_START_CLADD_CALIB_CONNECTION_A := ("DB16344_U2_STA3_CAM_CLADDING_CALIBRATE_TRIG".Error OR ("DB16000_OPC_UA_TRIGGER_ALARM".CLIENT.U2_STA3_COAXIAL.ALARMS.CAM_START_CLADD_CALIB_CONNECTION_A AND NOT "DB2120_MPP_ITC_IPC".RESET_FAULTS)) AND "DB7257_UNIT_2_STA_3_COAXIAL_ENABLE_DISABLE".ENABLED;
   "DB426_ALARMS_WARNINGS".ALARMS.UNIT_02.STATION_3_COAXIAL."720904" := "DB16000_OPC_UA_TRIGGER_ALARM".CLIENT.U2_STA3_COAXIAL.ALARMS.CAM_START_CLADD_CALIB_CONNECTION_A;
END_REGION

REGION Network 64: UNIT 2 STATION 3 COAXIAL CAMERA START CLADDING CALIBRATION METHOD WORKING OR BLOCKED ALARM
   RUNG wire#powerrail
      Contact( "DB16344_U2_STA3_CAM_CLADDING_CALIBRATE_TRIG".Done )
      { S7_Templates := "SrcType := Int" } NE_Contact(in1 := "DB16005_U2_STA3_COAXIAL_CLIENT_INTERFACE".U2_STA3_CAM_Calibrations."Calibrate cladding".Outputs.Result, in2 := 0)
      wire#w1
      Contact( "DB7257_UNIT_2_STA_3_COAXIAL_ENABLE_DISABLE".ENABLED )
      wire#w2
      Coil( "DB16000_OPC_UA_TRIGGER_ALARM".CLIENT.U2_STA3_COAXIAL.ALARMS.CAM_START_CLADD_CALIB_METHOD_WORKING_BLOCKED_A )
   END_RUNG
   RUNG wire#powerrail
      Contact( "DB16000_OPC_UA_TRIGGER_ALARM".CLIENT.U2_STA3_COAXIAL.ALARMS.CAM_START_CLADD_CALIB_METHOD_WORKING_BLOCKED_A )
      I_Contact( "DB2120_MPP_ITC_IPC".RESET_FAULTS )
   END_RUNG wire#w1
   RUNG wire#w2
      Coil( "DB426_ALARMS_WARNINGS".ALARMS.UNIT_02.STATION_3_COAXIAL."720905" )
   END_RUNG
   // the same network as SCL:
   "DB16000_OPC_UA_TRIGGER_ALARM".CLIENT.U2_STA3_COAXIAL.ALARMS.CAM_START_CLADD_CALIB_METHOD_WORKING_BLOCKED_A := (("DB16344_U2_STA3_CAM_CLADDING_CALIBRATE_TRIG".Done AND ("DB16005_U2_STA3_COAXIAL_CLIENT_INTERFACE".U2_STA3_CAM_Calibrations."Calibrate cladding".Outputs.Result <> 0)) OR ("DB16000_OPC_UA_TRIGGER_ALARM".CLIENT.U2_STA3_COAXIAL.ALARMS.CAM_START_CLADD_CALIB_METHOD_WORKING_BLOCKED_A AND NOT "DB2120_MPP_ITC_IPC".RESET_FAULTS)) AND "DB7257_UNIT_2_STA_3_COAXIAL_ENABLE_DISABLE".ENABLED;
   "DB426_ALARMS_WARNINGS".ALARMS.UNIT_02.STATION_3_COAXIAL."720905" := "DB16000_OPC_UA_TRIGGER_ALARM".CLIENT.U2_STA3_COAXIAL.ALARMS.CAM_START_CLADD_CALIB_METHOD_WORKING_BLOCKED_A;
END_REGION

REGION Network 65: UNIT 2 STATION 3 COAXIAL CAMERA START NOZZLE ANALISIS METHOD CONNECTION ALARM
   RUNG wire#powerrail
      Contact( "DB16345_U2_STA3_CAM_NOZZLE_ANALISIS_TRIG".Error )
      wire#w1
      Contact( "DB7257_UNIT_2_STA_3_COAXIAL_ENABLE_DISABLE".ENABLED )
      wire#w2
      Coil( "DB16000_OPC_UA_TRIGGER_ALARM".CLIENT.U2_STA3_COAXIAL.ALARMS.CAM_START_NOZZLE_ANALISIS_CONNECTION_A )
   END_RUNG
   RUNG wire#powerrail
      Contact( "DB16000_OPC_UA_TRIGGER_ALARM".CLIENT.U2_STA3_COAXIAL.ALARMS.CAM_START_NOZZLE_ANALISIS_CONNECTION_A )
      I_Contact( "DB2120_MPP_ITC_IPC".RESET_FAULTS )
   END_RUNG wire#w1
   RUNG wire#w2
      Coil( "DB426_ALARMS_WARNINGS".ALARMS.UNIT_02.STATION_3_COAXIAL."720912" )
   END_RUNG
   // the same network as SCL:
   "DB16000_OPC_UA_TRIGGER_ALARM".CLIENT.U2_STA3_COAXIAL.ALARMS.CAM_START_NOZZLE_ANALISIS_CONNECTION_A := ("DB16345_U2_STA3_CAM_NOZZLE_ANALISIS_TRIG".Error OR ("DB16000_OPC_UA_TRIGGER_ALARM".CLIENT.U2_STA3_COAXIAL.ALARMS.CAM_START_NOZZLE_ANALISIS_CONNECTION_A AND NOT "DB2120_MPP_ITC_IPC".RESET_FAULTS)) AND "DB7257_UNIT_2_STA_3_COAXIAL_ENABLE_DISABLE".ENABLED;
   "DB426_ALARMS_WARNINGS".ALARMS.UNIT_02.STATION_3_COAXIAL."720912" := "DB16000_OPC_UA_TRIGGER_ALARM".CLIENT.U2_STA3_COAXIAL.ALARMS.CAM_START_NOZZLE_ANALISIS_CONNECTION_A;
END_REGION

